REGION Network 8: XỬ LÍ CÂN CỐT LIỆU
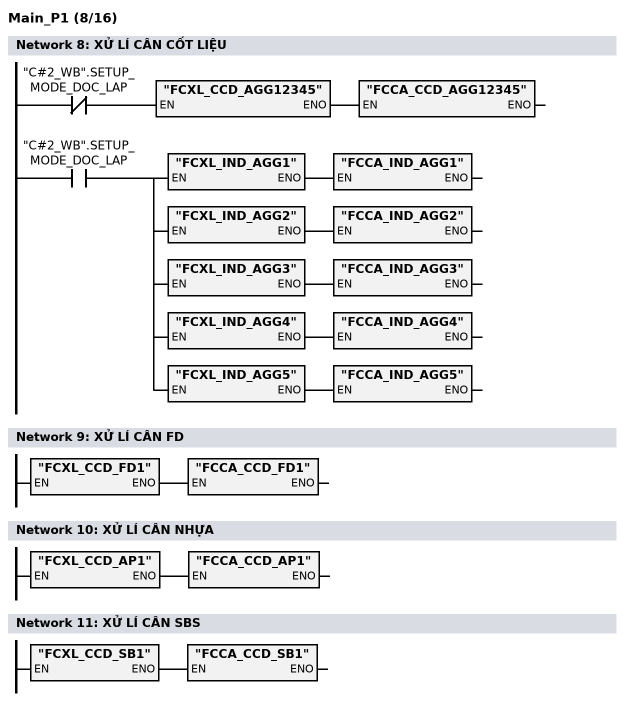
   RUNG wire#powerrail
      I_Contact( "C#2_WB".SETUP_MODE_DOC_LAP )
      "FCXL_CCD_AGG12345"()
      "FCCA_CCD_AGG12345"()
   END_RUNG
   RUNG wire#powerrail
      Contact( "C#2_WB".SETUP_MODE_DOC_LAP )
      wire#w1
      "FCXL_IND_AGG1"()
      "FCCA_IND_AGG1"()
   END_RUNG
   RUNG wire#w1
      "FCXL_IND_AGG2"()
      "FCCA_IND_AGG2"()
   END_RUNG
   RUNG wire#w1
      "FCXL_IND_AGG3"()
      "FCCA_IND_AGG3"()
   END_RUNG
   RUNG wire#w1
      "FCXL_IND_AGG4"()
      "FCCA_IND_AGG4"()
   END_RUNG
   RUNG wire#w1
      "FCXL_IND_AGG5"()
      "FCCA_IND_AGG5"()
   END_RUNG
   // the same network as SCL:
   "FCXL_CCD_AGG12345"(EN := NOT "C#2_WB".SETUP_MODE_DOC_LAP, ENO => #_w1);
   IF #_w1 THEN "FCCA_CCD_AGG12345"(); END_IF;
   #_w3 := "C#2_WB".SETUP_MODE_DOC_LAP;
   "FCXL_IND_AGG1"(EN := "C#2_WB".SETUP_MODE_DOC_LAP, ENO => #_w2);
   IF #_w2 THEN "FCCA_IND_AGG1"(); END_IF;
   "FCXL_IND_AGG2"(EN := #_w3, ENO => #_w4);
   IF #_w4 THEN "FCCA_IND_AGG2"(); END_IF;
   "FCXL_IND_AGG3"(EN := #_w3, ENO => #_w5);
   IF #_w5 THEN "FCCA_IND_AGG3"(); END_IF;
   "FCXL_IND_AGG4"(EN := #_w3, ENO => #_w6);
   IF #_w6 THEN "FCCA_IND_AGG4"(); END_IF;
   "FCXL_IND_AGG5"(EN := #_w3, ENO => #_w7);
   IF #_w7 THEN "FCCA_IND_AGG5"(); END_IF;
END_REGION

REGION Network 9: XỬ LÍ CÂN FD
   RUNG wire#powerrail
      "FCXL_CCD_FD1"()
      "FCCA_CCD_FD1"()
   END_RUNG
   // the same network as SCL:
   "FCXL_CCD_FD1"(ENO => #_w1);
   IF #_w1 THEN "FCCA_CCD_FD1"(); END_IF;
END_REGION

REGION Network 10: XỬ LÍ CÂN NHỰA
   RUNG wire#powerrail
      "FCXL_CCD_AP1"()
      "FCCA_CCD_AP1"()
   END_RUNG
   // the same network as SCL:
   "FCXL_CCD_AP1"(ENO => #_w1);
   IF #_w1 THEN "FCCA_CCD_AP1"(); END_IF;
END_REGION

REGION Network 11: XỬ LÍ CÂN SBS
   RUNG wire#powerrail
      "FCXL_CCD_SB1"()
      "FCCA_CCD_SB1"()
   END_RUNG
   // the same network as SCL:
   "FCXL_CCD_SB1"(ENO => #_w1);
   IF #_w1 THEN "FCCA_CCD_SB1"(); END_IF;
END_REGION

REGION Network 12: NẠP LIỆU NỒI TRỘN
   // Theo phân tích thì lẽ ra lệnh so sánh SV_FD1=0 nó phải bypass cả WCE1_FU thì mới đúng vì nếu theo logic cũ trong hàm xử lý cân (FC10 của FD1) tín hiệu SV_FD1=0 không bypass /NEXT_WCEM1 khiến WCE1_FU sẽ không được bật ON khi SV_FD1=0, dẫn đến mạch hở, không nạp liệu được.
   // Sau đó trong quá trình sửa đã bypass trong FC10, tuy nhiên làm như thế không hay, vì có cân đâu mà bảo nó FULL, vậy nên hay nhất sẽ là sửa ở đây, bypass WCE1_FU nếu như Setpoint của FD1=0
   // Lưu ý:
   // - Nhựa nóng thì cần có AP1 nên mới có lệnh so sánh SMX_AP1=SMC_MIXER và lệnh tiếp điểm WWA1_FU (cân đủ số mẻ và Full thì mới nạp được)
   // - Chỉ bypass bột đá FD1 hoặc phụ gia SB1 hoặc thậm chí bypass cả 2, nhưng không có chuyện bypass AP1
   // Nhựa nóng nên phải có nhựa, đó là lý do network này đang dự vào SMC_AP1 để so sánh với các SMC của các phểu cân FD1 và SBS1 (khoogn có AG1), mục đích là để kiểm tra xem các phểu cân đã được cân đầy và đủ thành phần chưa (có FD1/SBS1 không) (****)
   // - Lệnh so sánh SMX_FD1 hoặc SMX_SB1 với số mẻ trộn SMC_MIXER mục đích là để đảm bảo việc nạp liệu nó cần lặp lại giữa các mẻ. Logic ở đây là:
   // - Khi chưa nạp liêu (chưa nạp mẻ nào) thì SMC_MIXER tất nhiên là zero, và tất nhiên 2 thằng FD1 và SB1 nó cũng bằng zero, vì nó đã xả vào nồi mẻ nào đâu (lưu ý là sau khi nạp liệu xong thì biến NTR_FU sẽ bật và SMC_MIXER lúc này tăng lên 1)
   // - Vậy nên điều kiện này đúng, và tất nhiên trước khi xả thì tất cả các phểu cân phải có số mẻ cân bằng nhau nên nhận định 4**** ở trên là đúng (SMC_AP1=SMC_FD1=SMC_SB1), trừ khi không cân các thành phần này thì nó không bằng nhau, thì lúc đó có lệnh bypass lo.
   // - Còn lệnh so sánh SMX_AP1=SMC_MIXER là để kiểm tra việc xả các phểu cân liệu xong, rồi tới lúc nồi trộn nạp đầy NTR_FU thì SMC_MIXER tăng lên 1 (xem network13), đủ đk này thì mới nạp liệu lại được (nạp cho mẻ tiếp theo), logic ở đây là: lúc đầu chưa xả cái phểu nào thì 2 thông số này đều bằng zero đúng không, vậy thõa đk và có thể cho NẠP LIỆU, sau khi thằng AG1 nó xả/nạp vào nồi trộn thì SMX của nó tăng lên, tương tự cac phểu khác cũng có SMX tăng lên 1, trong đó có AP1, như vậy là NAP LIEU kết thúc, mà sau khi nạp liệu xong thì thằng nồi trộn nó phải xả ra chứ đúng không, vậy là một lúc sau khi nó trộn xong nó sẽ cả, lúc này SMX_MIXER sẽ tăng lên 1, làm điều kiện cần để cho một chu kỳ xả hay NẠP LIỆU tiếp theo.
   // - Sẽ có đứa hỏi, khi xả thì sẽ có thằng xả trước thằng xả sau, dẫn đến điều kiện so sánh nó không thỏa, mạch hở, NAP LIEU sẽ OFF, ví dụ như thằng SB1 nó ít nên nó xả lẹ hơn, empty sớm hơn mấy thằng kia, dẫn đến số mẻ xả của nó được tăng lên 1 sớm hơn, khi đó mất bit NAP LIEU thì các phểu các sao kịp xả.
   // ==> OK, phân tích tôt, nhưng chưa đủ sâu, cần phải biết là để xả/nạp liệu thì các phểu phải cân đủ liệu, và phải sẵn sàng hết tất cả sau đó mới nạp (tức thời điểm đó các điều kiện ở trên đều đã sẵn sàng), thứ 2 là NAP LIEU chỉ là đk cần cho việc bật tín hiệu NẠP tương ứng với tưng phểu cân, nhìn vào lệnh bên dưới sẽ thấy, và khi có NAP LIEU thì các tín hiệu sẽ được set lên đồng thời (vì điều kiện đã đợi sẵn hết cả rồi thím ợ, chỉ cần nhú lên là quất thôi).
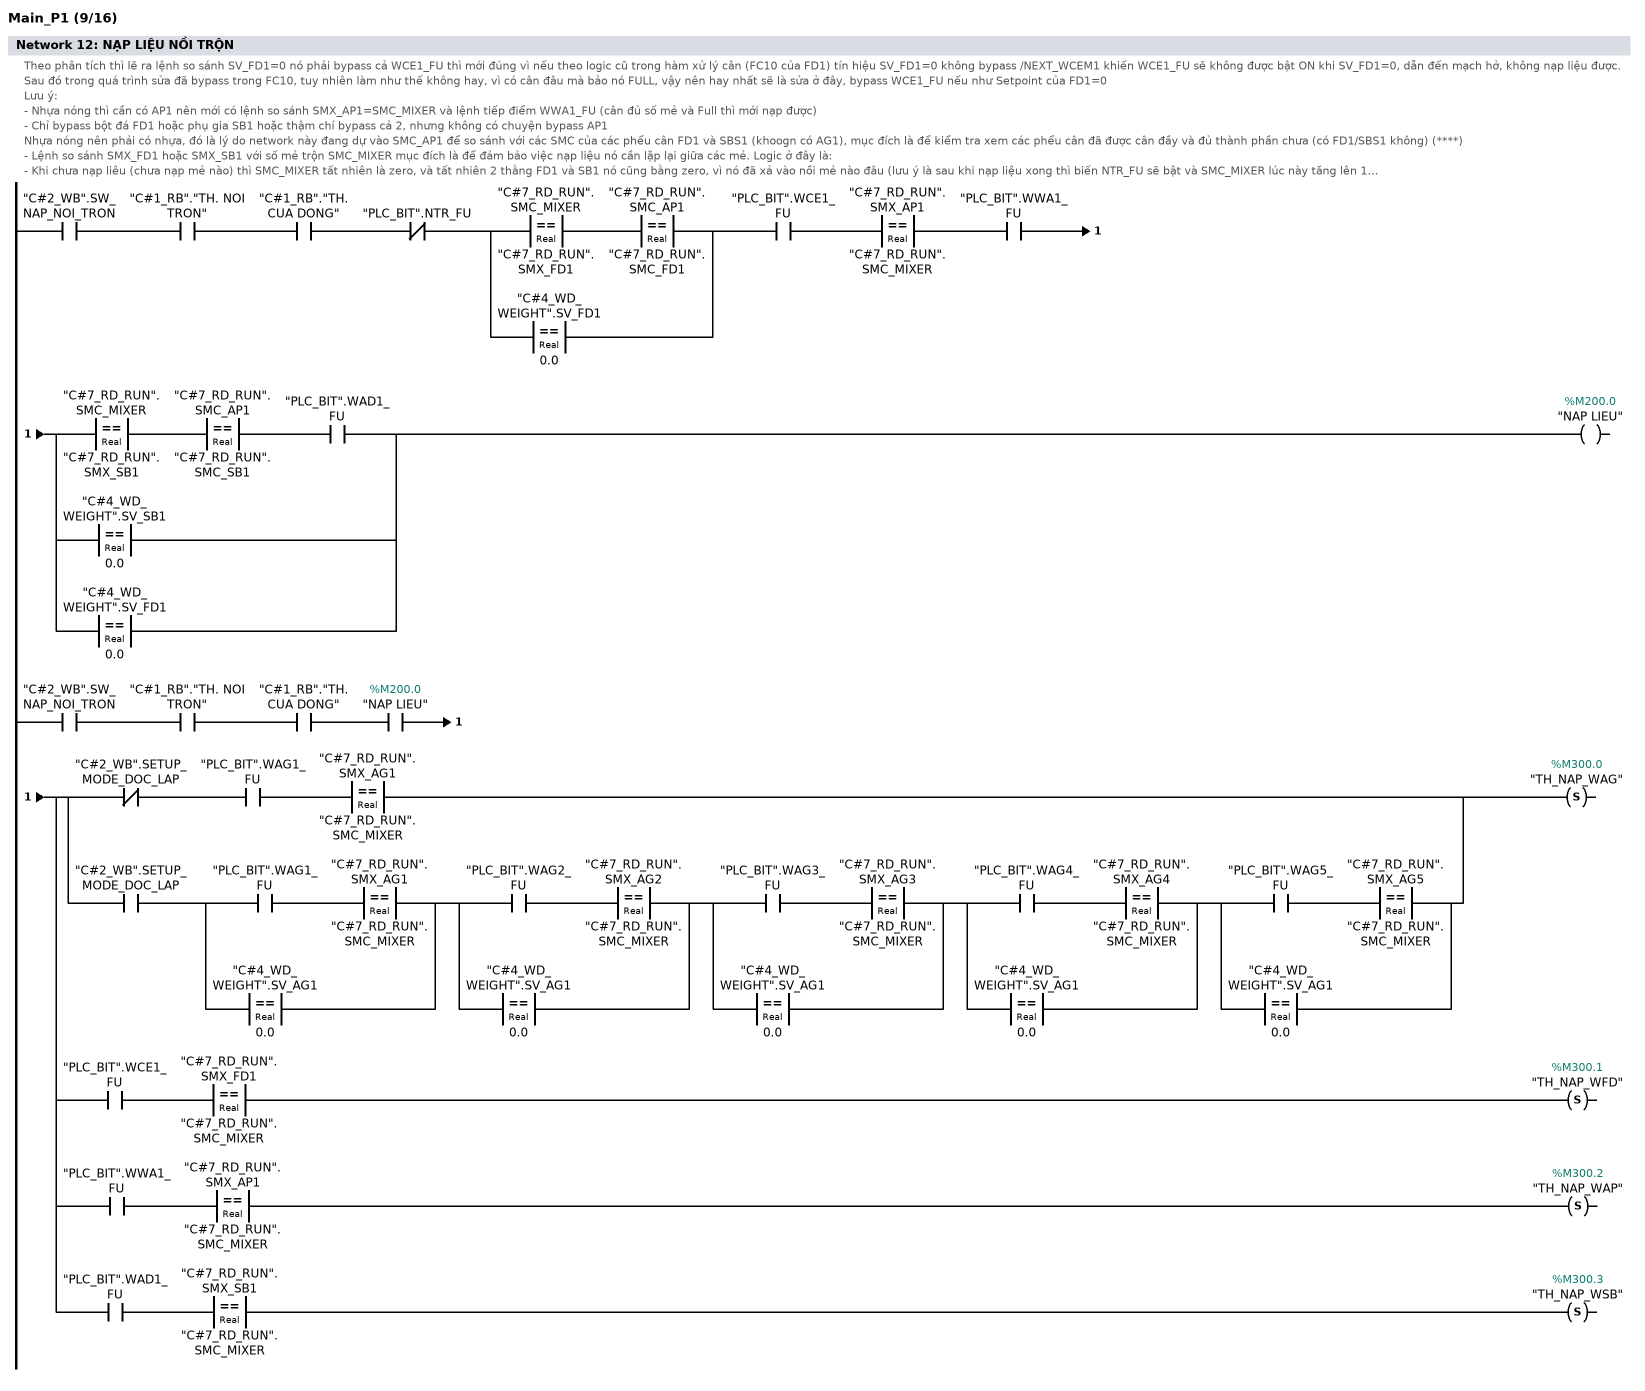
   RUNG wire#powerrail
      Contact( "C#2_WB".SW_NAP_NOI_TRON )
      Contact( "C#1_RB"."TH. NOI TRON" )
      Contact( "C#1_RB"."TH. CUA DONG" )
      I_Contact( "PLC_BIT".NTR_FU )
      wire#w1
      { S7_Templates := "SrcType := Real" } EQ_Contact(in1 := "C#7_RD_RUN".SMC_MIXER, in2 := "C#7_RD_RUN".SMX_FD1)
      { S7_Templates := "SrcType := Real" } EQ_Contact(in1 := "C#7_RD_RUN".SMC_AP1, in2 := "C#7_RD_RUN".SMC_FD1)
      wire#w2
      Contact( "PLC_BIT".WCE1_FU )
      { S7_Templates := "SrcType := Real" } EQ_Contact(in1 := "C#7_RD_RUN".SMX_AP1, in2 := "C#7_RD_RUN".SMC_MIXER)
      Contact( "PLC_BIT".WWA1_FU )
      wire#w3
      { S7_Templates := "SrcType := Real" } EQ_Contact(in1 := "C#7_RD_RUN".SMC_MIXER, in2 := "C#7_RD_RUN".SMX_SB1)
      { S7_Templates := "SrcType := Real" } EQ_Contact(in1 := "C#7_RD_RUN".SMC_AP1, in2 := "C#7_RD_RUN".SMC_SB1)
      Contact( "PLC_BIT".WAD1_FU )
      wire#w4
      Coil( "NAP LIEU" )
   END_RUNG
   RUNG wire#w1
      { S7_Templates := "SrcType := Real" } EQ_Contact(in1 := "C#4_WD_WEIGHT".SV_FD1, in2 := 0.0)
   END_RUNG wire#w2
   RUNG wire#w3
      { S7_Templates := "SrcType := Real" } EQ_Contact(in1 := "C#4_WD_WEIGHT".SV_SB1, in2 := 0.0)
   END_RUNG wire#w4
   RUNG wire#w3
      { S7_Templates := "SrcType := Real" } EQ_Contact(in1 := "C#4_WD_WEIGHT".SV_FD1, in2 := 0.0)
   END_RUNG wire#w4
   RUNG wire#powerrail
      Contact( "C#2_WB".SW_NAP_NOI_TRON )
      Contact( "C#1_RB"."TH. NOI TRON" )
      Contact( "C#1_RB"."TH. CUA DONG" )
      Contact( "NAP LIEU" )
      wire#w5
      I_Contact( "C#2_WB".SETUP_MODE_DOC_LAP )
      Contact( "PLC_BIT".WAG1_FU )
      { S7_Templates := "SrcType := Real" } EQ_Contact(in1 := "C#7_RD_RUN".SMX_AG1, in2 := "C#7_RD_RUN".SMC_MIXER)
      wire#w6
      S_Coil( "TH_NAP_WAG" )
   END_RUNG
   RUNG wire#w5
      Contact( "C#2_WB".SETUP_MODE_DOC_LAP )
      wire#w7
      Contact( "PLC_BIT".WAG1_FU )
      { S7_Templates := "SrcType := Real" } EQ_Contact(in1 := "C#7_RD_RUN".SMX_AG1, in2 := "C#7_RD_RUN".SMC_MIXER)
      wire#w8
      Contact( "PLC_BIT".WAG2_FU )
      { S7_Templates := "SrcType := Real" } EQ_Contact(in1 := "C#7_RD_RUN".SMX_AG2, in2 := "C#7_RD_RUN".SMC_MIXER)
      wire#w9
      Contact( "PLC_BIT".WAG3_FU )
      { S7_Templates := "SrcType := Real" } EQ_Contact(in1 := "C#7_RD_RUN".SMX_AG3, in2 := "C#7_RD_RUN".SMC_MIXER)
      wire#w10
      Contact( "PLC_BIT".WAG4_FU )
      { S7_Templates := "SrcType := Real" } EQ_Contact(in1 := "C#7_RD_RUN".SMX_AG4, in2 := "C#7_RD_RUN".SMC_MIXER)
      wire#w11
      Contact( "PLC_BIT".WAG5_FU )
      { S7_Templates := "SrcType := Real" } EQ_Contact(in1 := "C#7_RD_RUN".SMX_AG5, in2 := "C#7_RD_RUN".SMC_MIXER)
   END_RUNG wire#w6
   RUNG wire#w7
      { S7_Templates := "SrcType := Real" } EQ_Contact(in1 := "C#4_WD_WEIGHT".SV_AG1, in2 := 0.0)
   END_RUNG wire#w8
   RUNG wire#w8
      { S7_Templates := "SrcType := Real" } EQ_Contact(in1 := "C#4_WD_WEIGHT".SV_AG1, in2 := 0.0)
   END_RUNG wire#w9
   RUNG wire#w9
      { S7_Templates := "SrcType := Real" } EQ_Contact(in1 := "C#4_WD_WEIGHT".SV_AG1, in2 := 0.0)
   END_RUNG wire#w10
   RUNG wire#w10
      { S7_Templates := "SrcType := Real" } EQ_Contact(in1 := "C#4_WD_WEIGHT".SV_AG1, in2 := 0.0)
   END_RUNG wire#w11
   RUNG wire#w11
      { S7_Templates := "SrcType := Real" } EQ_Contact(in1 := "C#4_WD_WEIGHT".SV_AG1, in2 := 0.0)
   END_RUNG wire#w6
   RUNG wire#w5
      Contact( "PLC_BIT".WCE1_FU )
      { S7_Templates := "SrcType := Real" } EQ_Contact(in1 := "C#7_RD_RUN".SMX_FD1, in2 := "C#7_RD_RUN".SMC_MIXER)
      S_Coil( "TH_NAP_WFD" )
   END_RUNG
   RUNG wire#w5
      Contact( "PLC_BIT".WWA1_FU )
      { S7_Templates := "SrcType := Real" } EQ_Contact(in1 := "C#7_RD_RUN".SMX_AP1, in2 := "C#7_RD_RUN".SMC_MIXER)
      S_Coil( "TH_NAP_WAP" )
   END_RUNG
   RUNG wire#w5
      Contact( "PLC_BIT".WAD1_FU )
      { S7_Templates := "SrcType := Real" } EQ_Contact(in1 := "C#7_RD_RUN".SMX_SB1, in2 := "C#7_RD_RUN".SMC_MIXER)
      S_Coil( "TH_NAP_WSB" )
   END_RUNG
   // the same network as SCL:
   "NAP LIEU" := "C#2_WB".SW_NAP_NOI_TRON AND "C#1_RB"."TH. NOI TRON" AND "C#1_RB"."TH. CUA DONG" AND NOT "PLC_BIT".NTR_FU AND ((("C#7_RD_RUN".SMC_MIXER = "C#7_RD_RUN".SMX_FD1) AND ("C#7_RD_RUN".SMC_AP1 = "C#7_RD_RUN".SMC_FD1)) OR ("C#4_WD_WEIGHT".SV_FD1 = 0.0)) AND "PLC_BIT".WCE1_FU AND ("C#7_RD_RUN".SMX_AP1 = "C#7_RD_RUN".SMC_MIXER) AND "PLC_BIT".WWA1_FU AND ((("C#7_RD_RUN".SMC_MIXER = "C#7_RD_RUN".SMX_SB1) AND ("C#7_RD_RUN".SMC_AP1 = "C#7_RD_RUN".SMC_SB1) AND "PLC_BIT".WAD1_FU) OR ("C#4_WD_WEIGHT".SV_SB1 = 0.0) OR ("C#4_WD_WEIGHT".SV_FD1 = 0.0));
   #_w1 := "C#2_WB".SW_NAP_NOI_TRON AND "C#1_RB"."TH. NOI TRON" AND "C#1_RB"."TH. CUA DONG" AND "NAP LIEU";
   IF #_w1 AND ((NOT "C#2_WB".SETUP_MODE_DOC_LAP AND "PLC_BIT".WAG1_FU AND ("C#7_RD_RUN".SMX_AG1 = "C#7_RD_RUN".SMC_MIXER)) OR ("C#2_WB".SETUP_MODE_DOC_LAP AND (("PLC_BIT".WAG1_FU AND ("C#7_RD_RUN".SMX_AG1 = "C#7_RD_RUN".SMC_MIXER)) OR ("C#4_WD_WEIGHT".SV_AG1 = 0.0)) AND (("PLC_BIT".WAG2_FU AND ("C#7_RD_RUN".SMX_AG2 = "C#7_RD_RUN".SMC_MIXER)) OR ("C#4_WD_WEIGHT".SV_AG1 = 0.0)) AND (("PLC_BIT".WAG3_FU AND ("C#7_RD_RUN".SMX_AG3 = "C#7_RD_RUN".SMC_MIXER)) OR ("C#4_WD_WEIGHT".SV_AG1 = 0.0)) AND (("PLC_BIT".WAG4_FU AND ("C#7_RD_RUN".SMX_AG4 = "C#7_RD_RUN".SMC_MIXER)) OR ("C#4_WD_WEIGHT".SV_AG1 = 0.0)) AND (("PLC_BIT".WAG5_FU AND ("C#7_RD_RUN".SMX_AG5 = "C#7_RD_RUN".SMC_MIXER)) OR ("C#4_WD_WEIGHT".SV_AG1 = 0.0)))) THEN
       "TH_NAP_WAG" := TRUE;
   END_IF;
   IF #_w1 AND "PLC_BIT".WCE1_FU AND ("C#7_RD_RUN".SMX_FD1 = "C#7_RD_RUN".SMC_MIXER) THEN
       "TH_NAP_WFD" := TRUE;
   END_IF;
   IF #_w1 AND "PLC_BIT".WWA1_FU AND ("C#7_RD_RUN".SMX_AP1 = "C#7_RD_RUN".SMC_MIXER) THEN
       "TH_NAP_WAP" := TRUE;
   END_IF;
   IF #_w1 AND "PLC_BIT".WAD1_FU AND ("C#7_RD_RUN".SMX_SB1 = "C#7_RD_RUN".SMC_MIXER) THEN
       "TH_NAP_WSB" := TRUE;
   END_IF;
END_REGION

REGION Network 13: XỬ LÍ NỒI TRỘN
   // Đây là network xử lý tình huống là các phểu đã nạp/xả vào nồi trộn rồi, nhưng nồi trộn chưa có xả nhé (có thể là nó đang trộn nên mới đặt tên là NTR_FU, chứ thực tế thằng nồi trộn nó có cân mẹ đâu mà Full với không).
   // Lệnh so sánh SMX_AP1>SMC_MIXER sẽ thỏa, vì trước khi nạp vào nồi trộn thì SMC_AP1 cũng như các phểu cân khác đều sẽ lơn hơn SMC_MIXER, vụ thể là 1>0. mục đích là để việc bật bít NTR_FU diễn ra trước khi SMC_MIXER tăng lên 1, vì điều kiện đếm tăng là cạnh lên của NTR_FU mà.
   // @@@ XUỐNG TỚI NETWORK NÀY THÌ SMC_MIXER MỚI ĐƯỢC TĂNG LÊN 1@@@
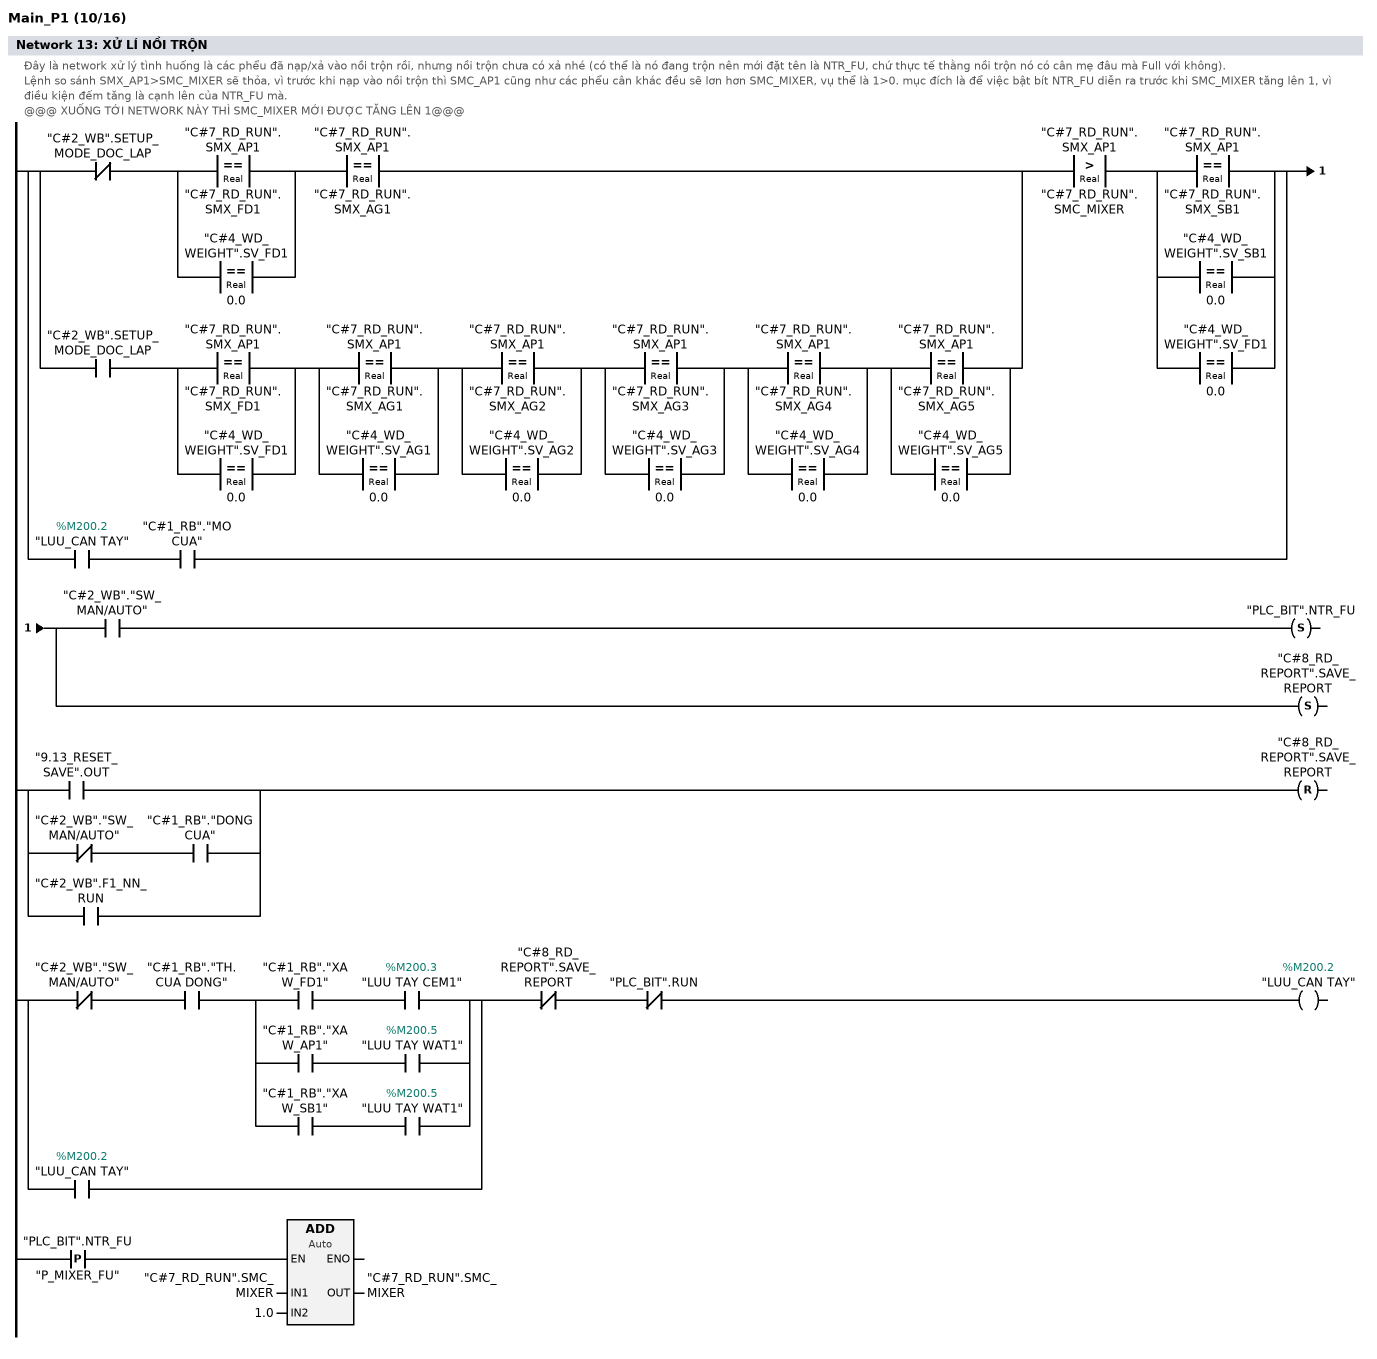
   RUNG wire#powerrail
      I_Contact( "C#2_WB".SETUP_MODE_DOC_LAP )
      wire#w1
      { S7_Templates := "SrcType := Real" } EQ_Contact(in1 := "C#7_RD_RUN".SMX_AP1, in2 := "C#7_RD_RUN".SMX_FD1)
      wire#w2
      { S7_Templates := "SrcType := Real" } EQ_Contact(in1 := "C#7_RD_RUN".SMX_AP1, in2 := "C#7_RD_RUN".SMX_AG1)
      wire#w3
      { S7_Templates := "SrcType := Real" } GT_Contact(in1 := "C#7_RD_RUN".SMX_AP1, in2 := "C#7_RD_RUN".SMC_MIXER)
      wire#w10
      { S7_Templates := "SrcType := Real" } EQ_Contact(in1 := "C#7_RD_RUN".SMX_AP1, in2 := "C#7_RD_RUN".SMX_SB1)
      wire#w11
      Contact( "C#2_WB"."SW_MAN/AUTO" )
      S_Coil( "PLC_BIT".NTR_FU )
   END_RUNG
   RUNG wire#w1
      { S7_Templates := "SrcType := Real" } EQ_Contact(in1 := "C#4_WD_WEIGHT".SV_FD1, in2 := 0.0)
   END_RUNG wire#w2
   RUNG wire#powerrail
      Contact( "C#2_WB".SETUP_MODE_DOC_LAP )
      wire#w4
      { S7_Templates := "SrcType := Real" } EQ_Contact(in1 := "C#7_RD_RUN".SMX_AP1, in2 := "C#7_RD_RUN".SMX_FD1)
      wire#w5
      { S7_Templates := "SrcType := Real" } EQ_Contact(in1 := "C#7_RD_RUN".SMX_AP1, in2 := "C#7_RD_RUN".SMX_AG1)
      wire#w6
      { S7_Templates := "SrcType := Real" } EQ_Contact(in1 := "C#7_RD_RUN".SMX_AP1, in2 := "C#7_RD_RUN".SMX_AG2)
      wire#w7
      { S7_Templates := "SrcType := Real" } EQ_Contact(in1 := "C#7_RD_RUN".SMX_AP1, in2 := "C#7_RD_RUN".SMX_AG3)
      wire#w8
      { S7_Templates := "SrcType := Real" } EQ_Contact(in1 := "C#7_RD_RUN".SMX_AP1, in2 := "C#7_RD_RUN".SMX_AG4)
      wire#w9
      { S7_Templates := "SrcType := Real" } EQ_Contact(in1 := "C#7_RD_RUN".SMX_AP1, in2 := "C#7_RD_RUN".SMX_AG5)
   END_RUNG wire#w3
   RUNG wire#w4
      { S7_Templates := "SrcType := Real" } EQ_Contact(in1 := "C#4_WD_WEIGHT".SV_FD1, in2 := 0.0)
   END_RUNG wire#w5
   RUNG wire#w5
      { S7_Templates := "SrcType := Real" } EQ_Contact(in1 := "C#4_WD_WEIGHT".SV_AG1, in2 := 0.0)
   END_RUNG wire#w6
   RUNG wire#w6
      { S7_Templates := "SrcType := Real" } EQ_Contact(in1 := "C#4_WD_WEIGHT".SV_AG2, in2 := 0.0)
   END_RUNG wire#w7
   RUNG wire#w7
      { S7_Templates := "SrcType := Real" } EQ_Contact(in1 := "C#4_WD_WEIGHT".SV_AG3, in2 := 0.0)
   END_RUNG wire#w8
   RUNG wire#w8
      { S7_Templates := "SrcType := Real" } EQ_Contact(in1 := "C#4_WD_WEIGHT".SV_AG4, in2 := 0.0)
   END_RUNG wire#w9
   RUNG wire#w9
      { S7_Templates := "SrcType := Real" } EQ_Contact(in1 := "C#4_WD_WEIGHT".SV_AG5, in2 := 0.0)
   END_RUNG wire#w3
   RUNG wire#w10
      { S7_Templates := "SrcType := Real" } EQ_Contact(in1 := "C#4_WD_WEIGHT".SV_SB1, in2 := 0.0)
   END_RUNG wire#w11
   RUNG wire#w10
      { S7_Templates := "SrcType := Real" } EQ_Contact(in1 := "C#4_WD_WEIGHT".SV_FD1, in2 := 0.0)
   END_RUNG wire#w11
   RUNG wire#powerrail
      Contact( "LUU_CAN TAY" )
      Contact( "C#1_RB"."MO CUA" )
   END_RUNG wire#w11
   RUNG wire#w11
      S_Coil( "C#8_RD_REPORT".SAVE_REPORT )
   END_RUNG
   RUNG wire#powerrail
      Contact( "9.13_RESET_SAVE".OUT )
      wire#w12
      R_Coil( "C#8_RD_REPORT".SAVE_REPORT )
   END_RUNG
   RUNG wire#powerrail
      I_Contact( "C#2_WB"."SW_MAN/AUTO" )
      Contact( "C#1_RB"."DONG CUA" )
   END_RUNG wire#w12
   RUNG wire#powerrail
      Contact( "C#2_WB".F1_NN_RUN )
   END_RUNG wire#w12
   RUNG wire#powerrail
      I_Contact( "C#2_WB"."SW_MAN/AUTO" )
      Contact( "C#1_RB"."TH. CUA DONG" )
      wire#w13
      Contact( "C#1_RB"."XA W_FD1" )
      Contact( "LUU TAY CEM1" )
      wire#w14
      I_Contact( "C#8_RD_REPORT".SAVE_REPORT )
      I_Contact( "PLC_BIT".RUN )
      Coil( "LUU_CAN TAY" )
   END_RUNG
   RUNG wire#w13
      Contact( "C#1_RB"."XA W_AP1" )
      Contact( "LUU TAY WAT1" )
   END_RUNG wire#w14
   RUNG wire#w13
      Contact( "C#1_RB"."XA W_SB1" )
      Contact( "LUU TAY WAT1" )
   END_RUNG wire#w14
   RUNG wire#powerrail
      Contact( "LUU_CAN TAY" )
   END_RUNG wire#w14
   RUNG wire#powerrail
      P_Contact(operand := "PLC_BIT".NTR_FU, bit := "P_MIXER_FU")
      Add(in1 := "C#7_RD_RUN".SMC_MIXER, in2 := 1.0, out => "C#7_RD_RUN".SMC_MIXER)
   END_RUNG
   // the same network as SCL:
   #_w1 := (((NOT "C#2_WB".SETUP_MODE_DOC_LAP AND (("C#7_RD_RUN".SMX_AP1 = "C#7_RD_RUN".SMX_FD1) OR ("C#4_WD_WEIGHT".SV_FD1 = 0.0)) AND ("C#7_RD_RUN".SMX_AP1 = "C#7_RD_RUN".SMX_AG1)) OR ("C#2_WB".SETUP_MODE_DOC_LAP AND (("C#7_RD_RUN".SMX_AP1 = "C#7_RD_RUN".SMX_FD1) OR ("C#4_WD_WEIGHT".SV_FD1 = 0.0)) AND (("C#7_RD_RUN".SMX_AP1 = "C#7_RD_RUN".SMX_AG1) OR ("C#4_WD_WEIGHT".SV_AG1 = 0.0)) AND (("C#7_RD_RUN".SMX_AP1 = "C#7_RD_RUN".SMX_AG2) OR ("C#4_WD_WEIGHT".SV_AG2 = 0.0)) AND (("C#7_RD_RUN".SMX_AP1 = "C#7_RD_RUN".SMX_AG3) OR ("C#4_WD_WEIGHT".SV_AG3 = 0.0)) AND (("C#7_RD_RUN".SMX_AP1 = "C#7_RD_RUN".SMX_AG4) OR ("C#4_WD_WEIGHT".SV_AG4 = 0.0)) AND (("C#7_RD_RUN".SMX_AP1 = "C#7_RD_RUN".SMX_AG5) OR ("C#4_WD_WEIGHT".SV_AG5 = 0.0)))) AND ("C#7_RD_RUN".SMX_AP1 > "C#7_RD_RUN".SMC_MIXER) AND (("C#7_RD_RUN".SMX_AP1 = "C#7_RD_RUN".SMX_SB1) OR ("C#4_WD_WEIGHT".SV_SB1 = 0.0) OR ("C#4_WD_WEIGHT".SV_FD1 = 0.0))) OR ("LUU_CAN TAY" AND "C#1_RB"."MO CUA");
   IF #_w1 AND "C#2_WB"."SW_MAN/AUTO" THEN "PLC_BIT".NTR_FU := TRUE; END_IF;
   IF #_w1 THEN "C#8_RD_REPORT".SAVE_REPORT := TRUE; END_IF;
   IF "9.13_RESET_SAVE".OUT OR (NOT "C#2_WB"."SW_MAN/AUTO" AND "C#1_RB"."DONG CUA") OR "C#2_WB".F1_NN_RUN THEN
       "C#8_RD_REPORT".SAVE_REPORT := FALSE;
   END_IF;
   "LUU_CAN TAY" := ((NOT "C#2_WB"."SW_MAN/AUTO" AND "C#1_RB"."TH. CUA DONG" AND (("C#1_RB"."XA W_FD1" AND "LUU TAY CEM1") OR ("C#1_RB"."XA W_AP1" AND "LUU TAY WAT1") OR ("C#1_RB"."XA W_SB1" AND "LUU TAY WAT1"))) OR "LUU_CAN TAY") AND NOT "C#8_RD_REPORT".SAVE_REPORT AND NOT "PLC_BIT".RUN;
   #_w2 := "PLC_BIT".NTR_FU AND NOT "P_MIXER_FU";   // rising edge of "PLC_BIT".NTR_FU
   "P_MIXER_FU" := "PLC_BIT".NTR_FU;
   IF #_w2 THEN "C#7_RD_RUN".SMC_MIXER := "C#7_RD_RUN".SMC_MIXER + 1.0; END_IF;
END_REGION

REGION Network 14: QUA TRÌNH NẠP LIỆU NỒI TRỘN
   // Network này sẽ bật các địa chỉ XẢ của phểu cân tương ứng nếu có tín hiệu NAP LIEU và các tín hiệu NAP_ của phểu cân tương ứng được bật lên
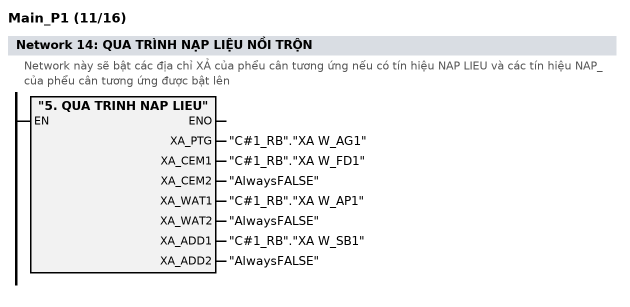
   RUNG wire#powerrail
      "5. QUA TRINH NAP LIEU"(XA_PTG => "C#1_RB"."XA W_AG1", XA_CEM1 => "C#1_RB"."XA W_FD1", XA_CEM2 => "AlwaysFALSE", XA_WAT1 => "C#1_RB"."XA W_AP1", XA_WAT2 => "AlwaysFALSE", XA_ADD1 => "C#1_RB"."XA W_SB1", XA_ADD2 => "AlwaysFALSE")
   END_RUNG
   // the same network as SCL:
   "5. QUA TRINH NAP LIEU"(XA_PTG => "C#1_RB"."XA W_AG1",
                           XA_CEM1 => "C#1_RB"."XA W_FD1",
                           XA_CEM2 => "AlwaysFALSE",
                           XA_WAT1 => "C#1_RB"."XA W_AP1",
                           XA_WAT2 => "AlwaysFALSE",
                           XA_ADD1 => "C#1_RB"."XA W_SB1",
                           XA_ADD2 => "AlwaysFALSE");
END_REGION

REGION Network 15: RESET NAP LIEU VA THOI GIAN TRE NAP SAU PTG
   // Ở chế độ CCD, việc xả sẽ theo trình tự, vậy nên sẽ có các timer để kiểm xoát, sử dụng hộp thoại cài đặt thời gian để cài đặt thời gian xả chậm hơn AGG là bao lâu (lúc trước chương trình ko có gửi giá trị cài đặt TG_Xa_FD_Sau_AG (Thời gian xả AP1 sau AGG), khả năng quên lập trình, nên lúc đó đã tạm thời thay thế địa chỉ cài đặt thời gian này thành thời gian xả SBS sau AGG, một giải pháp tạm). Theo đó, logic thời gian sẽ như sau:
   // - FD sẽ bắt đầu đếm thời gian sau khi phẩu cân AG1 có tín hiệu xả "C#1_RB"."XA W_AG1"
   // - AP1 và SBS1 sẽ bắt đầu đếm thời gian nếu như AG1 xả hết tức bít "PLC_BIT".WAG1_EM được bật
   // - Khi có tín hiệu nạp AP1, bơm tưới nhựa sẽ được bật (xả nhựa xuống là nó bơm luôn), nhưng nếu có cài thời gian cộng thêm cho nó thì sau khi phểu cân nhựa AP1 xả hết, nó sẽ bắt đầu đếm thời gian bơm nhựa thêm
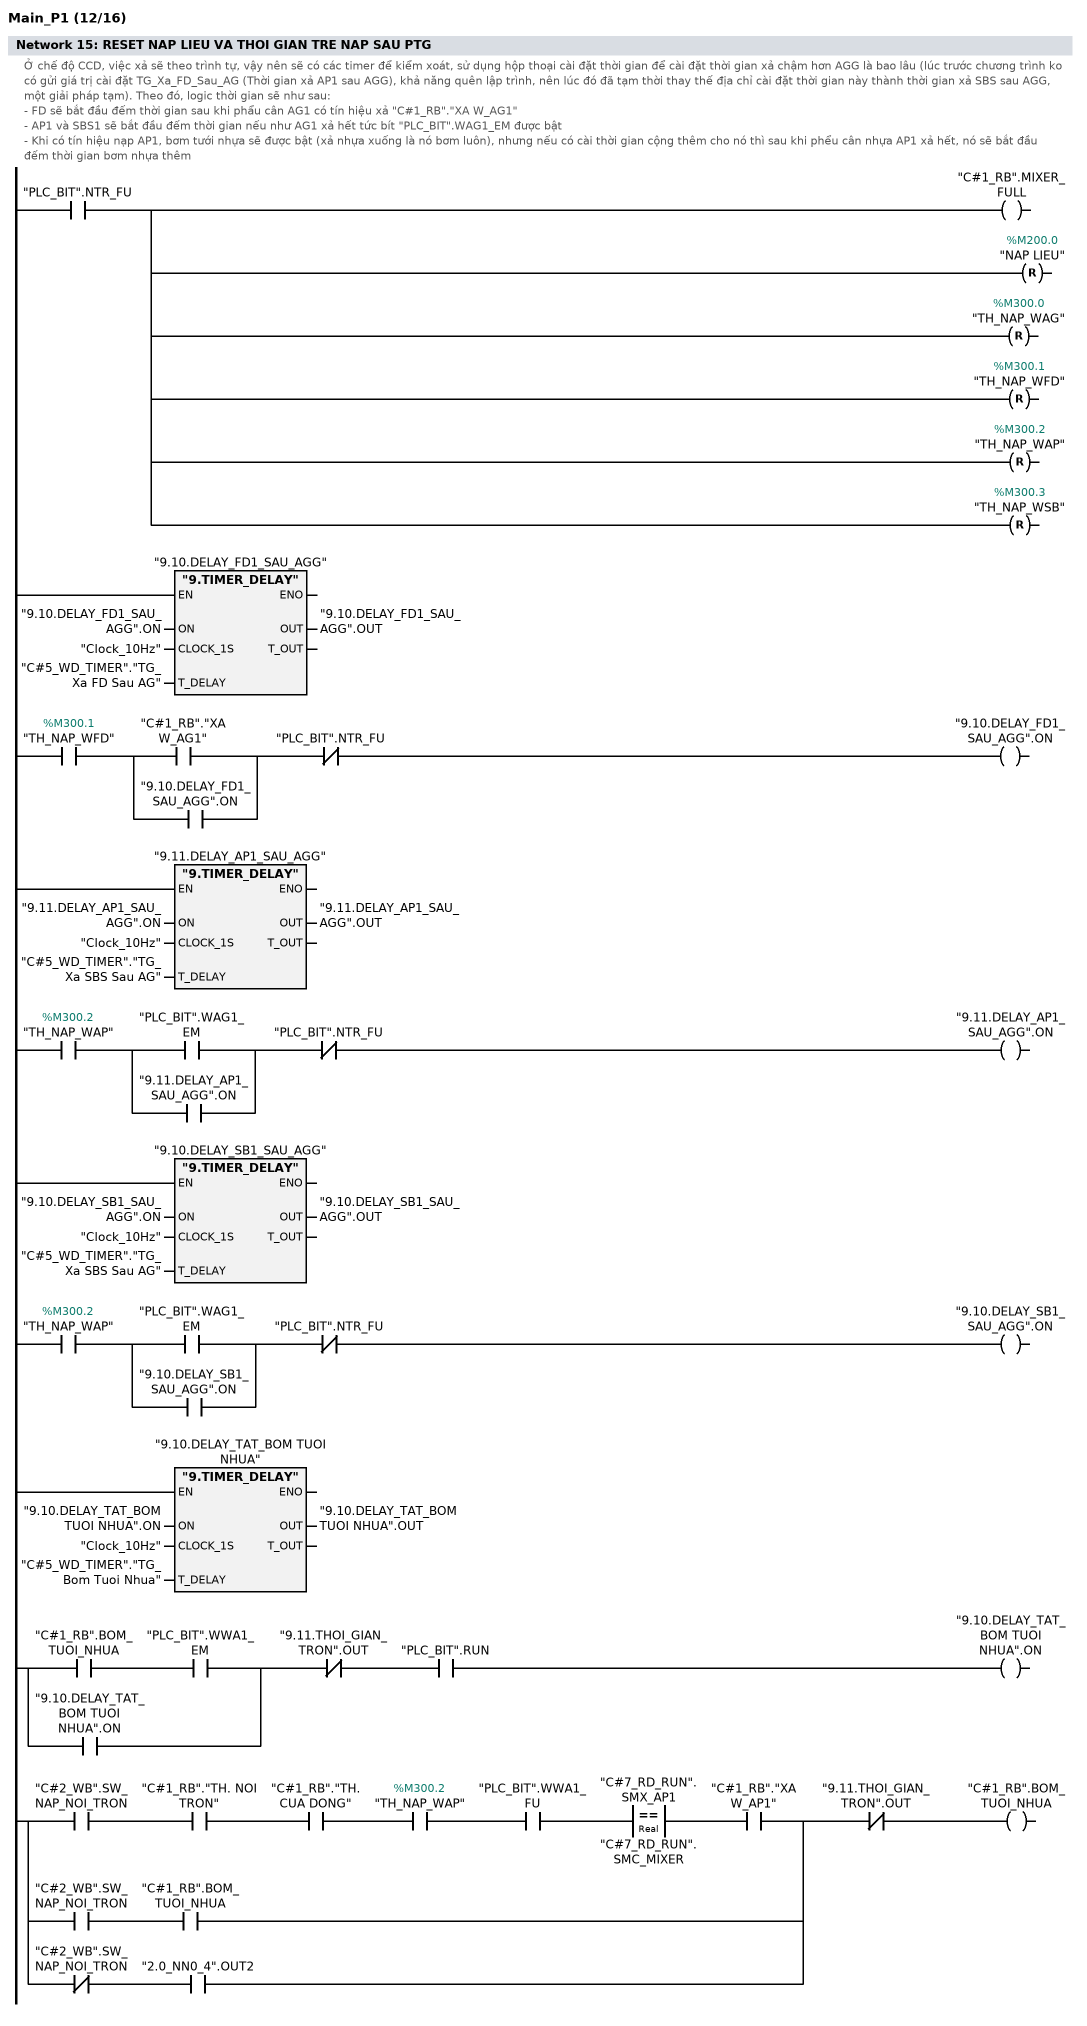
   RUNG wire#powerrail
      Contact( "PLC_BIT".NTR_FU )
      wire#w1
      Coil( "C#1_RB".MIXER_FULL )
   END_RUNG
   RUNG wire#w1
      R_Coil( "NAP LIEU" )
   END_RUNG
   RUNG wire#w1
      R_Coil( "TH_NAP_WAG" )
   END_RUNG
   RUNG wire#w1
      R_Coil( "TH_NAP_WFD" )
   END_RUNG
   RUNG wire#w1
      R_Coil( "TH_NAP_WAP" )
   END_RUNG
   RUNG wire#w1
      R_Coil( "TH_NAP_WSB" )
   END_RUNG
   RUNG wire#powerrail
      "9.10.DELAY_FD1_SAU_AGG"(ON := "9.10.DELAY_FD1_SAU_AGG".ON, CLOCK_1S := "Clock_10Hz", T_DELAY := "C#5_WD_TIMER"."TG_Xa FD Sau AG", OUT => "9.10.DELAY_FD1_SAU_AGG".OUT, T_OUT =>)
   END_RUNG
   RUNG wire#powerrail
      Contact( "TH_NAP_WFD" )
      wire#w2
      Contact( "C#1_RB"."XA W_AG1" )
      wire#w3
      I_Contact( "PLC_BIT".NTR_FU )
      Coil( "9.10.DELAY_FD1_SAU_AGG".ON )
   END_RUNG
   RUNG wire#w2
      Contact( "9.10.DELAY_FD1_SAU_AGG".ON )
   END_RUNG wire#w3
   RUNG wire#powerrail
      "9.11.DELAY_AP1_SAU_AGG"(ON := "9.11.DELAY_AP1_SAU_AGG".ON, CLOCK_1S := "Clock_10Hz", T_DELAY := "C#5_WD_TIMER"."TG_Xa SBS Sau AG", OUT => "9.11.DELAY_AP1_SAU_AGG".OUT, T_OUT =>)
   END_RUNG
   RUNG wire#powerrail
      Contact( "TH_NAP_WAP" )
      wire#w4
      Contact( "PLC_BIT".WAG1_EM )
      wire#w5
      I_Contact( "PLC_BIT".NTR_FU )
      Coil( "9.11.DELAY_AP1_SAU_AGG".ON )
   END_RUNG
   RUNG wire#w4
      Contact( "9.11.DELAY_AP1_SAU_AGG".ON )
   END_RUNG wire#w5
   RUNG wire#powerrail
      "9.10.DELAY_SB1_SAU_AGG"(ON := "9.10.DELAY_SB1_SAU_AGG".ON, CLOCK_1S := "Clock_10Hz", T_DELAY := "C#5_WD_TIMER"."TG_Xa SBS Sau AG", OUT => "9.10.DELAY_SB1_SAU_AGG".OUT, T_OUT =>)
   END_RUNG
   RUNG wire#powerrail
      Contact( "TH_NAP_WAP" )
      wire#w6
      Contact( "PLC_BIT".WAG1_EM )
      wire#w7
      I_Contact( "PLC_BIT".NTR_FU )
      Coil( "9.10.DELAY_SB1_SAU_AGG".ON )
   END_RUNG
   RUNG wire#w6
      Contact( "9.10.DELAY_SB1_SAU_AGG".ON )
   END_RUNG wire#w7
   RUNG wire#powerrail
      "9.10.DELAY_TAT_BOM TUOI NHUA"(ON := "9.10.DELAY_TAT_BOM TUOI NHUA".ON, CLOCK_1S := "Clock_10Hz", T_DELAY := "C#5_WD_TIMER"."TG_Bom Tuoi Nhua", OUT => "9.10.DELAY_TAT_BOM TUOI NHUA".OUT, T_OUT =>)
   END_RUNG
   RUNG wire#powerrail
      Contact( "C#1_RB".BOM_TUOI_NHUA )
      Contact( "PLC_BIT".WWA1_EM )
      wire#w8
      I_Contact( "9.11.THOI_GIAN_TRON".OUT )
      Contact( "PLC_BIT".RUN )
      Coil( "9.10.DELAY_TAT_BOM TUOI NHUA".ON )
   END_RUNG
   RUNG wire#powerrail
      Contact( "9.10.DELAY_TAT_BOM TUOI NHUA".ON )
   END_RUNG wire#w8
   RUNG wire#powerrail
      Contact( "C#2_WB".SW_NAP_NOI_TRON )
      Contact( "C#1_RB"."TH. NOI TRON" )
      Contact( "C#1_RB"."TH. CUA DONG" )
      Contact( "TH_NAP_WAP" )
      Contact( "PLC_BIT".WWA1_FU )
      { S7_Templates := "SrcType := Real" } EQ_Contact(in1 := "C#7_RD_RUN".SMX_AP1, in2 := "C#7_RD_RUN".SMC_MIXER)
      Contact( "C#1_RB"."XA W_AP1" )
      wire#w9
      I_Contact( "9.11.THOI_GIAN_TRON".OUT )
      Coil( "C#1_RB".BOM_TUOI_NHUA )
   END_RUNG
   RUNG wire#powerrail
      Contact( "C#2_WB".SW_NAP_NOI_TRON )
      Contact( "C#1_RB".BOM_TUOI_NHUA )
   END_RUNG wire#w9
   RUNG wire#powerrail
      I_Contact( "C#2_WB".SW_NAP_NOI_TRON )
      Contact( "2.0_NN0_4".OUT2 )
   END_RUNG wire#w9
   // the same network as SCL:
   "C#1_RB".MIXER_FULL := "PLC_BIT".NTR_FU;
   IF "PLC_BIT".NTR_FU THEN
       "NAP LIEU" := FALSE;
       "TH_NAP_WAG" := FALSE;
       "TH_NAP_WFD" := FALSE;
       "TH_NAP_WAP" := FALSE;
       "TH_NAP_WSB" := FALSE;
   END_IF;
   "9.10.DELAY_FD1_SAU_AGG"(ON := "9.10.DELAY_FD1_SAU_AGG".ON,   // "9.TIMER_DELAY"
                           CLOCK_1S := "Clock_10Hz",
                           T_DELAY := "C#5_WD_TIMER"."TG_Xa FD Sau AG",
                           OUT => "9.10.DELAY_FD1_SAU_AGG".OUT);
   "9.10.DELAY_FD1_SAU_AGG".ON := "TH_NAP_WFD" AND ("C#1_RB"."XA W_AG1" OR "9.10.DELAY_FD1_SAU_AGG".ON) AND NOT "PLC_BIT".NTR_FU;
   "9.11.DELAY_AP1_SAU_AGG"(ON := "9.11.DELAY_AP1_SAU_AGG".ON,   // "9.TIMER_DELAY"
                           CLOCK_1S := "Clock_10Hz",
                           T_DELAY := "C#5_WD_TIMER"."TG_Xa SBS Sau AG",
                           OUT => "9.11.DELAY_AP1_SAU_AGG".OUT);
   "9.11.DELAY_AP1_SAU_AGG".ON := "TH_NAP_WAP" AND ("PLC_BIT".WAG1_EM OR "9.11.DELAY_AP1_SAU_AGG".ON) AND NOT "PLC_BIT".NTR_FU;
   "9.10.DELAY_SB1_SAU_AGG"(ON := "9.10.DELAY_SB1_SAU_AGG".ON,   // "9.TIMER_DELAY"
                           CLOCK_1S := "Clock_10Hz",
                           T_DELAY := "C#5_WD_TIMER"."TG_Xa SBS Sau AG",
                           OUT => "9.10.DELAY_SB1_SAU_AGG".OUT);
   "9.10.DELAY_SB1_SAU_AGG".ON := "TH_NAP_WAP" AND ("PLC_BIT".WAG1_EM OR "9.10.DELAY_SB1_SAU_AGG".ON) AND NOT "PLC_BIT".NTR_FU;
   "9.10.DELAY_TAT_BOM TUOI NHUA"(ON := "9.10.DELAY_TAT_BOM TUOI NHUA".ON,   // "9.TIMER_DELAY"
                           CLOCK_1S := "Clock_10Hz",
                           T_DELAY := "C#5_WD_TIMER"."TG_Bom Tuoi Nhua",
                           OUT => "9.10.DELAY_TAT_BOM TUOI NHUA".OUT);
   "9.10.DELAY_TAT_BOM TUOI NHUA".ON := (("C#1_RB".BOM_TUOI_NHUA AND "PLC_BIT".WWA1_EM) OR "9.10.DELAY_TAT_BOM TUOI NHUA".ON) AND NOT "9.11.THOI_GIAN_TRON".OUT AND "PLC_BIT".RUN;
   "C#1_RB".BOM_TUOI_NHUA := (("C#2_WB".SW_NAP_NOI_TRON AND "C#1_RB"."TH. NOI TRON" AND "C#1_RB"."TH. CUA DONG" AND "TH_NAP_WAP" AND "PLC_BIT".WWA1_FU AND ("C#7_RD_RUN".SMX_AP1 = "C#7_RD_RUN".SMC_MIXER) AND "C#1_RB"."XA W_AP1") OR ("C#2_WB".SW_NAP_NOI_TRON AND "C#1_RB".BOM_TUOI_NHUA) OR (NOT "C#2_WB".SW_NAP_NOI_TRON AND "2.0_NN0_4".OUT2)) AND NOT "9.11.THOI_GIAN_TRON".OUT;
END_REGION

REGION Network 16: THOI GIAN TRON
   // Chỗ này tính thời gian TG_THUC TRON hơi dị, tại sao lại lấy giá trị cài đặt timer trừ đi giá trị đang đếm, nếu tính ra nó thời gian còn lại mà timer chưa đếm được do timer bị OFF đột ngột.
   // Cửa nổi sẽ bắt đầu mở sau thời gian cài đặt chính là thời gian Bơm tưới nhựa (thời gian cộng thêm)
   // Sau khi mở chạm giới hạn thì bắt đầu đếm thời gian xả được cài đặt bằng TG_XA 100, sau khi hết thời gian xả thì kích đóng cửa, cựa chạm vào giới hạn thì dừng.
   // @@@@Ở đây cần lưu ý:
   // - bít NTR_FU nó vẫn tồn tại cho đến chu trình xả, nó chỉ bị xóa đi khi đã kết thức quy trình xả
   // - SMX_MIXER sẽ được tăng lên 1 sau khi NTR_FU có cạnh xuống, hay chính xác hơn là khi nồi trộn xả hết mẻ đang trộn thì SMX_MIXER sẽ tăng lên 1 (hợp lý mà)
   // - Lệnh tăng SMC_MIXER bị lặp lại lần thứ 2, trước đó ở network 13 nó đã có rồi, ở đây lặp lại không cần thiêt.
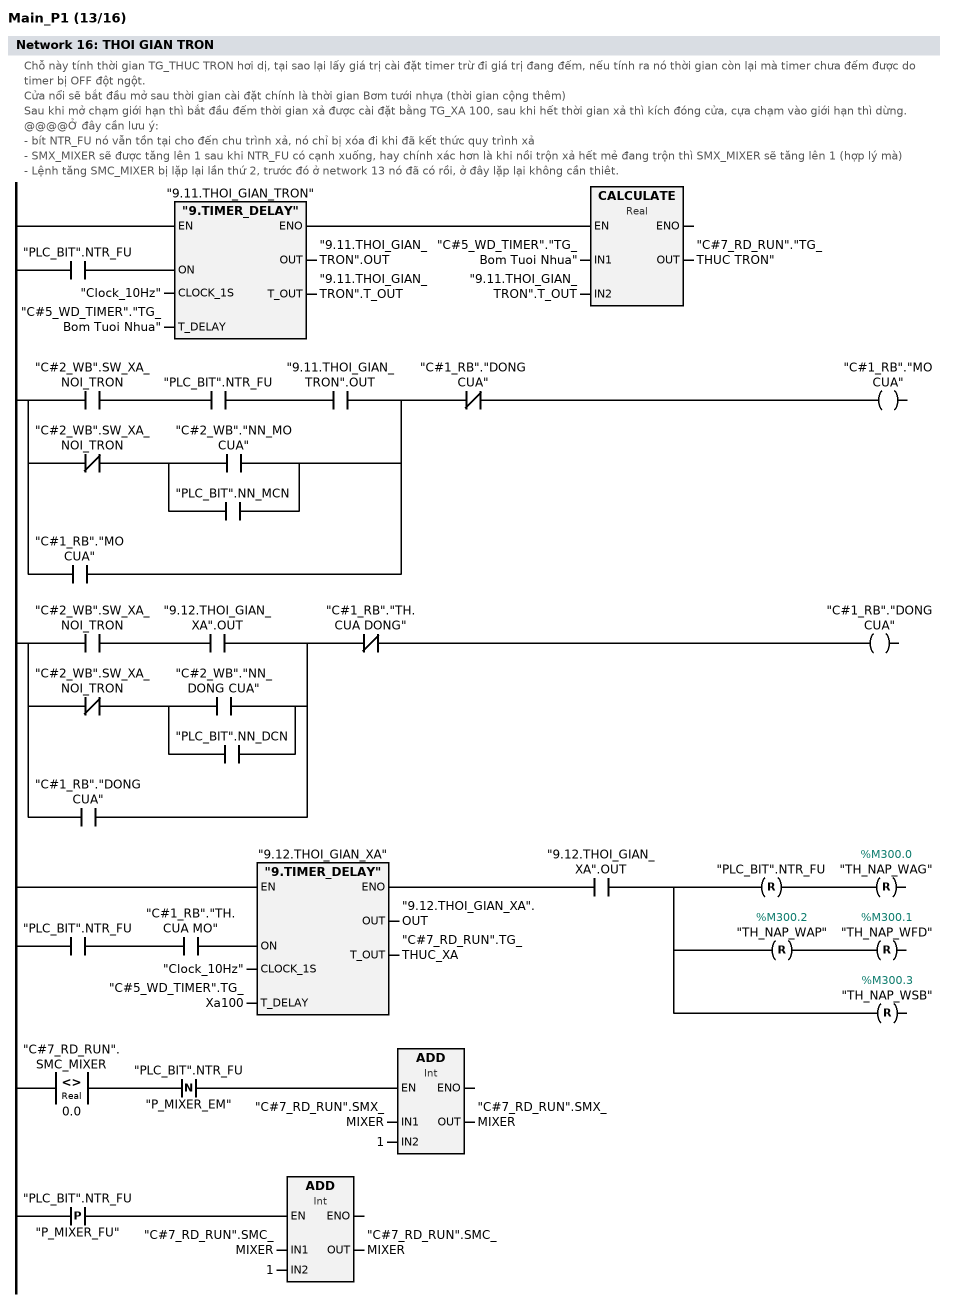
   RUNG wire#powerrail
      "9.11.THOI_GIAN_TRON"(ON := wire#w1, CLOCK_1S := "Clock_10Hz", T_DELAY := "C#5_WD_TIMER"."TG_Bom Tuoi Nhua", OUT => "9.11.THOI_GIAN_TRON".OUT, T_OUT => "9.11.THOI_GIAN_TRON".T_OUT)
      { S7_Templates := "SrcType := Real"; S7_Expression := "IN1-IN2" } Calculate(in1 := "C#5_WD_TIMER"."TG_Bom Tuoi Nhua", in2 := "9.11.THOI_GIAN_TRON".T_OUT, out => "C#7_RD_RUN"."TG_THUC TRON")
   END_RUNG
   RUNG wire#powerrail
      Contact( "PLC_BIT".NTR_FU )
   END_RUNG wire#w1
   RUNG wire#powerrail
      Contact( "C#2_WB".SW_XA_NOI_TRON )
      Contact( "PLC_BIT".NTR_FU )
      Contact( "9.11.THOI_GIAN_TRON".OUT )
      wire#w2
      I_Contact( "C#1_RB"."DONG CUA" )
      Coil( "C#1_RB"."MO CUA" )
   END_RUNG
   RUNG wire#powerrail
      I_Contact( "C#2_WB".SW_XA_NOI_TRON )
      wire#w3
      Contact( "C#2_WB"."NN_MO CUA" )
   END_RUNG wire#w2
   RUNG wire#w3
      Contact( "PLC_BIT".NN_MCN )
   END_RUNG wire#w2
   RUNG wire#powerrail
      Contact( "C#1_RB"."MO CUA" )
   END_RUNG wire#w2
   RUNG wire#powerrail
      Contact( "C#2_WB".SW_XA_NOI_TRON )
      Contact( "9.12.THOI_GIAN_XA".OUT )
      wire#w4
      I_Contact( "C#1_RB"."TH. CUA DONG" )
      Coil( "C#1_RB"."DONG CUA" )
   END_RUNG
   RUNG wire#powerrail
      I_Contact( "C#2_WB".SW_XA_NOI_TRON )
      wire#w5
      Contact( "C#2_WB"."NN_DONG CUA" )
   END_RUNG wire#w4
   RUNG wire#w5
      Contact( "PLC_BIT".NN_DCN )
   END_RUNG wire#w4
   RUNG wire#powerrail
      Contact( "C#1_RB"."DONG CUA" )
   END_RUNG wire#w4
   RUNG wire#powerrail
      "9.12.THOI_GIAN_XA"(ON := wire#w6, CLOCK_1S := "Clock_10Hz", T_DELAY := "C#5_WD_TIMER".TG_Xa100, OUT => "9.12.THOI_GIAN_XA".OUT, T_OUT => "C#7_RD_RUN".TG_THUC_XA)
      Contact( "9.12.THOI_GIAN_XA".OUT )
      wire#w7
      R_Coil( "PLC_BIT".NTR_FU )
      R_Coil( "TH_NAP_WAG" )
   END_RUNG
   RUNG wire#powerrail
      Contact( "PLC_BIT".NTR_FU )
      Contact( "C#1_RB"."TH. CUA MO" )
   END_RUNG wire#w6
   RUNG wire#w7
      R_Coil( "TH_NAP_WAP" )
      R_Coil( "TH_NAP_WFD" )
   END_RUNG
   RUNG wire#w7
      R_Coil( "TH_NAP_WSB" )
   END_RUNG
   RUNG wire#powerrail
      { S7_Templates := "SrcType := Real" } NE_Contact(in1 := "C#7_RD_RUN".SMC_MIXER, in2 := 0.0)
      N_Contact(operand := "PLC_BIT".NTR_FU, bit := "P_MIXER_EM")
      { S7_Templates := "SrcType := Int" } Add(in1 := "C#7_RD_RUN".SMX_MIXER, in2 := 1, out => "C#7_RD_RUN".SMX_MIXER)
   END_RUNG
   RUNG wire#powerrail
      P_Contact(operand := "PLC_BIT".NTR_FU, bit := "P_MIXER_FU")
      { S7_Templates := "SrcType := Int" } Add(in1 := "C#7_RD_RUN".SMC_MIXER, in2 := 1, out => "C#7_RD_RUN".SMC_MIXER)
   END_RUNG
   // the same network as SCL:
   "9.11.THOI_GIAN_TRON"(ON := "PLC_BIT".NTR_FU,   // "9.TIMER_DELAY"
                         CLOCK_1S := "Clock_10Hz",
                         T_DELAY := "C#5_WD_TIMER"."TG_Bom Tuoi Nhua",
                         OUT => "9.11.THOI_GIAN_TRON".OUT,
                         T_OUT => "9.11.THOI_GIAN_TRON".T_OUT,
                         ENO => #_w1);
   IF #_w1 THEN
       "C#7_RD_RUN"."TG_THUC TRON" := "C#5_WD_TIMER"."TG_Bom Tuoi Nhua"-"9.11.THOI_GIAN_TRON".T_OUT;
   END_IF;
   "C#1_RB"."MO CUA" := (("C#2_WB".SW_XA_NOI_TRON AND "PLC_BIT".NTR_FU AND "9.11.THOI_GIAN_TRON".OUT) OR (NOT "C#2_WB".SW_XA_NOI_TRON AND ("C#2_WB"."NN_MO CUA" OR "PLC_BIT".NN_MCN)) OR "C#1_RB"."MO CUA") AND NOT "C#1_RB"."DONG CUA";
   "C#1_RB"."DONG CUA" := (("C#2_WB".SW_XA_NOI_TRON AND "9.12.THOI_GIAN_XA".OUT) OR (NOT "C#2_WB".SW_XA_NOI_TRON AND ("C#2_WB"."NN_DONG CUA" OR "PLC_BIT".NN_DCN)) OR "C#1_RB"."DONG CUA") AND NOT "C#1_RB"."TH. CUA DONG";
   "9.12.THOI_GIAN_XA"(ON := "PLC_BIT".NTR_FU AND "C#1_RB"."TH. CUA MO",   // "9.TIMER_DELAY"
                       CLOCK_1S := "Clock_10Hz",
                       T_DELAY := "C#5_WD_TIMER".TG_Xa100,
                       OUT => "9.12.THOI_GIAN_XA".OUT,
                       T_OUT => "C#7_RD_RUN".TG_THUC_XA,
                       ENO => #_w2);
   IF #_w2 AND "9.12.THOI_GIAN_XA".OUT THEN
       "PLC_BIT".NTR_FU := FALSE;
       "TH_NAP_WAG" := FALSE;
       "TH_NAP_WAP" := FALSE;
       "TH_NAP_WFD" := FALSE;
       "TH_NAP_WSB" := FALSE;
   END_IF;
   #_w3 := ("C#7_RD_RUN".SMC_MIXER <> 0.0) AND NOT "PLC_BIT".NTR_FU AND "P_MIXER_EM";   // falling edge of "PLC_BIT".NTR_FU
   "P_MIXER_EM" := "PLC_BIT".NTR_FU;
   IF #_w3 THEN "C#7_RD_RUN".SMX_MIXER := "C#7_RD_RUN".SMX_MIXER + 1; END_IF;
   #_w4 := "PLC_BIT".NTR_FU AND NOT "P_MIXER_FU";   // rising edge of "PLC_BIT".NTR_FU
   "P_MIXER_FU" := "PLC_BIT".NTR_FU;
   IF #_w4 THEN "C#7_RD_RUN".SMC_MIXER := "C#7_RD_RUN".SMC_MIXER + 1; END_IF;
END_REGION

REGION Network 17: TEST SAVE DATA
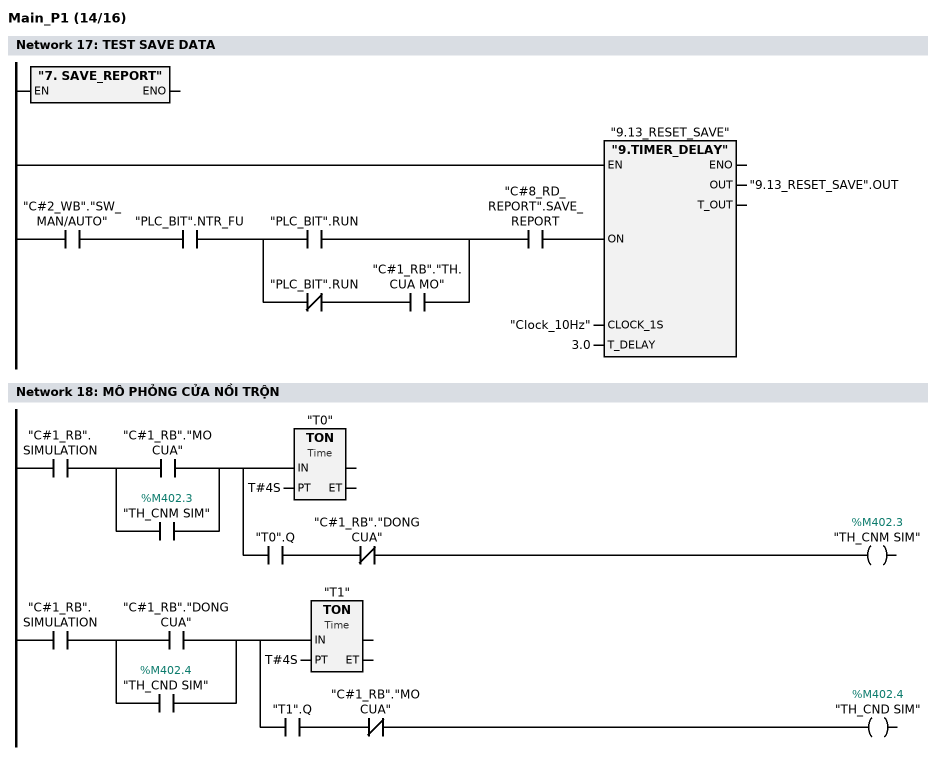
   RUNG wire#powerrail
      "7. SAVE_REPORT"()
   END_RUNG
   RUNG wire#powerrail
      "9.13_RESET_SAVE"(ON := wire#w3, CLOCK_1S := "Clock_10Hz", T_DELAY := 3.0, OUT => "9.13_RESET_SAVE".OUT, T_OUT =>)
   END_RUNG
   RUNG wire#powerrail
      Contact( "C#2_WB"."SW_MAN/AUTO" )
      Contact( "PLC_BIT".NTR_FU )
      wire#w1
      Contact( "PLC_BIT".RUN )
      wire#w2
      Contact( "C#8_RD_REPORT".SAVE_REPORT )
   END_RUNG wire#w3
   RUNG wire#w1
      I_Contact( "PLC_BIT".RUN )
      Contact( "C#1_RB"."TH. CUA MO" )
   END_RUNG wire#w2
   // the same network as SCL:
   "7. SAVE_REPORT"();
   "9.13_RESET_SAVE"(ON := "C#2_WB"."SW_MAN/AUTO" AND "PLC_BIT".NTR_FU AND ("PLC_BIT".RUN OR (NOT "PLC_BIT".RUN AND "C#1_RB"."TH. CUA MO")) AND "C#8_RD_REPORT".SAVE_REPORT,   // "9.TIMER_DELAY"
                     CLOCK_1S := "Clock_10Hz",
                     T_DELAY := 3.0,
                     OUT => "9.13_RESET_SAVE".OUT);
END_REGION

REGION Network 18: MÔ PHỎNG CỬA NỒI TRỘN
   RUNG wire#powerrail
      Contact( "C#1_RB".SIMULATION )
      wire#w1
      Contact( "C#1_RB"."MO CUA" )
      wire#w2
      { S7_Templates := "time_type := Time" } "T0".TON(pt := T#4S, et =>)
   END_RUNG
   RUNG wire#w1
      Contact( "TH_CNM SIM" )
   END_RUNG wire#w2
   RUNG wire#w2
      Contact( "T0".Q )
      I_Contact( "C#1_RB"."DONG CUA" )
      Coil( "TH_CNM SIM" )
   END_RUNG
   RUNG wire#powerrail
      Contact( "C#1_RB".SIMULATION )
      wire#w3
      Contact( "C#1_RB"."DONG CUA" )
      wire#w4
      { S7_Templates := "time_type := Time" } "T1".TON(pt := T#4S, et =>)
   END_RUNG
   RUNG wire#w3
      Contact( "TH_CND SIM" )
   END_RUNG wire#w4
   RUNG wire#w4
      Contact( "T1".Q )
      I_Contact( "C#1_RB"."MO CUA" )
      Coil( "TH_CND SIM" )
   END_RUNG
   // the same network as SCL:
   #_w1 := "C#1_RB".SIMULATION AND ("C#1_RB"."MO CUA" OR "TH_CNM SIM");
   "T0".TON(IN := #_w1, PT := T#4S);
   "TH_CNM SIM" := #_w1 AND "T0".Q AND NOT "C#1_RB"."DONG CUA";
   #_w2 := "C#1_RB".SIMULATION AND ("C#1_RB"."DONG CUA" OR "TH_CND SIM");
   "T1".TON(IN := #_w2, PT := T#4S);
   "TH_CND SIM" := #_w2 AND "T1".Q AND NOT "C#1_RB"."MO CUA";
END_REGION

REGION Network 19: CHẾ ĐỘ XẢ LIỆU
   // Cốt liệu ở đây là cac van Cát đá, khi người vận hành bật băng tải ngang và bật nút btnCheDoXaCan trên màn hình từ MAN sang Auto, thì cửa xả của các Cốt Liệu này sẽ được xả tự động nếu như Setpoint của các AGGx tương ứng khác 0, ở đây không thấy tín hiệu báo tràn AGx nó liên kết với Input hay nút nhấn nào trên màn hình (khả năng chưa có thiết lập).
   // Về cơ bản cách vận hành là người vận hành khi phát hiện tràn thì tắt chế độ xả Auto, và chuyển sang MAN, khi nào cần cốt liệu nào thì xả thủ công liệu đó.
   // Bên dưới có network dùng để rung các phểu này cho liệu nó rơi xuống, nếu bị kẹt (cái chấm tròn nhỏ trên phểu cân)
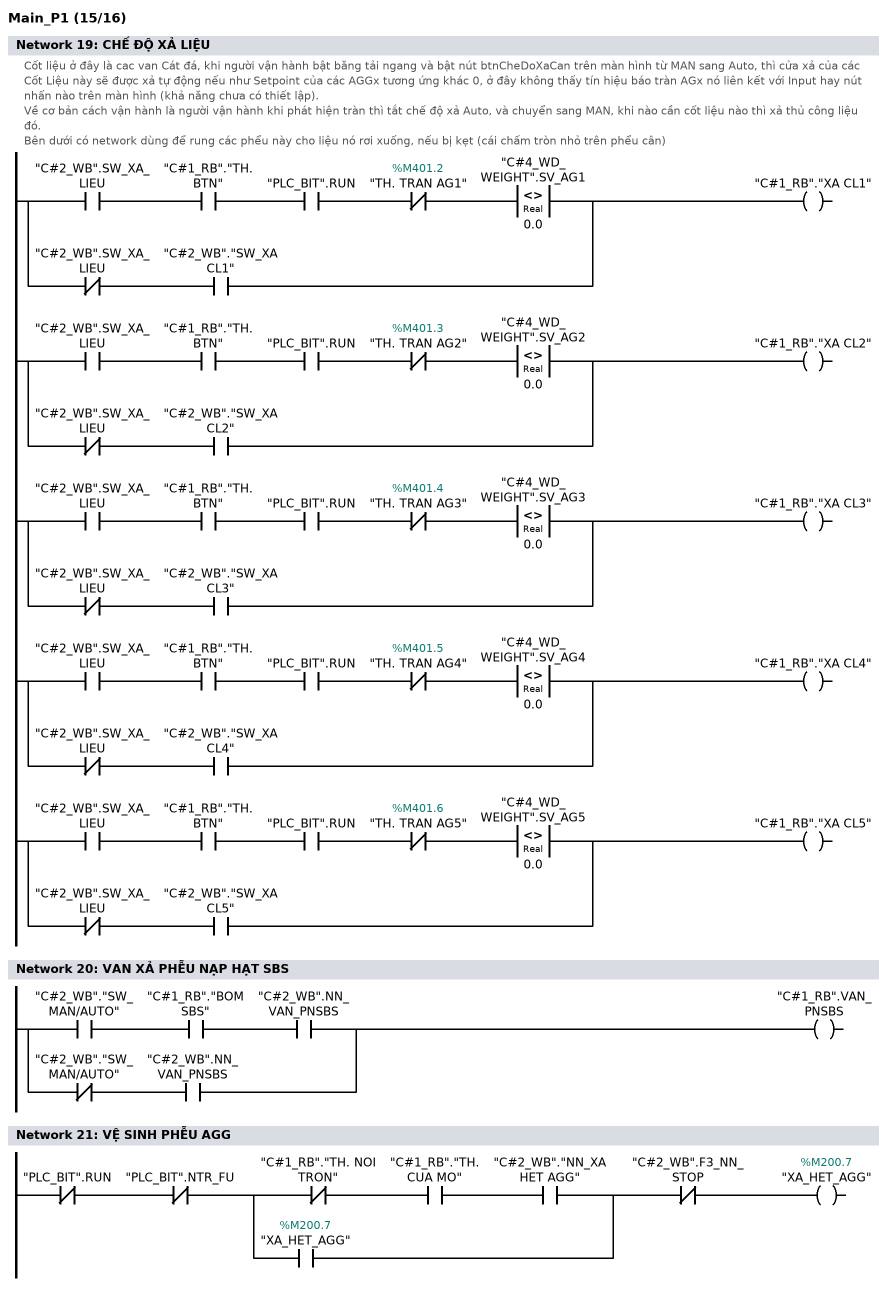
   RUNG wire#powerrail
      Contact( "C#2_WB".SW_XA_LIEU )
      Contact( "C#1_RB"."TH. BTN" )
      Contact( "PLC_BIT".RUN )
      I_Contact( "TH. TRAN AG1" )
      { S7_Templates := "SrcType := Real" } NE_Contact(in1 := "C#4_WD_WEIGHT".SV_AG1, in2 := 0.0)
      wire#w1
      Coil( "C#1_RB"."XA CL1" )
   END_RUNG
   RUNG wire#powerrail
      I_Contact( "C#2_WB".SW_XA_LIEU )
      Contact( "C#2_WB"."SW_XA CL1" )
   END_RUNG wire#w1
   RUNG wire#powerrail
      Contact( "C#2_WB".SW_XA_LIEU )
      Contact( "C#1_RB"."TH. BTN" )
      Contact( "PLC_BIT".RUN )
      I_Contact( "TH. TRAN AG2" )
      { S7_Templates := "SrcType := Real" } NE_Contact(in1 := "C#4_WD_WEIGHT".SV_AG2, in2 := 0.0)
      wire#w2
      Coil( "C#1_RB"."XA CL2" )
   END_RUNG
   RUNG wire#powerrail
      I_Contact( "C#2_WB".SW_XA_LIEU )
      Contact( "C#2_WB"."SW_XA CL2" )
   END_RUNG wire#w2
   RUNG wire#powerrail
      Contact( "C#2_WB".SW_XA_LIEU )
      Contact( "C#1_RB"."TH. BTN" )
      Contact( "PLC_BIT".RUN )
      I_Contact( "TH. TRAN AG3" )
      { S7_Templates := "SrcType := Real" } NE_Contact(in1 := "C#4_WD_WEIGHT".SV_AG3, in2 := 0.0)
      wire#w3
      Coil( "C#1_RB"."XA CL3" )
   END_RUNG
   RUNG wire#powerrail
      I_Contact( "C#2_WB".SW_XA_LIEU )
      Contact( "C#2_WB"."SW_XA CL3" )
   END_RUNG wire#w3
   RUNG wire#powerrail
      Contact( "C#2_WB".SW_XA_LIEU )
      Contact( "C#1_RB"."TH. BTN" )
      Contact( "PLC_BIT".RUN )
      I_Contact( "TH. TRAN AG4" )
      { S7_Templates := "SrcType := Real" } NE_Contact(in1 := "C#4_WD_WEIGHT".SV_AG4, in2 := 0.0)
      wire#w4
      Coil( "C#1_RB"."XA CL4" )
   END_RUNG
   RUNG wire#powerrail
      I_Contact( "C#2_WB".SW_XA_LIEU )
      Contact( "C#2_WB"."SW_XA CL4" )
   END_RUNG wire#w4
   RUNG wire#powerrail
      Contact( "C#2_WB".SW_XA_LIEU )
      Contact( "C#1_RB"."TH. BTN" )
      Contact( "PLC_BIT".RUN )
      I_Contact( "TH. TRAN AG5" )
      { S7_Templates := "SrcType := Real" } NE_Contact(in1 := "C#4_WD_WEIGHT".SV_AG5, in2 := 0.0)
      wire#w5
      Coil( "C#1_RB"."XA CL5" )
   END_RUNG
   RUNG wire#powerrail
      I_Contact( "C#2_WB".SW_XA_LIEU )
      Contact( "C#2_WB"."SW_XA CL5" )
   END_RUNG wire#w5
   // the same network as SCL:
   "C#1_RB"."XA CL1" := ("C#2_WB".SW_XA_LIEU AND "C#1_RB"."TH. BTN" AND "PLC_BIT".RUN AND NOT "TH. TRAN AG1" AND ("C#4_WD_WEIGHT".SV_AG1 <> 0.0)) OR (NOT "C#2_WB".SW_XA_LIEU AND "C#2_WB"."SW_XA CL1");
   "C#1_RB"."XA CL2" := ("C#2_WB".SW_XA_LIEU AND "C#1_RB"."TH. BTN" AND "PLC_BIT".RUN AND NOT "TH. TRAN AG2" AND ("C#4_WD_WEIGHT".SV_AG2 <> 0.0)) OR (NOT "C#2_WB".SW_XA_LIEU AND "C#2_WB"."SW_XA CL2");
   "C#1_RB"."XA CL3" := ("C#2_WB".SW_XA_LIEU AND "C#1_RB"."TH. BTN" AND "PLC_BIT".RUN AND NOT "TH. TRAN AG3" AND ("C#4_WD_WEIGHT".SV_AG3 <> 0.0)) OR (NOT "C#2_WB".SW_XA_LIEU AND "C#2_WB"."SW_XA CL3");
   "C#1_RB"."XA CL4" := ("C#2_WB".SW_XA_LIEU AND "C#1_RB"."TH. BTN" AND "PLC_BIT".RUN AND NOT "TH. TRAN AG4" AND ("C#4_WD_WEIGHT".SV_AG4 <> 0.0)) OR (NOT "C#2_WB".SW_XA_LIEU AND "C#2_WB"."SW_XA CL4");
   "C#1_RB"."XA CL5" := ("C#2_WB".SW_XA_LIEU AND "C#1_RB"."TH. BTN" AND "PLC_BIT".RUN AND NOT "TH. TRAN AG5" AND ("C#4_WD_WEIGHT".SV_AG5 <> 0.0)) OR (NOT "C#2_WB".SW_XA_LIEU AND "C#2_WB"."SW_XA CL5");
END_REGION

REGION Network 20: VAN XẢ PHỄU NẠP HẠT SBS
   RUNG wire#powerrail
      Contact( "C#2_WB"."SW_MAN/AUTO" )
      Contact( "C#1_RB"."BOM SBS" )
      Contact( "C#2_WB".NN_VAN_PNSBS )
      wire#w1
      Coil( "C#1_RB".VAN_PNSBS )
   END_RUNG
   RUNG wire#powerrail
      I_Contact( "C#2_WB"."SW_MAN/AUTO" )
      Contact( "C#2_WB".NN_VAN_PNSBS )
   END_RUNG wire#w1
   // the same network as SCL:
   "C#1_RB".VAN_PNSBS := ("C#2_WB"."SW_MAN/AUTO" AND "C#1_RB"."BOM SBS" AND "C#2_WB".NN_VAN_PNSBS) OR (NOT "C#2_WB"."SW_MAN/AUTO" AND "C#2_WB".NN_VAN_PNSBS);
END_REGION

REGION Network 21: VỆ SINH PHỄU AGG
   RUNG wire#powerrail
      I_Contact( "PLC_BIT".RUN )
      I_Contact( "PLC_BIT".NTR_FU )
      wire#w1
      I_Contact( "C#1_RB"."TH. NOI TRON" )
      Contact( "C#1_RB"."TH. CUA MO" )
      Contact( "C#2_WB"."NN_XA HET AGG" )
      wire#w2
      I_Contact( "C#2_WB".F3_NN_STOP )
      Coil( "XA_HET_AGG" )
   END_RUNG
   RUNG wire#w1
      Contact( "XA_HET_AGG" )
   END_RUNG wire#w2
   // the same network as SCL:
   "XA_HET_AGG" := NOT "PLC_BIT".RUN AND NOT "PLC_BIT".NTR_FU AND ((NOT "C#1_RB"."TH. NOI TRON" AND "C#1_RB"."TH. CUA MO" AND "C#2_WB"."NN_XA HET AGG") OR "XA_HET_AGG") AND NOT "C#2_WB".F3_NN_STOP;
END_REGION

REGION Network 22: RUNG PHEU COT LIEU
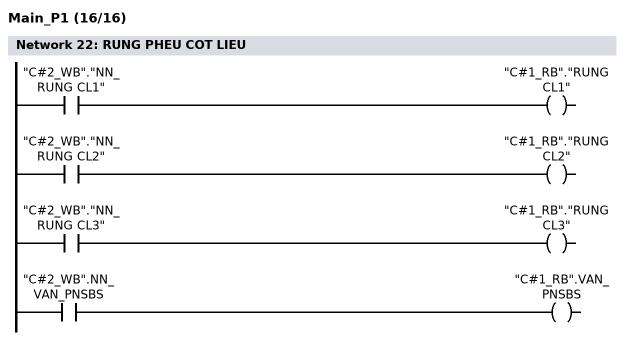
   RUNG wire#powerrail
      Contact( "C#2_WB"."NN_RUNG CL1" )
      Coil( "C#1_RB"."RUNG CL1" )
   END_RUNG
   RUNG wire#powerrail
      Contact( "C#2_WB"."NN_RUNG CL2" )
      Coil( "C#1_RB"."RUNG CL2" )
   END_RUNG
   RUNG wire#powerrail
      Contact( "C#2_WB"."NN_RUNG CL3" )
      Coil( "C#1_RB"."RUNG CL3" )
   END_RUNG
   RUNG wire#powerrail
      Contact( "C#2_WB".NN_VAN_PNSBS )
      Coil( "C#1_RB".VAN_PNSBS )
   END_RUNG
   // the same network as SCL:
   "C#1_RB"."RUNG CL1" := "C#2_WB"."NN_RUNG CL1";
   "C#1_RB"."RUNG CL2" := "C#2_WB"."NN_RUNG CL2";
   "C#1_RB"."RUNG CL3" := "C#2_WB"."NN_RUNG CL3";
   "C#1_RB".VAN_PNSBS := "C#2_WB".NN_VAN_PNSBS;
END_REGION
END_ORGANIZATION_BLOCK

FUNCTION "2.MOVE_OUT" : Void   // FC2, LAD
{ S7_Optimized_Access := 'TRUE' }
VERSION : 0.1
// stored: AutoNumber false, CodeModifiedDate 2025-08-27T17:06:54.9207011Z, CompileDate 2026-01-15T16:25:52.8890325Z, CreationDate 2026-01-15T16:22:49.8270549Z, HandleErrorsWithinBlock false, InterfaceModifiedDate 2023-08-09T15:10:11.0888586Z, IsConsistent true, IsIECCheckEnabled false, IsKnowHowProtected false, IsWriteProtected false, LibraryConformanceStatus The object is library-conformant., ModifiedDate 2025-08-27T17:06:54.9207011Z, ParameterModified 2023-08-09T15:10:11.0888586Z, PLCSimAdvancedSupport false, SetENOAutomatically False, StructureModified 2023-08-09T15:10:11.0888586Z, UDAEnableTagReadback false
   VAR_INPUT
      "0.0" : Bool;
      "0.1" : Bool;
      "0.2" : Bool;
      "0.3" : Bool;
      "0.4" : Bool;
      "0.5" : Bool;
      "0.6" : Bool;
      "0.7" : Bool;
   END_VAR
   VAR_OUTPUT
      "0_0" : Bool;
      "0_1" : Bool;
      "0_2" : Bool;
      "0_3" : Bool;
      "0_4" : Bool;
      "0_5" : Bool;
      "0_6" : Bool;
      "0_7" : Bool;
   END_VAR
BEGIN

REGION Network 3
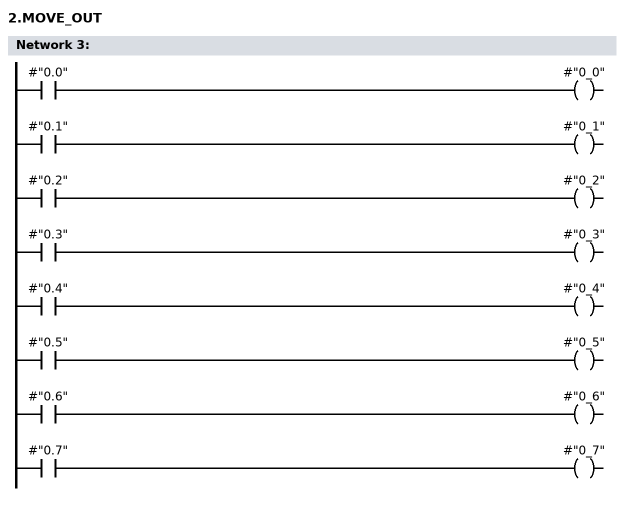
   RUNG wire#powerrail
      Contact( #"0.0" )
      Coil( #"0_0" )
   END_RUNG
   RUNG wire#powerrail
      Contact( #"0.1" )
      Coil( #"0_1" )
   END_RUNG
   RUNG wire#powerrail
      Contact( #"0.2" )
      Coil( #"0_2" )
   END_RUNG
   RUNG wire#powerrail
      Contact( #"0.3" )
      Coil( #"0_3" )
   END_RUNG
   RUNG wire#powerrail
      Contact( #"0.4" )
      Coil( #"0_4" )
   END_RUNG
   RUNG wire#powerrail
      Contact( #"0.5" )
      Coil( #"0_5" )
   END_RUNG
   RUNG wire#powerrail
      Contact( #"0.6" )
      Coil( #"0_6" )
   END_RUNG
   RUNG wire#powerrail
      Contact( #"0.7" )
      Coil( #"0_7" )
   END_RUNG
   // the same network as SCL:
   #"0_0" := #"0.0";
   #"0_1" := #"0.1";
   #"0_2" := #"0.2";
   #"0_3" := #"0.3";
   #"0_4" := #"0.4";
   #"0_5" := #"0.5";
   #"0_6" := #"0.6";
   #"0_7" := #"0.7";
END_REGION
END_FUNCTION

FUNCTION_BLOCK "2.MANUAL_CONTROL"   // FB2, LAD
TITLE = MODE=0 thì nhấn dạng Toggle, MODE=1 thì nhấn như một nút nhấn thông thường, nếu RS=1 thì ngõ ra sẽ bị Reset
{ S7_Optimized_Access := 'TRUE' }
VERSION : 0.1
// Chức năng của FB: xác định phương thức tác động khi nhấn nút NN1, NN2, NN3 theo 2 cách
// Cách 1: MODE = 0, thực hiện như một Toggle, mỗi lần nhấn sẽ đổi trạng thái OUT, từ OFF sang ON và ngược lại.
// NN là nút nhấn trên HMI/SCADA
// OUT là ngõ ra cần được SET hoặc RESET
// ST chính là OUT (nó như là phản hồi để biết OUT đang được SET hay RESET
// RS là tín hiệu để reset ngõ ra
// Nó dùng M là một biến Static để lưu số lần nhấn nút (ban đầu nếu chưa có ngõ ra OUT, thì M là 0, nhưng khi đã có OUT thì M  là 1), từ đây nếu NN nhấn mà chưa có OUT thì OUT11 sẽ được SET, còn nếu NN được nhấn mà có OUT11 thì sẽ Reset OUT11 đi)
// Cách 2: MODE=1, nó thực hiện như một nút nhấn mình thường dạng Momentory, nghĩa là Nhấn thì đầu ra sẽ có, còn nhả ra thì mất OUT.
// stored: AutoNumber false, CodeModifiedDate 2025-08-27T17:14:33.2091456Z, CompileDate 2026-01-15T16:25:51.6735735Z, CreationDate 2026-01-15T16:22:49.8270549Z, DownloadWithoutReinit false, HandleErrorsWithinBlock false, InterfaceModifiedDate 2025-08-27T17:14:33.2091456Z, IsConsistent true, IsIECCheckEnabled false, IsKnowHowProtected false, IsRetainMemResEnabled false, IsWriteProtected false, LibraryConformanceStatus The object is library-conformant., MemoryReserve 100, ModifiedDate 2025-10-23T13:27:09.8211701Z, ParameterModified 2024-10-13T14:59:19.5830719Z, PLCSimAdvancedSupport false, SetENOAutomatically False, StructureModified 2025-08-27T17:14:33.2091456Z, UDAEnableTagReadback false
   VAR_INPUT
      MODE : Bool;
      NN1 : Bool;
      NN2 : Bool;
      NN3 : Bool;
      ST1 : Bool;
      ST2 : Bool;
      ST3 : Bool;
      RS1 : Bool;
      RS2 : Bool;
      RS3 : Bool;
   END_VAR
   VAR_OUTPUT
      OUT1 : Bool;
      OUT2 : Bool;
      OUT3 : Bool;
   END_VAR
   VAR
      OUT11 : Bool;
      OUT12 : Bool;
      OUT21 : Bool;
      OUT22 : Bool;
      OUT31 : Bool;
      OUT32 : Bool;
      M1 : Int;
      M2 : Int;
      M3 : Int;
      M4 : Bool;
      M5 : Bool;
      M6 : Bool;
   END_VAR
   VAR_TEMP
      T1 : Bool;
      T2 : Bool;
      T3 : Bool;
      T4 : Bool;
      T5 : Bool;
      T6 : Bool;
   END_VAR
   VAR_TEMP   // added for the SCL form of the ladder/FBD networks
      _w1 : Bool;
   END_VAR
BEGIN

REGION Network 1
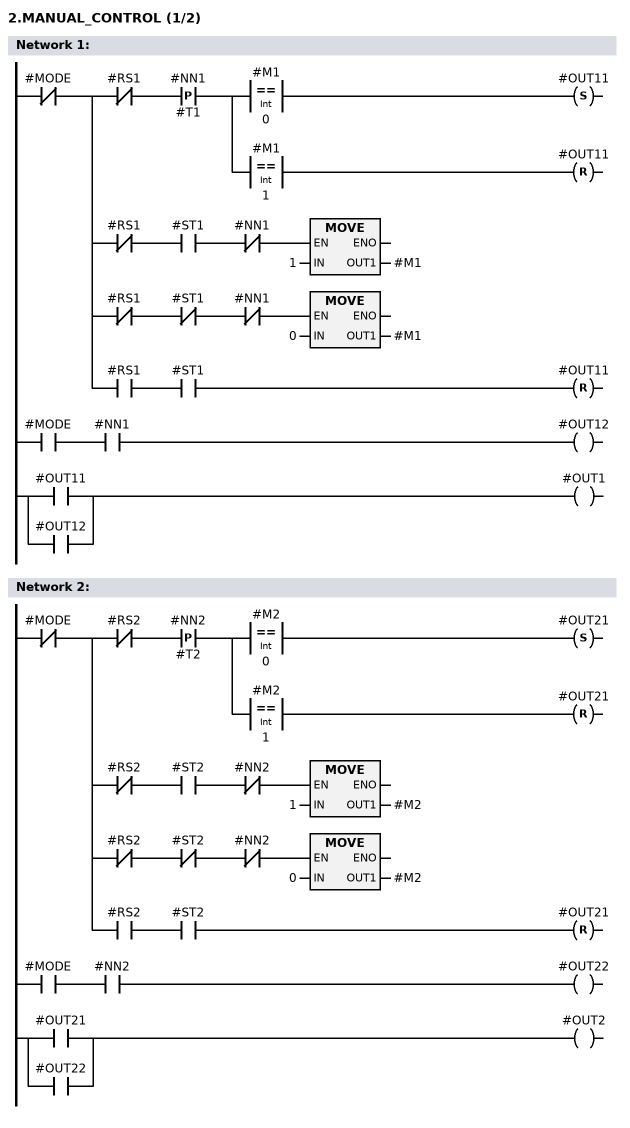
   RUNG wire#powerrail
      I_Contact( #MODE )
      wire#w1
      I_Contact( #RS1 )
      P_Contact(operand := #NN1, bit := #T1)
      wire#w2
      { S7_Templates := "SrcType := Int" } EQ_Contact(in1 := #M1, in2 := 0)
      S_Coil( #OUT11 )
   END_RUNG
   RUNG wire#w2
      { S7_Templates := "SrcType := Int" } EQ_Contact(in1 := #M1, in2 := 1)
      R_Coil( #OUT11 )
   END_RUNG
   RUNG wire#w1
      I_Contact( #RS1 )
      Contact( #ST1 )
      I_Contact( #NN1 )
      Move(in := 1, out1 => #M1)
   END_RUNG
   RUNG wire#w1
      I_Contact( #RS1 )
      I_Contact( #ST1 )
      I_Contact( #NN1 )
      Move(in := 0, out1 => #M1)
   END_RUNG
   RUNG wire#w1
      Contact( #RS1 )
      Contact( #ST1 )
      R_Coil( #OUT11 )
   END_RUNG
   RUNG wire#powerrail
      Contact( #MODE )
      Contact( #NN1 )
      Coil( #OUT12 )
   END_RUNG
   RUNG wire#powerrail
      Contact( #OUT11 )
      wire#w3
      Coil( #OUT1 )
   END_RUNG
   RUNG wire#powerrail
      Contact( #OUT12 )
   END_RUNG wire#w3
   // the same network as SCL:
   #_w1 := NOT #MODE AND NOT #RS1 AND #NN1 AND NOT #T1;   // rising edge of #NN1
   #T1 := #NN1;
   IF #_w1 AND (#M1 = 0) THEN #OUT11 := TRUE; END_IF;
   IF #_w1 AND (#M1 = 1) THEN #OUT11 := FALSE; END_IF;
   IF NOT #MODE AND NOT #RS1 AND #ST1 AND NOT #NN1 THEN #M1 := 1; END_IF;
   IF NOT #MODE AND NOT #RS1 AND NOT #ST1 AND NOT #NN1 THEN #M1 := 0; END_IF;
   IF NOT #MODE AND #RS1 AND #ST1 THEN #OUT11 := FALSE; END_IF;
   #OUT12 := #MODE AND #NN1;
   #OUT1 := #OUT11 OR #OUT12;
END_REGION

REGION Network 2
   RUNG wire#powerrail
      I_Contact( #MODE )
      wire#w1
      I_Contact( #RS2 )
      P_Contact(operand := #NN2, bit := #T2)
      wire#w2
      { S7_Templates := "SrcType := Int" } EQ_Contact(in1 := #M2, in2 := 0)
      S_Coil( #OUT21 )
   END_RUNG
   RUNG wire#w2
      { S7_Templates := "SrcType := Int" } EQ_Contact(in1 := #M2, in2 := 1)
      R_Coil( #OUT21 )
   END_RUNG
   RUNG wire#w1
      I_Contact( #RS2 )
      Contact( #ST2 )
      I_Contact( #NN2 )
      Move(in := 1, out1 => #M2)
   END_RUNG
   RUNG wire#w1
      I_Contact( #RS2 )
      I_Contact( #ST2 )
      I_Contact( #NN2 )
      Move(in := 0, out1 => #M2)
   END_RUNG
   RUNG wire#w1
      Contact( #RS2 )
      Contact( #ST2 )
      R_Coil( #OUT21 )
   END_RUNG
   RUNG wire#powerrail
      Contact( #MODE )
      Contact( #NN2 )
      Coil( #OUT22 )
   END_RUNG
   RUNG wire#powerrail
      Contact( #OUT21 )
      wire#w3
      Coil( #OUT2 )
   END_RUNG
   RUNG wire#powerrail
      Contact( #OUT22 )
   END_RUNG wire#w3
   // the same network as SCL:
   #_w1 := NOT #MODE AND NOT #RS2 AND #NN2 AND NOT #T2;   // rising edge of #NN2
   #T2 := #NN2;
   IF #_w1 AND (#M2 = 0) THEN #OUT21 := TRUE; END_IF;
   IF #_w1 AND (#M2 = 1) THEN #OUT21 := FALSE; END_IF;
   IF NOT #MODE AND NOT #RS2 AND #ST2 AND NOT #NN2 THEN #M2 := 1; END_IF;
   IF NOT #MODE AND NOT #RS2 AND NOT #ST2 AND NOT #NN2 THEN #M2 := 0; END_IF;
   IF NOT #MODE AND #RS2 AND #ST2 THEN #OUT21 := FALSE; END_IF;
   #OUT22 := #MODE AND #NN2;
   #OUT2 := #OUT21 OR #OUT22;
END_REGION

REGION Network 3
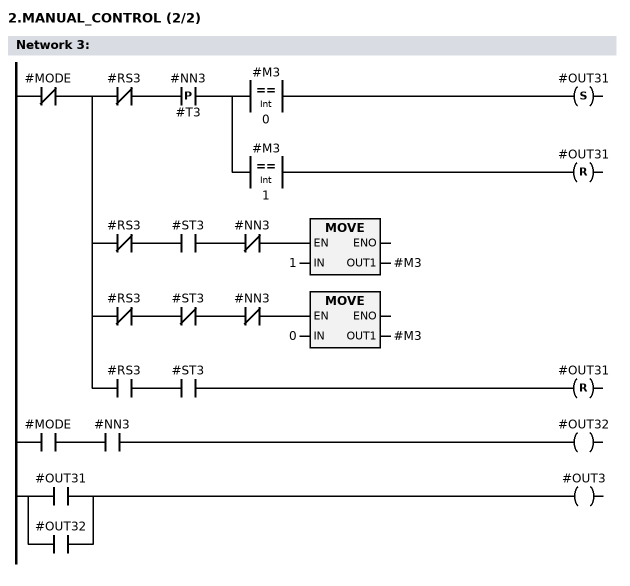
   RUNG wire#powerrail
      I_Contact( #MODE )
      wire#w1
      I_Contact( #RS3 )
      P_Contact(operand := #NN3, bit := #T3)
      wire#w2
      { S7_Templates := "SrcType := Int" } EQ_Contact(in1 := #M3, in2 := 0)
      S_Coil( #OUT31 )
   END_RUNG
   RUNG wire#w2
      { S7_Templates := "SrcType := Int" } EQ_Contact(in1 := #M3, in2 := 1)
      R_Coil( #OUT31 )
   END_RUNG
   RUNG wire#w1
      I_Contact( #RS3 )
      Contact( #ST3 )
      I_Contact( #NN3 )
      Move(in := 1, out1 => #M3)
   END_RUNG
   RUNG wire#w1
      I_Contact( #RS3 )
      I_Contact( #ST3 )
      I_Contact( #NN3 )
      Move(in := 0, out1 => #M3)
   END_RUNG
   RUNG wire#w1
      Contact( #RS3 )
      Contact( #ST3 )
      R_Coil( #OUT31 )
   END_RUNG
   RUNG wire#powerrail
      Contact( #MODE )
      Contact( #NN3 )
      Coil( #OUT32 )
   END_RUNG
   RUNG wire#powerrail
      Contact( #OUT31 )
      wire#w3
      Coil( #OUT3 )
   END_RUNG
   RUNG wire#powerrail
      Contact( #OUT32 )
   END_RUNG wire#w3
   // the same network as SCL:
   #_w1 := NOT #MODE AND NOT #RS3 AND #NN3 AND NOT #T3;   // rising edge of #NN3
   #T3 := #NN3;
   IF #_w1 AND (#M3 = 0) THEN #OUT31 := TRUE; END_IF;
   IF #_w1 AND (#M3 = 1) THEN #OUT31 := FALSE; END_IF;
   IF NOT #MODE AND NOT #RS3 AND #ST3 AND NOT #NN3 THEN #M3 := 1; END_IF;
   IF NOT #MODE AND NOT #RS3 AND NOT #ST3 AND NOT #NN3 THEN #M3 := 0; END_IF;
   IF NOT #MODE AND #RS3 AND #ST3 THEN #OUT31 := FALSE; END_IF;
   #OUT32 := #MODE AND #NN3;
   #OUT3 := #OUT31 OR #OUT32;
END_REGION
END_FUNCTION_BLOCK

FUNCTION_BLOCK "1.ANALOG_INPUT"   // FB1, LAD
{ S7_Optimized_Access := 'TRUE' }
VERSION : 0.1
// stored: AutoNumber false, CodeModifiedDate 2025-09-22T19:33:21.555545Z, CompileDate 2026-01-15T16:25:51.8952099Z, CreationDate 2026-01-15T16:22:49.8270549Z, DownloadWithoutReinit false, HandleErrorsWithinBlock false, InterfaceModifiedDate 2025-09-22T19:30:11.8403437Z, IsConsistent true, IsIECCheckEnabled false, IsKnowHowProtected false, IsRetainMemResEnabled false, IsWriteProtected false, LibraryConformanceStatus The object is library-conformant., MemoryReserve 100, ModifiedDate 2026-01-11T09:46:51.3925903Z, ParameterModified 2025-08-30T17:31:01.4104373Z, PLCSimAdvancedSupport false, SetENOAutomatically False, StructureModified 2025-09-22T19:30:11.8403437Z, UDAEnableTagReadback false
   VAR_INPUT
      AI : Int;
      A_MODE : Real;
      ZERO : Real;
      SPAN : Real;
      BT_ZERO : Bool;
      BT_SPAN : Bool;
      B_MANUAL : Real;
      HMI_Manual_Trigger : Bool;
   END_VAR
   VAR_OUTPUT
      W_OUT : Real;
      X_OUT : Real;
   END_VAR
   VAR RETAIN
      T_AI { ExternalAccessible := 'False'; ExternalVisible := 'False'; ExternalWritable := 'False'} : Real;
      T_AN { ExternalAccessible := 'False'; ExternalVisible := 'False'; ExternalWritable := 'False'} : Real;
      T_ZERO { ExternalAccessible := 'False'; ExternalVisible := 'False'; ExternalWritable := 'False'} : Real;
      AN_ZERO { ExternalAccessible := 'False'; ExternalVisible := 'False'; ExternalWritable := 'False'} : Real;
      T_SPAN { ExternalAccessible := 'False'; ExternalVisible := 'False'; ExternalWritable := 'False'} : Real;
      AN_SPAN { ExternalAccessible := 'False'; ExternalVisible := 'False'; ExternalWritable := 'False'} : Real;
   END_VAR
   VAR
      B_MANUAL_SAVED : Real;
      B_HAS_CHANGED : Bool;
   END_VAR
   VAR RETAIN
      IS_MANUAL_MODE : Bool;
   END_VAR
   VAR
      BT_ZERO_Raising : Bool;
      BT_SPAN_Riasing : Bool;
      MANUAL_Raissing : Bool;
      Bit_Reset_Man_Mode : Bool;
   END_VAR
   VAR_TEMP
      AI_MIN : Int;
      AI_MAX : Int;
      AN_MIN : Real;
      AN_MAX : Real;
      GT_INTEGER : DInt;
      TEMP_RESULT_DINT : DInt;
      W_OUT_MANUAL : Real;
      W_OUT_AUTO : Real;
   END_VAR
   VAR_TEMP   // added for the SCL form of the ladder/FBD networks
      _w1 : Bool;
   END_VAR
BEGIN

REGION Network 1: ANALOG MODE
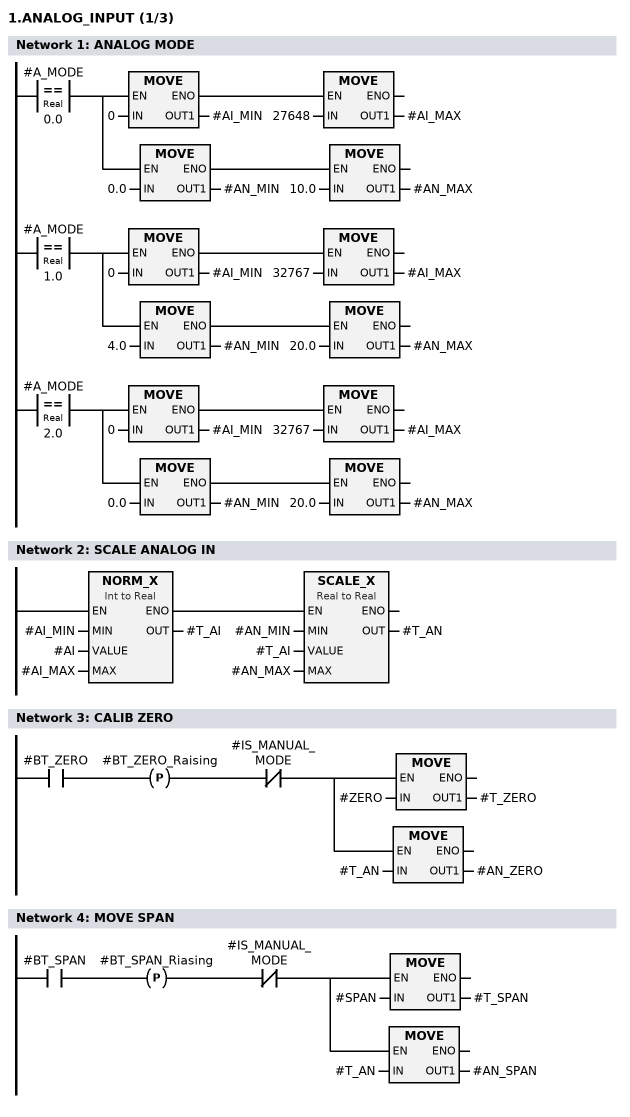
   RUNG wire#powerrail
      { S7_Templates := "SrcType := Real" } EQ_Contact(in1 := #A_MODE, in2 := 0.0)
      wire#w1
      Move(in := 0, out1 => #AI_MIN)
      Move(in := 27648, out1 => #AI_MAX)
   END_RUNG
   RUNG wire#w1
      Move(in := 0.0, out1 => #AN_MIN)
      Move(in := 10.0, out1 => #AN_MAX)
   END_RUNG
   RUNG wire#powerrail
      { S7_Templates := "SrcType := Real" } EQ_Contact(in1 := #A_MODE, in2 := 1.0)
      wire#w2
      Move(in := 0, out1 => #AI_MIN)
      Move(in := 32767, out1 => #AI_MAX)
   END_RUNG
   RUNG wire#w2
      Move(in := 4.0, out1 => #AN_MIN)
      Move(in := 20.0, out1 => #AN_MAX)
   END_RUNG
   RUNG wire#powerrail
      { S7_Templates := "SrcType := Real" } EQ_Contact(in1 := #A_MODE, in2 := 2.0)
      wire#w3
      Move(in := 0, out1 => #AI_MIN)
      Move(in := 32767, out1 => #AI_MAX)
   END_RUNG
   RUNG wire#w3
      Move(in := 0.0, out1 => #AN_MIN)
      Move(in := 20.0, out1 => #AN_MAX)
   END_RUNG
   // the same network as SCL:
   IF #A_MODE = 0.0 THEN
       #AI_MIN := 0;
       #AI_MAX := 27648;
       #AN_MIN := 0.0;
       #AN_MAX := 10.0;
   END_IF;
   IF #A_MODE = 1.0 THEN
       #AI_MIN := 0;
       #AI_MAX := 32767;
       #AN_MIN := 4.0;
       #AN_MAX := 20.0;
   END_IF;
   IF #A_MODE = 2.0 THEN
       #AI_MIN := 0;
       #AI_MAX := 32767;
       #AN_MIN := 0.0;
       #AN_MAX := 20.0;
   END_IF;
END_REGION

REGION Network 2: SCALE ANALOG IN
   RUNG wire#powerrail
      { S7_Templates := "[SrcType := Int, DestType := Real]" } Normalize(min := #AI_MIN, value := #AI, max := #AI_MAX, out => #T_AI)
      { S7_Templates := "[SrcType := Real, DestType := Real]" } Scale(min := #AN_MIN, value := #T_AI, max := #AN_MAX, out => #T_AN)
   END_RUNG
   // the same network as SCL:
   #T_AI := NORM_X(MIN := #AI_MIN, VALUE := #AI, MAX := #AI_MAX);
   #T_AN := SCALE_X(MIN := #AN_MIN, VALUE := #T_AI, MAX := #AN_MAX);
END_REGION

REGION Network 3: CALIB ZERO
   RUNG wire#powerrail
      Contact( #BT_ZERO )
      P_Trig( #BT_ZERO_Raising )
      I_Contact( #IS_MANUAL_MODE )
      wire#w1
      Move(in := #ZERO, out1 => #T_ZERO)
   END_RUNG
   RUNG wire#w1
      Move(in := #T_AN, out1 => #AN_ZERO)
   END_RUNG
   // the same network as SCL:
   #_w1 := #BT_ZERO AND NOT #BT_ZERO_Raising;   // rising edge
   #BT_ZERO_Raising := #BT_ZERO;
   IF #_w1 AND NOT #IS_MANUAL_MODE THEN
       #T_ZERO := #ZERO;
       #AN_ZERO := #T_AN;
   END_IF;
END_REGION

REGION Network 4: MOVE SPAN
   RUNG wire#powerrail
      Contact( #BT_SPAN )
      P_Trig( #BT_SPAN_Riasing )
      I_Contact( #IS_MANUAL_MODE )
      wire#w1
      Move(in := #SPAN, out1 => #T_SPAN)
   END_RUNG
   RUNG wire#w1
      Move(in := #T_AN, out1 => #AN_SPAN)
   END_RUNG
   // the same network as SCL:
   #_w1 := #BT_SPAN AND NOT #BT_SPAN_Riasing;   // rising edge
   #BT_SPAN_Riasing := #BT_SPAN;
   IF #_w1 AND NOT #IS_MANUAL_MODE THEN
       #T_SPAN := #SPAN;
       #AN_SPAN := #T_AN;
   END_IF;
END_REGION

REGION Network 5: WEIGHT OUT
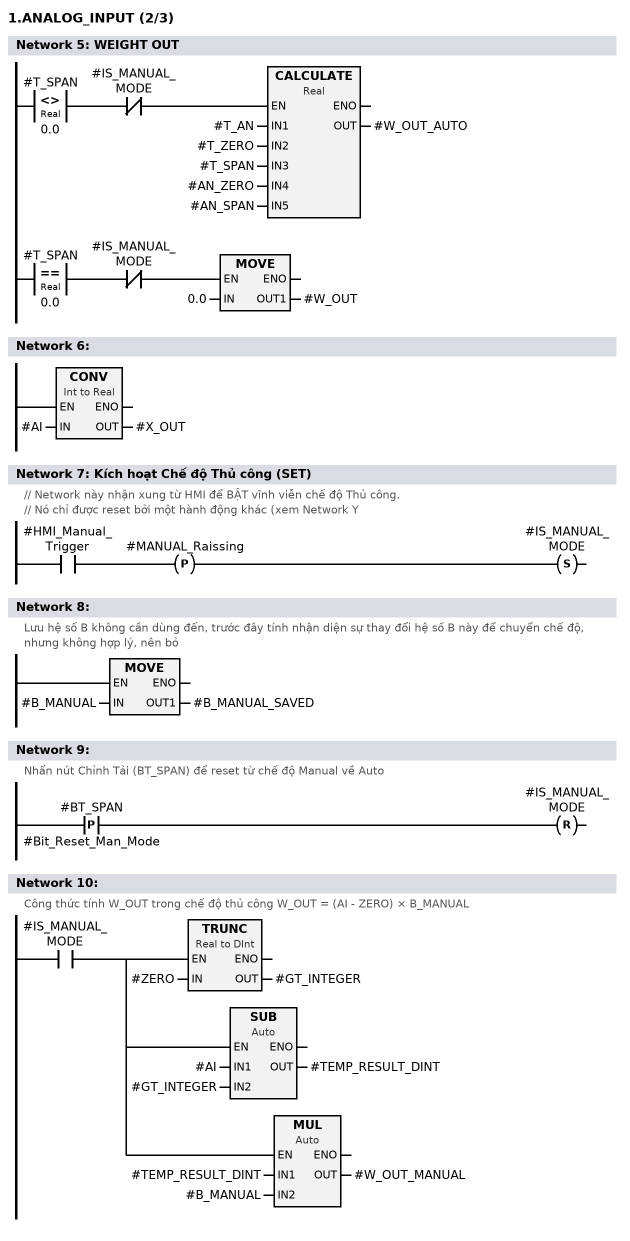
   RUNG wire#powerrail
      { S7_Templates := "SrcType := Real" } NE_Contact(in1 := #T_SPAN, in2 := 0.0)
      I_Contact( #IS_MANUAL_MODE )
      { S7_Templates := "SrcType := Real"; S7_Expression := "(IN1-IN4)/((IN5-IN4)/(IN3-IN2))" } Calculate(in1 := #T_AN, in2 := #T_ZERO, in3 := #T_SPAN, in4 := #AN_ZERO, in5 := #AN_SPAN, out => #W_OUT_AUTO)
   END_RUNG
   RUNG wire#powerrail
      { S7_Templates := "SrcType := Real" } EQ_Contact(in1 := #T_SPAN, in2 := 0.0)
      I_Contact( #IS_MANUAL_MODE )
      Move(in := 0.0, out1 => #W_OUT)
   END_RUNG
   // the same network as SCL:
   IF (#T_SPAN <> 0.0) AND NOT #IS_MANUAL_MODE THEN
       #W_OUT_AUTO := (#T_AN-#AN_ZERO)/((#AN_SPAN-#AN_ZERO)/(#T_SPAN-#T_ZERO));
   END_IF;
   IF (#T_SPAN = 0.0) AND NOT #IS_MANUAL_MODE THEN #W_OUT := 0.0; END_IF;
END_REGION

REGION Network 6
   RUNG wire#powerrail
      { S7_Templates := "[SrcType := Int, DestType := Real]" } Convert(in := #AI, out => #X_OUT)
   END_RUNG
   // the same network as SCL:
   #X_OUT := INT_TO_REAL(#AI);
END_REGION

REGION Network 7: Kích hoạt Chế độ Thủ công (SET)
   // // Network này nhận xung từ HMI để BẬT vĩnh viễn chế độ Thủ công.
   // // Nó chỉ được reset bởi một hành động khác (xem Network Y
   RUNG wire#powerrail
      Contact( #HMI_Manual_Trigger )
      P_Trig( #MANUAL_Raissing )
      S_Coil( #IS_MANUAL_MODE )
   END_RUNG
   // the same network as SCL:
   #_w1 := #HMI_Manual_Trigger AND NOT #MANUAL_Raissing;   // rising edge
   #MANUAL_Raissing := #HMI_Manual_Trigger;
   IF #_w1 THEN #IS_MANUAL_MODE := TRUE; END_IF;
END_REGION

REGION Network 8
   // Lưu hệ số B không cần dùng đến, trước đây tính nhận diện sự thay đổi hệ số B này để chuyển chế độ, nhưng không hợp lý, nên bỏ
   RUNG wire#powerrail
      Move(in := #B_MANUAL, out1 => #B_MANUAL_SAVED)
   END_RUNG
   // the same network as SCL:
   #B_MANUAL_SAVED := #B_MANUAL;
END_REGION

REGION Network 9
   // Nhấn nút Chỉnh Tải (BT_SPAN) để reset từ chế độ Manual về Auto
   RUNG wire#powerrail
      P_Contact(operand := #BT_SPAN, bit := #Bit_Reset_Man_Mode)
      R_Coil( #IS_MANUAL_MODE )
   END_RUNG
   // the same network as SCL:
   #_w1 := #BT_SPAN AND NOT #Bit_Reset_Man_Mode;   // rising edge of #BT_SPAN
   #Bit_Reset_Man_Mode := #BT_SPAN;
   IF #_w1 THEN #IS_MANUAL_MODE := FALSE; END_IF;
END_REGION

REGION Network 10
   // Công thức tính W_OUT trong chế độ thủ công W_OUT = (AI - ZERO) × B_MANUAL
   RUNG wire#powerrail
      Contact( #IS_MANUAL_MODE )
      wire#w1
      { S7_Templates := "[SrcType := Real, DestType := DInt]" } Trunc(in := #ZERO, out => #GT_INTEGER)
   END_RUNG
   RUNG wire#w1
      Sub(in1 := #AI, in2 := #GT_INTEGER, out => #TEMP_RESULT_DINT)
   END_RUNG
   RUNG wire#w1
      Mul(in1 := #TEMP_RESULT_DINT, in2 := #B_MANUAL, out => #W_OUT_MANUAL)
   END_RUNG
   // the same network as SCL:
   IF #IS_MANUAL_MODE THEN
       #GT_INTEGER := TRUNC(#ZERO);
       #TEMP_RESULT_DINT := #AI - #GT_INTEGER;
       #W_OUT_MANUAL := #TEMP_RESULT_DINT * #B_MANUAL;
   END_IF;
END_REGION

REGION Network 11
   // Lệnh chọn đầu ra W_OUT theo 2 chế độ Auto và Manual
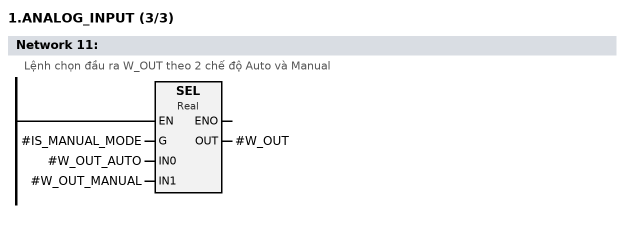
   RUNG wire#powerrail
      { S7_Templates := "value_type := Real" } SEL(g := #IS_MANUAL_MODE, in0 := #W_OUT_AUTO, in1 := #W_OUT_MANUAL, out => #W_OUT)
   END_RUNG
   // the same network as SCL:
   #W_OUT := SEL(G := #IS_MANUAL_MODE, IN0 := #W_OUT_AUTO, IN1 := #W_OUT_MANUAL);
END_REGION
END_FUNCTION_BLOCK

FUNCTION "1. CONVER TC" : Void   // FC1, LAD
{ S7_Optimized_Access := 'TRUE' }
VERSION : 0.1
// stored: AutoNumber true, CodeModifiedDate 2025-08-27T17:05:49.4204143Z, CompileDate 2026-01-15T16:25:52.7071747Z, CreationDate 2026-01-15T16:22:49.8270549Z, HandleErrorsWithinBlock false, InterfaceModifiedDate 2024-10-18T04:03:55.072308Z, IsConsistent true, IsIECCheckEnabled false, IsKnowHowProtected false, IsWriteProtected false, LibraryConformanceStatus The object is library-conformant., ModifiedDate 2025-08-27T17:05:49.4204143Z, ParameterModified 2024-10-18T04:03:55.072308Z, PLCSimAdvancedSupport false, SetENOAutomatically False, StructureModified 2024-10-18T04:03:55.072308Z, UDAEnableTagReadback false
   VAR_INPUT
      AI : Int;
      HS : Real;
   END_VAR
   VAR_OUTPUT
      TEMP_OUT : Real;
      XUNG_OUT : Real;
   END_VAR
   VAR_TEMP
      AI_REAL : Real;
   END_VAR
BEGIN

REGION Network 1
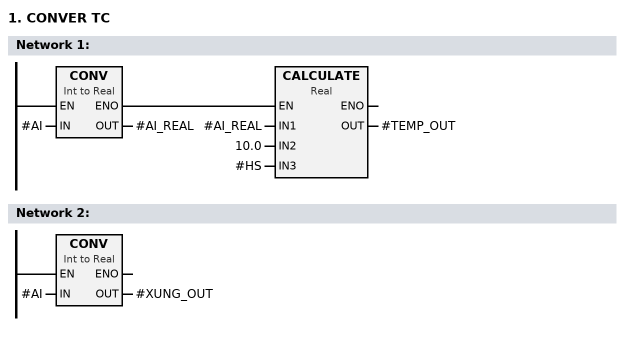
   RUNG wire#powerrail
      { S7_Templates := "[SrcType := Int, DestType := Real]" } Convert(in := #AI, out => #AI_REAL)
      { S7_Templates := "SrcType := Real"; S7_Expression := "(IN1/IN2)*IN3" } Calculate(in1 := #AI_REAL, in2 := 10.0, in3 := #HS, out => #TEMP_OUT)
   END_RUNG
   // the same network as SCL:
   #AI_REAL := INT_TO_REAL(#AI);
   #TEMP_OUT := (#AI_REAL/10.0)*#HS;
END_REGION

REGION Network 2
   RUNG wire#powerrail
      { S7_Templates := "[SrcType := Int, DestType := Real]" } Convert(in := #AI, out => #XUNG_OUT)
   END_RUNG
   // the same network as SCL:
   #XUNG_OUT := INT_TO_REAL(#AI);
END_REGION
END_FUNCTION

FUNCTION_BLOCK "4.SIMULATION_DATA"   // FB4, LAD
{ S7_Optimized_Access := 'TRUE' }
VERSION : 0.1
// stored: AutoNumber false, CodeModifiedDate 2025-08-27T17:12:03.7644125Z, CompileDate 2026-01-15T16:25:51.5973447Z, CreationDate 2026-01-15T16:22:49.8270549Z, DownloadWithoutReinit false, HandleErrorsWithinBlock false, InterfaceModifiedDate 2023-11-28T22:28:44.2264332Z, IsConsistent true, IsIECCheckEnabled false, IsKnowHowProtected false, IsRetainMemResEnabled false, IsWriteProtected false, LibraryConformanceStatus The object is library-conformant., MemoryReserve 100, ModifiedDate 2025-08-27T17:12:03.7644125Z, ParameterModified 2023-11-28T22:28:44.2264332Z, PLCSimAdvancedSupport false, SetENOAutomatically False, StructureModified 2023-11-28T22:28:44.2264332Z, UDAEnableTagReadback false
   VAR_INPUT
      RE_SET : Bool;
      XUNG_CLOCK : Bool;
      CAN_1 : Bool;
      CAN_2 : Bool;
      CAN_3 : Bool;
      CAN_4 : Bool;
      CAN_5 : Bool;
      CAN_6 : Bool;
      CAN_7 : Bool;
      CAN_8 : Bool;
      CAN_9 : Bool;
      CAN_10 : Bool;
      CAN_11 : Bool;
      CAN_12 : Bool;
      XA_1 : Bool;
      XA_2 : Bool;
      XA_3 : Bool;
      XA_4 : Bool;
      XA_5 : Bool;
      XA_6 : Bool;
      XA_7 : Bool;
      XA_8 : Bool;
      XA_9 : Bool;
      XA_10 : Bool;
      XA_11 : Bool;
      XA_12 : Bool;
      HS_NAP_AGG1 : Real;
      HS_NAP_AGG2 : Real;
      HS_NAP_AGG3 : Real;
      HS_NAP_AGG4 : Real;
      HS_NAP_AGG5 : Real;
      HS_NAP_AGG6 : Real;
      HS_NAP_CEM1 : Real;
      HS_NAP_CEM2 : Real;
      HS_NAP_WAT1 : Real;
      HS_NAP_WAT2 : Real;
      HS_NAP_ADD1 : Real;
      HS_NAP_ADD2 : Real;
      HS_XA_AGG1 : Real;
      HS_XA_AGG2 : Real;
      HS_XA_AGG3 : Real;
      HS_XA_AGG4 : Real;
      HS_XA_AGG5 : Real;
      HS_XA_AGG6 : Real;
      HS_XA_CEM1 : Real;
      HS_XA_CEM2 : Real;
      HS_XA_WAT1 : Real;
      HS_XA_WAT2 : Real;
      HS_XA_ADD1 : Real;
      HS_XA_ADD2 : Real;
   END_VAR
   VAR_OUTPUT
      AGG1 : Real;
      AGG2 : Real;
      AGG3 : Real;
      AGG4 : Real;
      AGG5 : Real;
      AGG6 : Real;
      CEM1 : Real;
      CEM2 : Real;
      WAT1 : Real;
      WAT2 : Real;
      WADD1 : Real;
      WADD2 : Real;
   END_VAR
   VAR
      A1 : Bool;
      B1 : Bool;
      A2 : Bool;
      B2 : Bool;
      A3 : Bool;
      B3 : Bool;
      A4 : Bool;
      B4 : Bool;
      A5 : Bool;
      B5 : Bool;
      A6 : Bool;
      B6 : Bool;
      A7 : Bool;
      B7 : Bool;
      A8 : Bool;
      B8 : Bool;
      A9 : Bool;
      B9 : Bool;
      A10 : Bool;
      B10 : Bool;
      A11 : Bool;
      B11 : Bool;
      A12 : Bool;
      B12 : Bool;
   END_VAR
   VAR_TEMP   // added for the SCL form of the ladder/FBD networks
      _w1 : Bool;
      _w2 : Bool;
   END_VAR
BEGIN

REGION Network 1: RESET
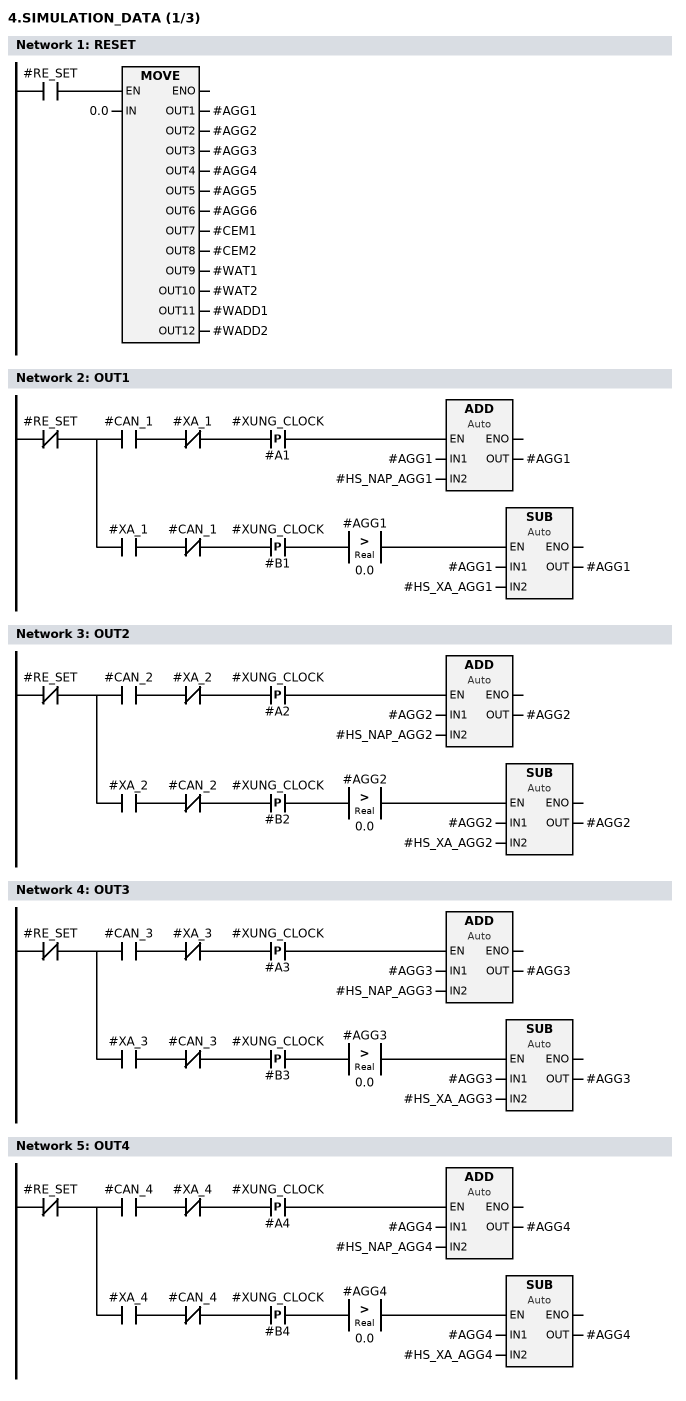
   RUNG wire#powerrail
      Contact( #RE_SET )
      Move(in := 0.0, out1 => #AGG1, out2 => #AGG2, out3 => #AGG3, out4 => #AGG4, out5 => #AGG5, out6 => #AGG6, out7 => #CEM1, out8 => #CEM2, out9 => #WAT1, out10 => #WAT2, out11 => #WADD1, out12 => #WADD2)
   END_RUNG
   // the same network as SCL:
   IF #RE_SET THEN
       #AGG1 := 0.0;
       #AGG2 := 0.0;
       #AGG3 := 0.0;
       #AGG4 := 0.0;
       #AGG5 := 0.0;
       #AGG6 := 0.0;
       #CEM1 := 0.0;
       #CEM2 := 0.0;
       #WAT1 := 0.0;
       #WAT2 := 0.0;
       #WADD1 := 0.0;
       #WADD2 := 0.0;
   END_IF;
END_REGION

REGION Network 2: OUT1
   RUNG wire#powerrail
      I_Contact( #RE_SET )
      wire#w1
      Contact( #CAN_1 )
      I_Contact( #XA_1 )
      P_Contact(operand := #XUNG_CLOCK, bit := #A1)
      Add(in1 := #AGG1, in2 := #HS_NAP_AGG1, out => #AGG1)
   END_RUNG
   RUNG wire#w1
      Contact( #XA_1 )
      I_Contact( #CAN_1 )
      P_Contact(operand := #XUNG_CLOCK, bit := #B1)
      { S7_Templates := "SrcType := Real" } GT_Contact(in1 := #AGG1, in2 := 0.0)
      Sub(in1 := #AGG1, in2 := #HS_XA_AGG1, out => #AGG1)
   END_RUNG
   // the same network as SCL:
   #_w1 := NOT #RE_SET AND #CAN_1 AND NOT #XA_1 AND #XUNG_CLOCK AND NOT #A1;   // rising edge of #XUNG_CLOCK
   #A1 := #XUNG_CLOCK;
   IF #_w1 THEN #AGG1 := #AGG1 + #HS_NAP_AGG1; END_IF;
   #_w2 := NOT #RE_SET AND #XA_1 AND NOT #CAN_1 AND #XUNG_CLOCK AND NOT #B1;   // rising edge of #XUNG_CLOCK
   #B1 := #XUNG_CLOCK;
   IF #_w2 AND (#AGG1 > 0.0) THEN #AGG1 := #AGG1 - #HS_XA_AGG1; END_IF;
END_REGION

REGION Network 3: OUT2
   RUNG wire#powerrail
      I_Contact( #RE_SET )
      wire#w1
      Contact( #CAN_2 )
      I_Contact( #XA_2 )
      P_Contact(operand := #XUNG_CLOCK, bit := #A2)
      Add(in1 := #AGG2, in2 := #HS_NAP_AGG2, out => #AGG2)
   END_RUNG
   RUNG wire#w1
      Contact( #XA_2 )
      I_Contact( #CAN_2 )
      P_Contact(operand := #XUNG_CLOCK, bit := #B2)
      { S7_Templates := "SrcType := Real" } GT_Contact(in1 := #AGG2, in2 := 0.0)
      Sub(in1 := #AGG2, in2 := #HS_XA_AGG2, out => #AGG2)
   END_RUNG
   // the same network as SCL:
   #_w1 := NOT #RE_SET AND #CAN_2 AND NOT #XA_2 AND #XUNG_CLOCK AND NOT #A2;   // rising edge of #XUNG_CLOCK
   #A2 := #XUNG_CLOCK;
   IF #_w1 THEN #AGG2 := #AGG2 + #HS_NAP_AGG2; END_IF;
   #_w2 := NOT #RE_SET AND #XA_2 AND NOT #CAN_2 AND #XUNG_CLOCK AND NOT #B2;   // rising edge of #XUNG_CLOCK
   #B2 := #XUNG_CLOCK;
   IF #_w2 AND (#AGG2 > 0.0) THEN #AGG2 := #AGG2 - #HS_XA_AGG2; END_IF;
END_REGION

REGION Network 4: OUT3
   RUNG wire#powerrail
      I_Contact( #RE_SET )
      wire#w1
      Contact( #CAN_3 )
      I_Contact( #XA_3 )
      P_Contact(operand := #XUNG_CLOCK, bit := #A3)
      Add(in1 := #AGG3, in2 := #HS_NAP_AGG3, out => #AGG3)
   END_RUNG
   RUNG wire#w1
      Contact( #XA_3 )
      I_Contact( #CAN_3 )
      P_Contact(operand := #XUNG_CLOCK, bit := #B3)
      { S7_Templates := "SrcType := Real" } GT_Contact(in1 := #AGG3, in2 := 0.0)
      Sub(in1 := #AGG3, in2 := #HS_XA_AGG3, out => #AGG3)
   END_RUNG
   // the same network as SCL:
   #_w1 := NOT #RE_SET AND #CAN_3 AND NOT #XA_3 AND #XUNG_CLOCK AND NOT #A3;   // rising edge of #XUNG_CLOCK
   #A3 := #XUNG_CLOCK;
   IF #_w1 THEN #AGG3 := #AGG3 + #HS_NAP_AGG3; END_IF;
   #_w2 := NOT #RE_SET AND #XA_3 AND NOT #CAN_3 AND #XUNG_CLOCK AND NOT #B3;   // rising edge of #XUNG_CLOCK
   #B3 := #XUNG_CLOCK;
   IF #_w2 AND (#AGG3 > 0.0) THEN #AGG3 := #AGG3 - #HS_XA_AGG3; END_IF;
END_REGION

REGION Network 5: OUT4
   RUNG wire#powerrail
      I_Contact( #RE_SET )
      wire#w1
      Contact( #CAN_4 )
      I_Contact( #XA_4 )
      P_Contact(operand := #XUNG_CLOCK, bit := #A4)
      Add(in1 := #AGG4, in2 := #HS_NAP_AGG4, out => #AGG4)
   END_RUNG
   RUNG wire#w1
      Contact( #XA_4 )
      I_Contact( #CAN_4 )
      P_Contact(operand := #XUNG_CLOCK, bit := #B4)
      { S7_Templates := "SrcType := Real" } GT_Contact(in1 := #AGG4, in2 := 0.0)
      Sub(in1 := #AGG4, in2 := #HS_XA_AGG4, out => #AGG4)
   END_RUNG
   // the same network as SCL:
   #_w1 := NOT #RE_SET AND #CAN_4 AND NOT #XA_4 AND #XUNG_CLOCK AND NOT #A4;   // rising edge of #XUNG_CLOCK
   #A4 := #XUNG_CLOCK;
   IF #_w1 THEN #AGG4 := #AGG4 + #HS_NAP_AGG4; END_IF;
   #_w2 := NOT #RE_SET AND #XA_4 AND NOT #CAN_4 AND #XUNG_CLOCK AND NOT #B4;   // rising edge of #XUNG_CLOCK
   #B4 := #XUNG_CLOCK;
   IF #_w2 AND (#AGG4 > 0.0) THEN #AGG4 := #AGG4 - #HS_XA_AGG4; END_IF;
END_REGION

REGION Network 6: OUT5
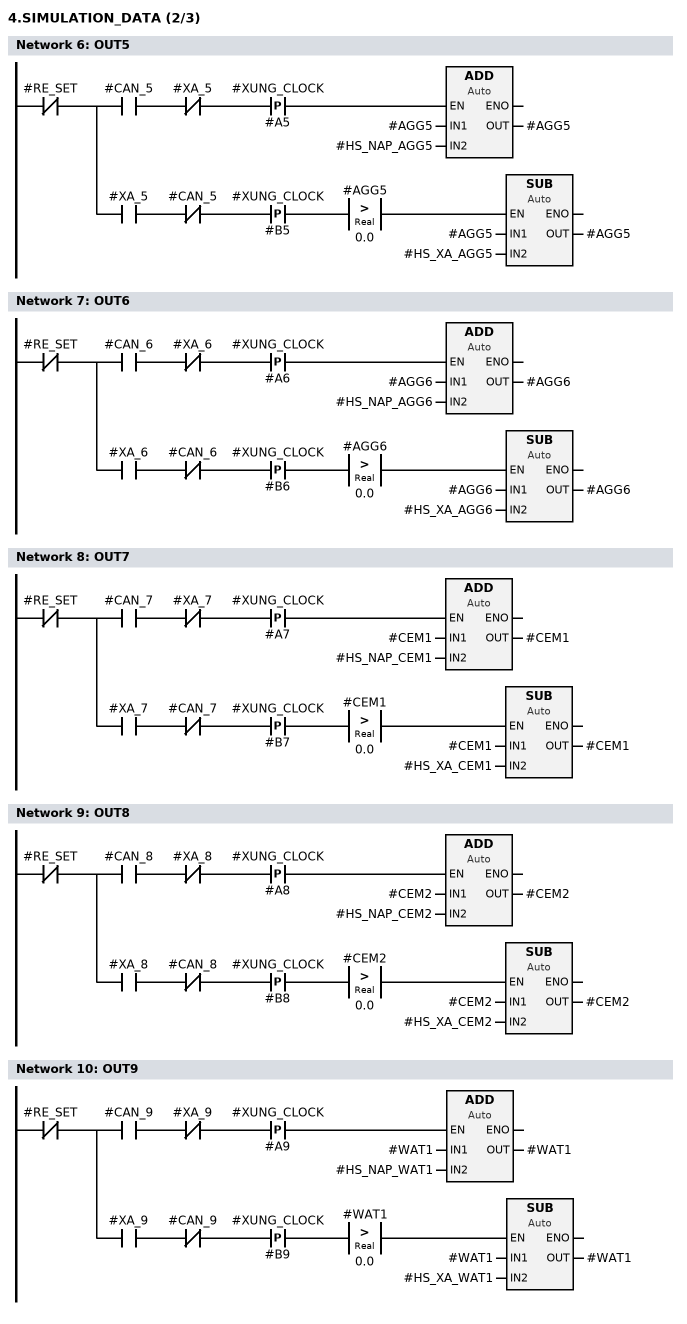
   RUNG wire#powerrail
      I_Contact( #RE_SET )
      wire#w1
      Contact( #CAN_5 )
      I_Contact( #XA_5 )
      P_Contact(operand := #XUNG_CLOCK, bit := #A5)
      Add(in1 := #AGG5, in2 := #HS_NAP_AGG5, out => #AGG5)
   END_RUNG
   RUNG wire#w1
      Contact( #XA_5 )
      I_Contact( #CAN_5 )
      P_Contact(operand := #XUNG_CLOCK, bit := #B5)
      { S7_Templates := "SrcType := Real" } GT_Contact(in1 := #AGG5, in2 := 0.0)
      Sub(in1 := #AGG5, in2 := #HS_XA_AGG5, out => #AGG5)
   END_RUNG
   // the same network as SCL:
   #_w1 := NOT #RE_SET AND #CAN_5 AND NOT #XA_5 AND #XUNG_CLOCK AND NOT #A5;   // rising edge of #XUNG_CLOCK
   #A5 := #XUNG_CLOCK;
   IF #_w1 THEN #AGG5 := #AGG5 + #HS_NAP_AGG5; END_IF;
   #_w2 := NOT #RE_SET AND #XA_5 AND NOT #CAN_5 AND #XUNG_CLOCK AND NOT #B5;   // rising edge of #XUNG_CLOCK
   #B5 := #XUNG_CLOCK;
   IF #_w2 AND (#AGG5 > 0.0) THEN #AGG5 := #AGG5 - #HS_XA_AGG5; END_IF;
END_REGION

REGION Network 7: OUT6
   RUNG wire#powerrail
      I_Contact( #RE_SET )
      wire#w1
      Contact( #CAN_6 )
      I_Contact( #XA_6 )
      P_Contact(operand := #XUNG_CLOCK, bit := #A6)
      Add(in1 := #AGG6, in2 := #HS_NAP_AGG6, out => #AGG6)
   END_RUNG
   RUNG wire#w1
      Contact( #XA_6 )
      I_Contact( #CAN_6 )
      P_Contact(operand := #XUNG_CLOCK, bit := #B6)
      { S7_Templates := "SrcType := Real" } GT_Contact(in1 := #AGG6, in2 := 0.0)
      Sub(in1 := #AGG6, in2 := #HS_XA_AGG6, out => #AGG6)
   END_RUNG
   // the same network as SCL:
   #_w1 := NOT #RE_SET AND #CAN_6 AND NOT #XA_6 AND #XUNG_CLOCK AND NOT #A6;   // rising edge of #XUNG_CLOCK
   #A6 := #XUNG_CLOCK;
   IF #_w1 THEN #AGG6 := #AGG6 + #HS_NAP_AGG6; END_IF;
   #_w2 := NOT #RE_SET AND #XA_6 AND NOT #CAN_6 AND #XUNG_CLOCK AND NOT #B6;   // rising edge of #XUNG_CLOCK
   #B6 := #XUNG_CLOCK;
   IF #_w2 AND (#AGG6 > 0.0) THEN #AGG6 := #AGG6 - #HS_XA_AGG6; END_IF;
END_REGION

REGION Network 8: OUT7
   RUNG wire#powerrail
      I_Contact( #RE_SET )
      wire#w1
      Contact( #CAN_7 )
      I_Contact( #XA_7 )
      P_Contact(operand := #XUNG_CLOCK, bit := #A7)
      Add(in1 := #CEM1, in2 := #HS_NAP_CEM1, out => #CEM1)
   END_RUNG
   RUNG wire#w1
      Contact( #XA_7 )
      I_Contact( #CAN_7 )
      P_Contact(operand := #XUNG_CLOCK, bit := #B7)
      { S7_Templates := "SrcType := Real" } GT_Contact(in1 := #CEM1, in2 := 0.0)
      Sub(in1 := #CEM1, in2 := #HS_XA_CEM1, out => #CEM1)
   END_RUNG
   // the same network as SCL:
   #_w1 := NOT #RE_SET AND #CAN_7 AND NOT #XA_7 AND #XUNG_CLOCK AND NOT #A7;   // rising edge of #XUNG_CLOCK
   #A7 := #XUNG_CLOCK;
   IF #_w1 THEN #CEM1 := #CEM1 + #HS_NAP_CEM1; END_IF;
   #_w2 := NOT #RE_SET AND #XA_7 AND NOT #CAN_7 AND #XUNG_CLOCK AND NOT #B7;   // rising edge of #XUNG_CLOCK
   #B7 := #XUNG_CLOCK;
   IF #_w2 AND (#CEM1 > 0.0) THEN #CEM1 := #CEM1 - #HS_XA_CEM1; END_IF;
END_REGION

REGION Network 9: OUT8
   RUNG wire#powerrail
      I_Contact( #RE_SET )
      wire#w1
      Contact( #CAN_8 )
      I_Contact( #XA_8 )
      P_Contact(operand := #XUNG_CLOCK, bit := #A8)
      Add(in1 := #CEM2, in2 := #HS_NAP_CEM2, out => #CEM2)
   END_RUNG
   RUNG wire#w1
      Contact( #XA_8 )
      I_Contact( #CAN_8 )
      P_Contact(operand := #XUNG_CLOCK, bit := #B8)
      { S7_Templates := "SrcType := Real" } GT_Contact(in1 := #CEM2, in2 := 0.0)
      Sub(in1 := #CEM2, in2 := #HS_XA_CEM2, out => #CEM2)
   END_RUNG
   // the same network as SCL:
   #_w1 := NOT #RE_SET AND #CAN_8 AND NOT #XA_8 AND #XUNG_CLOCK AND NOT #A8;   // rising edge of #XUNG_CLOCK
   #A8 := #XUNG_CLOCK;
   IF #_w1 THEN #CEM2 := #CEM2 + #HS_NAP_CEM2; END_IF;
   #_w2 := NOT #RE_SET AND #XA_8 AND NOT #CAN_8 AND #XUNG_CLOCK AND NOT #B8;   // rising edge of #XUNG_CLOCK
   #B8 := #XUNG_CLOCK;
   IF #_w2 AND (#CEM2 > 0.0) THEN #CEM2 := #CEM2 - #HS_XA_CEM2; END_IF;
END_REGION

REGION Network 10: OUT9
   RUNG wire#powerrail
      I_Contact( #RE_SET )
      wire#w1
      Contact( #CAN_9 )
      I_Contact( #XA_9 )
      P_Contact(operand := #XUNG_CLOCK, bit := #A9)
      Add(in1 := #WAT1, in2 := #HS_NAP_WAT1, out => #WAT1)
   END_RUNG
   RUNG wire#w1
      Contact( #XA_9 )
      I_Contact( #CAN_9 )
      P_Contact(operand := #XUNG_CLOCK, bit := #B9)
      { S7_Templates := "SrcType := Real" } GT_Contact(in1 := #WAT1, in2 := 0.0)
      Sub(in1 := #WAT1, in2 := #HS_XA_WAT1, out => #WAT1)
   END_RUNG
   // the same network as SCL:
   #_w1 := NOT #RE_SET AND #CAN_9 AND NOT #XA_9 AND #XUNG_CLOCK AND NOT #A9;   // rising edge of #XUNG_CLOCK
   #A9 := #XUNG_CLOCK;
   IF #_w1 THEN #WAT1 := #WAT1 + #HS_NAP_WAT1; END_IF;
   #_w2 := NOT #RE_SET AND #XA_9 AND NOT #CAN_9 AND #XUNG_CLOCK AND NOT #B9;   // rising edge of #XUNG_CLOCK
   #B9 := #XUNG_CLOCK;
   IF #_w2 AND (#WAT1 > 0.0) THEN #WAT1 := #WAT1 - #HS_XA_WAT1; END_IF;
END_REGION

REGION Network 11: OUT10
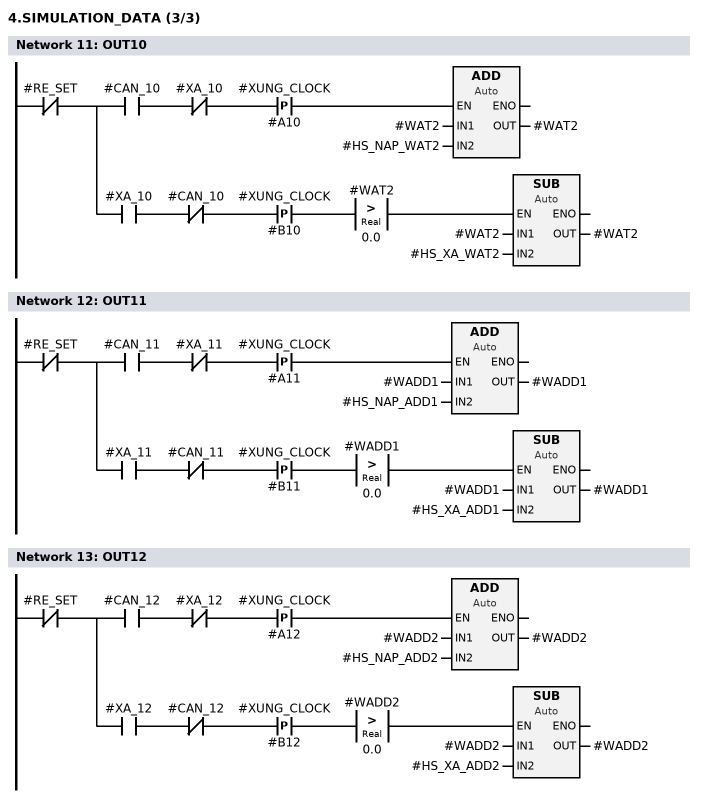
   RUNG wire#powerrail
      I_Contact( #RE_SET )
      wire#w1
      Contact( #CAN_10 )
      I_Contact( #XA_10 )
      P_Contact(operand := #XUNG_CLOCK, bit := #A10)
      Add(in1 := #WAT2, in2 := #HS_NAP_WAT2, out => #WAT2)
   END_RUNG
   RUNG wire#w1
      Contact( #XA_10 )
      I_Contact( #CAN_10 )
      P_Contact(operand := #XUNG_CLOCK, bit := #B10)
      { S7_Templates := "SrcType := Real" } GT_Contact(in1 := #WAT2, in2 := 0.0)
      Sub(in1 := #WAT2, in2 := #HS_XA_WAT2, out => #WAT2)
   END_RUNG
   // the same network as SCL:
   #_w1 := NOT #RE_SET AND #CAN_10 AND NOT #XA_10 AND #XUNG_CLOCK AND NOT #A10;   // rising edge of #XUNG_CLOCK
   #A10 := #XUNG_CLOCK;
   IF #_w1 THEN #WAT2 := #WAT2 + #HS_NAP_WAT2; END_IF;
   #_w2 := NOT #RE_SET AND #XA_10 AND NOT #CAN_10 AND #XUNG_CLOCK AND NOT #B10;   // rising edge of #XUNG_CLOCK
   #B10 := #XUNG_CLOCK;
   IF #_w2 AND (#WAT2 > 0.0) THEN #WAT2 := #WAT2 - #HS_XA_WAT2; END_IF;
END_REGION

REGION Network 12: OUT11
   RUNG wire#powerrail
      I_Contact( #RE_SET )
      wire#w1
      Contact( #CAN_11 )
      I_Contact( #XA_11 )
      P_Contact(operand := #XUNG_CLOCK, bit := #A11)
      Add(in1 := #WADD1, in2 := #HS_NAP_ADD1, out => #WADD1)
   END_RUNG
   RUNG wire#w1
      Contact( #XA_11 )
      I_Contact( #CAN_11 )
      P_Contact(operand := #XUNG_CLOCK, bit := #B11)
      { S7_Templates := "SrcType := Real" } GT_Contact(in1 := #WADD1, in2 := 0.0)
      Sub(in1 := #WADD1, in2 := #HS_XA_ADD1, out => #WADD1)
   END_RUNG
   // the same network as SCL:
   #_w1 := NOT #RE_SET AND #CAN_11 AND NOT #XA_11 AND #XUNG_CLOCK AND NOT #A11;   // rising edge of #XUNG_CLOCK
   #A11 := #XUNG_CLOCK;
   IF #_w1 THEN #WADD1 := #WADD1 + #HS_NAP_ADD1; END_IF;
   #_w2 := NOT #RE_SET AND #XA_11 AND NOT #CAN_11 AND #XUNG_CLOCK AND NOT #B11;   // rising edge of #XUNG_CLOCK
   #B11 := #XUNG_CLOCK;
   IF #_w2 AND (#WADD1 > 0.0) THEN #WADD1 := #WADD1 - #HS_XA_ADD1; END_IF;
END_REGION

REGION Network 13: OUT12
   RUNG wire#powerrail
      I_Contact( #RE_SET )
      wire#w1
      Contact( #CAN_12 )
      I_Contact( #XA_12 )
      P_Contact(operand := #XUNG_CLOCK, bit := #A12)
      Add(in1 := #WADD2, in2 := #HS_NAP_ADD2, out => #WADD2)
   END_RUNG
   RUNG wire#w1
      Contact( #XA_12 )
      I_Contact( #CAN_12 )
      P_Contact(operand := #XUNG_CLOCK, bit := #B12)
      { S7_Templates := "SrcType := Real" } GT_Contact(in1 := #WADD2, in2 := 0.0)
      Sub(in1 := #WADD2, in2 := #HS_XA_ADD2, out => #WADD2)
   END_RUNG
   // the same network as SCL:
   #_w1 := NOT #RE_SET AND #CAN_12 AND NOT #XA_12 AND #XUNG_CLOCK AND NOT #A12;   // rising edge of #XUNG_CLOCK
   #A12 := #XUNG_CLOCK;
   IF #_w1 THEN #WADD2 := #WADD2 + #HS_NAP_ADD2; END_IF;
   #_w2 := NOT #RE_SET AND #XA_12 AND NOT #CAN_12 AND #XUNG_CLOCK AND NOT #B12;   // rising edge of #XUNG_CLOCK
   #B12 := #XUNG_CLOCK;
   IF #_w2 AND (#WADD2 > 0.0) THEN #WADD2 := #WADD2 - #HS_XA_ADD2; END_IF;
END_REGION
END_FUNCTION_BLOCK

FUNCTION "FCXL_CCD_AGG12345" : Void   // FC9, LAD
{ S7_Optimized_Access := 'TRUE' }
VERSION : 0.1
// stored: AutoNumber true, CodeModifiedDate 2026-01-15T16:25:54.9938096Z, CompileDate 2026-01-15T16:25:55.0442288Z, CreationDate 2026-01-15T16:24:02.4619467Z, HandleErrorsWithinBlock false, InterfaceModifiedDate 2024-08-08T03:04:52.4075121Z, IsConsistent true, IsIECCheckEnabled false, IsKnowHowProtected false, IsWriteProtected false, LibraryConformanceStatus Error: The block contains calls of single instances. Warning: The object contains access to global data blocks. Warning: The block contains direct access to inputs, outputs, bit memories, indirect access to the registry or indirect access to external memory areas that are unknown at the time of compilation., ModifiedDate 2026-01-15T16:25:54.9938096Z, ParameterModified 2024-08-08T03:04:52.4075121Z, PLCSimAdvancedSupport false, SetENOAutomatically False, StructureModified 2024-08-08T03:04:52.4075121Z, UDAEnableTagReadback false
   VAR_TEMP   // added for the SCL form of the ladder/FBD networks
      _w1 : Bool;
      _w2 : Bool;
      _w3 : Bool;
   END_VAR
BEGIN

REGION Network 1: XU LY CAN AGG1
   // Các chân PV_IN và chân WR_IN không có tác dụng cho FB6
   // Mục đích của FB6 là xử lý giá trị cân WE_AG1 để biến nó thành cân có thể cân nhiều thành phần,bằng cách trừ bì thành phần đã cân trước đó
   // Chú ý tránh nhầm lẫn:
   // WE_AG1 hay những biến có chữ AG1 chưa chắc là dành cho cân thành phần AGG1 nhé, có thể nó là đang nói đến cái cân (thường có chữ W ở trước, ví dụ WE_AG1 là cái cân AGG nhé)
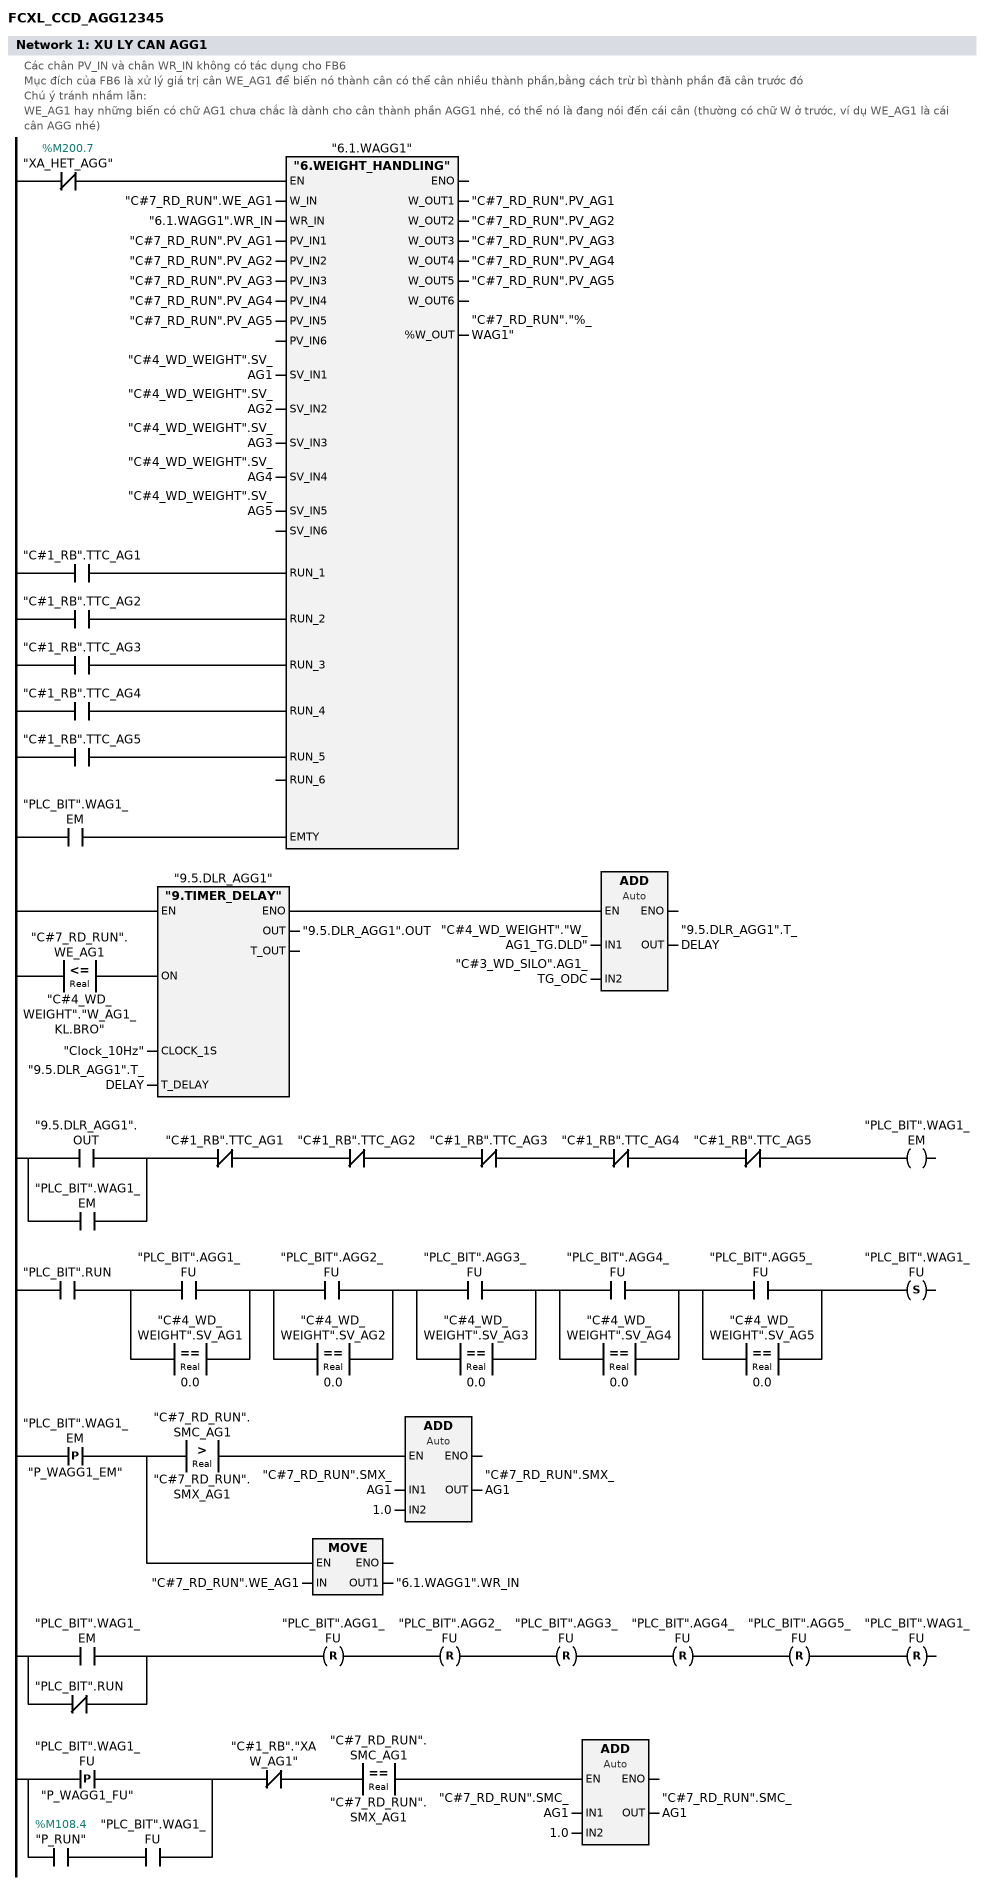
   RUNG wire#powerrail
      I_Contact( "XA_HET_AGG" )
      "6.1.WAGG1"(RUN_1 := wire#w1, RUN_2 := wire#w2, RUN_3 := wire#w3, RUN_4 := wire#w4, RUN_5 := wire#w5, EMTY := wire#w6, W_IN := "C#7_RD_RUN".WE_AG1, WR_IN := "6.1.WAGG1".WR_IN, PV_IN1 := "C#7_RD_RUN".PV_AG1, PV_IN2 := "C#7_RD_RUN".PV_AG2, PV_IN3 := "C#7_RD_RUN".PV_AG3, PV_IN4 := "C#7_RD_RUN".PV_AG4, PV_IN5 := "C#7_RD_RUN".PV_AG5, PV_IN6 :=, SV_IN1 := "C#4_WD_WEIGHT".SV_AG1, SV_IN2 := "C#4_WD_WEIGHT".SV_AG2, SV_IN3 := "C#4_WD_WEIGHT".SV_AG3, SV_IN4 := "C#4_WD_WEIGHT".SV_AG4, SV_IN5 := "C#4_WD_WEIGHT".SV_AG5, SV_IN6 :=, RUN_6 :=, W_OUT1 => "C#7_RD_RUN".PV_AG1, W_OUT2 => "C#7_RD_RUN".PV_AG2, W_OUT3 => "C#7_RD_RUN".PV_AG3, W_OUT4 => "C#7_RD_RUN".PV_AG4, W_OUT5 => "C#7_RD_RUN".PV_AG5, W_OUT6 =>, "%W_OUT" => "C#7_RD_RUN"."%_WAG1")
   END_RUNG
   RUNG wire#powerrail
      Contact( "C#1_RB".TTC_AG1 )
   END_RUNG wire#w1
   RUNG wire#powerrail
      Contact( "C#1_RB".TTC_AG2 )
   END_RUNG wire#w2
   RUNG wire#powerrail
      Contact( "C#1_RB".TTC_AG3 )
   END_RUNG wire#w3
   RUNG wire#powerrail
      Contact( "C#1_RB".TTC_AG4 )
   END_RUNG wire#w4
   RUNG wire#powerrail
      Contact( "C#1_RB".TTC_AG5 )
   END_RUNG wire#w5
   RUNG wire#powerrail
      Contact( "PLC_BIT".WAG1_EM )
   END_RUNG wire#w6
   RUNG wire#powerrail
      "9.5.DLR_AGG1"(ON := wire#w7, CLOCK_1S := "Clock_10Hz", T_DELAY := "9.5.DLR_AGG1".T_DELAY, OUT => "9.5.DLR_AGG1".OUT, T_OUT =>)
      Add(in1 := "C#4_WD_WEIGHT"."W_AG1_TG.DLD", in2 := "C#3_WD_SILO".AG1_TG_ODC, out => "9.5.DLR_AGG1".T_DELAY)
   END_RUNG
   RUNG wire#powerrail
      { S7_Templates := "SrcType := Real" } LE_Contact(in1 := "C#7_RD_RUN".WE_AG1, in2 := "C#4_WD_WEIGHT"."W_AG1_KL.BRO")
   END_RUNG wire#w7
   RUNG wire#powerrail
      Contact( "9.5.DLR_AGG1".OUT )
      wire#w8
      I_Contact( "C#1_RB".TTC_AG1 )
      I_Contact( "C#1_RB".TTC_AG2 )
      I_Contact( "C#1_RB".TTC_AG3 )
      I_Contact( "C#1_RB".TTC_AG4 )
      I_Contact( "C#1_RB".TTC_AG5 )
      Coil( "PLC_BIT".WAG1_EM )
   END_RUNG
   RUNG wire#powerrail
      Contact( "PLC_BIT".WAG1_EM )
   END_RUNG wire#w8
   RUNG wire#powerrail
      Contact( "PLC_BIT".RUN )
      wire#w9
      Contact( "PLC_BIT".AGG1_FU )
      wire#w10
      Contact( "PLC_BIT".AGG2_FU )
      wire#w11
      Contact( "PLC_BIT".AGG3_FU )
      wire#w12
      Contact( "PLC_BIT".AGG4_FU )
      wire#w13
      Contact( "PLC_BIT".AGG5_FU )
      wire#w14
      S_Coil( "PLC_BIT".WAG1_FU )
   END_RUNG
   RUNG wire#w9
      { S7_Templates := "SrcType := Real" } EQ_Contact(in1 := "C#4_WD_WEIGHT".SV_AG1, in2 := 0.0)
   END_RUNG wire#w10
   RUNG wire#w10
      { S7_Templates := "SrcType := Real" } EQ_Contact(in1 := "C#4_WD_WEIGHT".SV_AG2, in2 := 0.0)
   END_RUNG wire#w11
   RUNG wire#w11
      { S7_Templates := "SrcType := Real" } EQ_Contact(in1 := "C#4_WD_WEIGHT".SV_AG3, in2 := 0.0)
   END_RUNG wire#w12
   RUNG wire#w12
      { S7_Templates := "SrcType := Real" } EQ_Contact(in1 := "C#4_WD_WEIGHT".SV_AG4, in2 := 0.0)
   END_RUNG wire#w13
   RUNG wire#w13
      { S7_Templates := "SrcType := Real" } EQ_Contact(in1 := "C#4_WD_WEIGHT".SV_AG5, in2 := 0.0)
   END_RUNG wire#w14
   RUNG wire#powerrail
      P_Contact(operand := "PLC_BIT".WAG1_EM, bit := "P_WAGG1_EM")
      wire#w15
      { S7_Templates := "SrcType := Real" } GT_Contact(in1 := "C#7_RD_RUN".SMC_AG1, in2 := "C#7_RD_RUN".SMX_AG1)
      Add(in1 := "C#7_RD_RUN".SMX_AG1, in2 := 1.0, out => "C#7_RD_RUN".SMX_AG1)
   END_RUNG
   RUNG wire#w15
      Move(in := "C#7_RD_RUN".WE_AG1, out1 => "6.1.WAGG1".WR_IN)
   END_RUNG
   RUNG wire#powerrail
      Contact( "PLC_BIT".WAG1_EM )
      wire#w16
      R_Coil( "PLC_BIT".AGG1_FU )
      R_Coil( "PLC_BIT".AGG2_FU )
      R_Coil( "PLC_BIT".AGG3_FU )
      R_Coil( "PLC_BIT".AGG4_FU )
      R_Coil( "PLC_BIT".AGG5_FU )
      R_Coil( "PLC_BIT".WAG1_FU )
   END_RUNG
   RUNG wire#powerrail
      I_Contact( "PLC_BIT".RUN )
   END_RUNG wire#w16
   RUNG wire#powerrail
      P_Contact(operand := "PLC_BIT".WAG1_FU, bit := "P_WAGG1_FU")
      wire#w17
      I_Contact( "C#1_RB"."XA W_AG1" )
      { S7_Templates := "SrcType := Real" } EQ_Contact(in1 := "C#7_RD_RUN".SMC_AG1, in2 := "C#7_RD_RUN".SMX_AG1)
      Add(in1 := "C#7_RD_RUN".SMC_AG1, in2 := 1.0, out => "C#7_RD_RUN".SMC_AG1)
   END_RUNG
   RUNG wire#powerrail
      Contact( "P_RUN" )
      Contact( "PLC_BIT".WAG1_FU )
   END_RUNG wire#w17
   // the same network as SCL:
   IF NOT "XA_HET_AGG" THEN
       "6.1.WAGG1"(W_IN := "C#7_RD_RUN".WE_AG1,   // "6.WEIGHT_HANDLING"
                   WR_IN := "6.1.WAGG1".WR_IN,
                   PV_IN1 := "C#7_RD_RUN".PV_AG1,
                   PV_IN2 := "C#7_RD_RUN".PV_AG2,
                   PV_IN3 := "C#7_RD_RUN".PV_AG3,
                   PV_IN4 := "C#7_RD_RUN".PV_AG4,
                   PV_IN5 := "C#7_RD_RUN".PV_AG5,
                   SV_IN1 := "C#4_WD_WEIGHT".SV_AG1,
                   SV_IN2 := "C#4_WD_WEIGHT".SV_AG2,
                   SV_IN3 := "C#4_WD_WEIGHT".SV_AG3,
                   SV_IN4 := "C#4_WD_WEIGHT".SV_AG4,
                   SV_IN5 := "C#4_WD_WEIGHT".SV_AG5,
                   RUN_1 := "C#1_RB".TTC_AG1,
                   RUN_2 := "C#1_RB".TTC_AG2,
                   RUN_3 := "C#1_RB".TTC_AG3,
                   RUN_4 := "C#1_RB".TTC_AG4,
                   RUN_5 := "C#1_RB".TTC_AG5,
                   EMTY := "PLC_BIT".WAG1_EM,
                   W_OUT1 => "C#7_RD_RUN".PV_AG1,
                   W_OUT2 => "C#7_RD_RUN".PV_AG2,
                   W_OUT3 => "C#7_RD_RUN".PV_AG3,
                   W_OUT4 => "C#7_RD_RUN".PV_AG4,
                   W_OUT5 => "C#7_RD_RUN".PV_AG5,
                   "%W_OUT" => "C#7_RD_RUN"."%_WAG1");
   END_IF;
   "9.5.DLR_AGG1"(ON := "C#7_RD_RUN".WE_AG1 <= "C#4_WD_WEIGHT"."W_AG1_KL.BRO",   // "9.TIMER_DELAY"
                  CLOCK_1S := "Clock_10Hz",
                  T_DELAY := "9.5.DLR_AGG1".T_DELAY,
                  OUT => "9.5.DLR_AGG1".OUT,
                  ENO => #_w1);
   IF #_w1 THEN "9.5.DLR_AGG1".T_DELAY := "C#4_WD_WEIGHT"."W_AG1_TG.DLD" + "C#3_WD_SILO".AG1_TG_ODC; END_IF;
   "PLC_BIT".WAG1_EM := ("9.5.DLR_AGG1".OUT OR "PLC_BIT".WAG1_EM) AND NOT "C#1_RB".TTC_AG1 AND NOT "C#1_RB".TTC_AG2 AND NOT "C#1_RB".TTC_AG3 AND NOT "C#1_RB".TTC_AG4 AND NOT "C#1_RB".TTC_AG5;
   IF "PLC_BIT".RUN AND ("PLC_BIT".AGG1_FU OR ("C#4_WD_WEIGHT".SV_AG1 = 0.0)) AND ("PLC_BIT".AGG2_FU OR ("C#4_WD_WEIGHT".SV_AG2 = 0.0)) AND ("PLC_BIT".AGG3_FU OR ("C#4_WD_WEIGHT".SV_AG3 = 0.0)) AND ("PLC_BIT".AGG4_FU OR ("C#4_WD_WEIGHT".SV_AG4 = 0.0)) AND ("PLC_BIT".AGG5_FU OR ("C#4_WD_WEIGHT".SV_AG5 = 0.0)) THEN
       "PLC_BIT".WAG1_FU := TRUE;
   END_IF;
   #_w2 := "PLC_BIT".WAG1_EM AND NOT "P_WAGG1_EM";   // rising edge of "PLC_BIT".WAG1_EM
   "P_WAGG1_EM" := "PLC_BIT".WAG1_EM;
   IF #_w2 AND ("C#7_RD_RUN".SMC_AG1 > "C#7_RD_RUN".SMX_AG1) THEN
       "C#7_RD_RUN".SMX_AG1 := "C#7_RD_RUN".SMX_AG1 + 1.0;
   END_IF;
   IF #_w2 THEN "6.1.WAGG1".WR_IN := "C#7_RD_RUN".WE_AG1; END_IF;
   IF "PLC_BIT".WAG1_EM OR NOT "PLC_BIT".RUN THEN
       "PLC_BIT".AGG1_FU := FALSE;
       "PLC_BIT".AGG2_FU := FALSE;
       "PLC_BIT".AGG3_FU := FALSE;
       "PLC_BIT".AGG4_FU := FALSE;
       "PLC_BIT".AGG5_FU := FALSE;
       "PLC_BIT".WAG1_FU := FALSE;
   END_IF;
   #_w3 := "PLC_BIT".WAG1_FU AND NOT "P_WAGG1_FU";   // rising edge of "PLC_BIT".WAG1_FU
   "P_WAGG1_FU" := "PLC_BIT".WAG1_FU;
   IF (#_w3 OR ("P_RUN" AND "PLC_BIT".WAG1_FU)) AND NOT "C#1_RB"."XA W_AG1" AND ("C#7_RD_RUN".SMC_AG1 = "C#7_RD_RUN".SMX_AG1) THEN
       "C#7_RD_RUN".SMC_AG1 := "C#7_RD_RUN".SMC_AG1 + 1.0;
   END_IF;
END_REGION
END_FUNCTION

FUNCTION_BLOCK "6.WEIGHT_HANDLING"   // FB6, LAD
{ S7_Optimized_Access := 'TRUE' }
VERSION : 0.1
// stored: AutoNumber false, CodeModifiedDate 2025-08-27T17:12:27.5610885Z, CompileDate 2026-01-15T16:25:50.7557128Z, CreationDate 2026-01-15T16:22:49.8270549Z, DownloadWithoutReinit false, HandleErrorsWithinBlock false, InterfaceModifiedDate 2023-12-29T17:39:18.5236469Z, IsConsistent true, IsIECCheckEnabled false, IsKnowHowProtected false, IsRetainMemResEnabled false, IsWriteProtected false, LibraryConformanceStatus The object is library-conformant., MemoryReserve 100, ModifiedDate 2025-08-27T17:12:27.5610885Z, ParameterModified 2023-11-29T03:49:57.2782849Z, PLCSimAdvancedSupport false, SetENOAutomatically False, StructureModified 2023-12-29T17:39:18.5236469Z, UDAEnableTagReadback false
   VAR_INPUT
      W_IN { ExternalAccessible := 'False'; ExternalVisible := 'False'; ExternalWritable := 'False'} : Real;
      WR_IN : Real;
      PV_IN1 : Real;
      PV_IN2 : Real;
      PV_IN3 : Real;
      PV_IN4 : Real;
      PV_IN5 : Real;
      PV_IN6 : Real;
      SV_IN1 : Real;
      SV_IN2 : Real;
      SV_IN3 : Real;
      SV_IN4 : Real;
      SV_IN5 : Real;
      SV_IN6 : Real;
      RUN_1 { ExternalAccessible := 'False'; ExternalVisible := 'False'; ExternalWritable := 'False'} : Bool;
      RUN_2 { ExternalAccessible := 'False'; ExternalVisible := 'False'; ExternalWritable := 'False'} : Bool;
      RUN_3 { ExternalAccessible := 'False'; ExternalVisible := 'False'; ExternalWritable := 'False'} : Bool;
      RUN_4 { ExternalAccessible := 'False'; ExternalVisible := 'False'; ExternalWritable := 'False'} : Bool;
      RUN_5 { ExternalAccessible := 'False'; ExternalVisible := 'False'; ExternalWritable := 'False'} : Bool;
      RUN_6 { ExternalAccessible := 'False'; ExternalVisible := 'False'; ExternalWritable := 'False'} : Bool;
      EMTY { ExternalAccessible := 'False'; ExternalVisible := 'False'; ExternalWritable := 'False'} : Bool;
   END_VAR
   VAR_OUTPUT
      W_OUT1 { ExternalAccessible := 'False'; ExternalVisible := 'False'; ExternalWritable := 'False'} : Real;
      W_OUT2 { ExternalAccessible := 'False'; ExternalVisible := 'False'; ExternalWritable := 'False'} : Real;
      W_OUT3 { ExternalAccessible := 'False'; ExternalVisible := 'False'; ExternalWritable := 'False'} : Real;
      W_OUT4 { ExternalAccessible := 'False'; ExternalVisible := 'False'; ExternalWritable := 'False'} : Real;
      W_OUT5 { ExternalAccessible := 'False'; ExternalVisible := 'False'; ExternalWritable := 'False'} : Real;
      W_OUT6 { ExternalAccessible := 'False'; ExternalVisible := 'False'; ExternalWritable := 'False'} : Real;
      "%W_OUT" { ExternalAccessible := 'False'; ExternalVisible := 'False'; ExternalWritable := 'False'} : Real;
   END_VAR
   VAR RETAIN
      W_Star : Real;
      W_Temp : Real;
   END_VAR
   VAR
      P_RUN1 : Bool;
      P_RUN2 : Bool;
      P_RUN3 : Bool;
      P_RUN4 : Bool;
      P_RUN5 : Bool;
      P_RUN6 : Bool;
      N_RUN1 : Bool;
      N_RUN2 : Bool;
      N_RUN3 : Bool;
      N_RUN4 : Bool;
      N_RUN5 : Bool;
      N_RUN6 : Bool;
   END_VAR
   VAR RETAIN
      PV1 : Real;
      PV2 : Real;
      PV3 : Real;
      PV4 : Real;
      PV5 : Real;
      PV6 : Real;
   END_VAR
   VAR_TEMP   // added for the SCL form of the ladder/FBD networks
      _w1 : Bool;
      _w2 : Bool;
      _w3 : Bool;
      _w4 : Bool;
      _w5 : Bool;
      _w6 : Bool;
   END_VAR
BEGIN

REGION Network 1
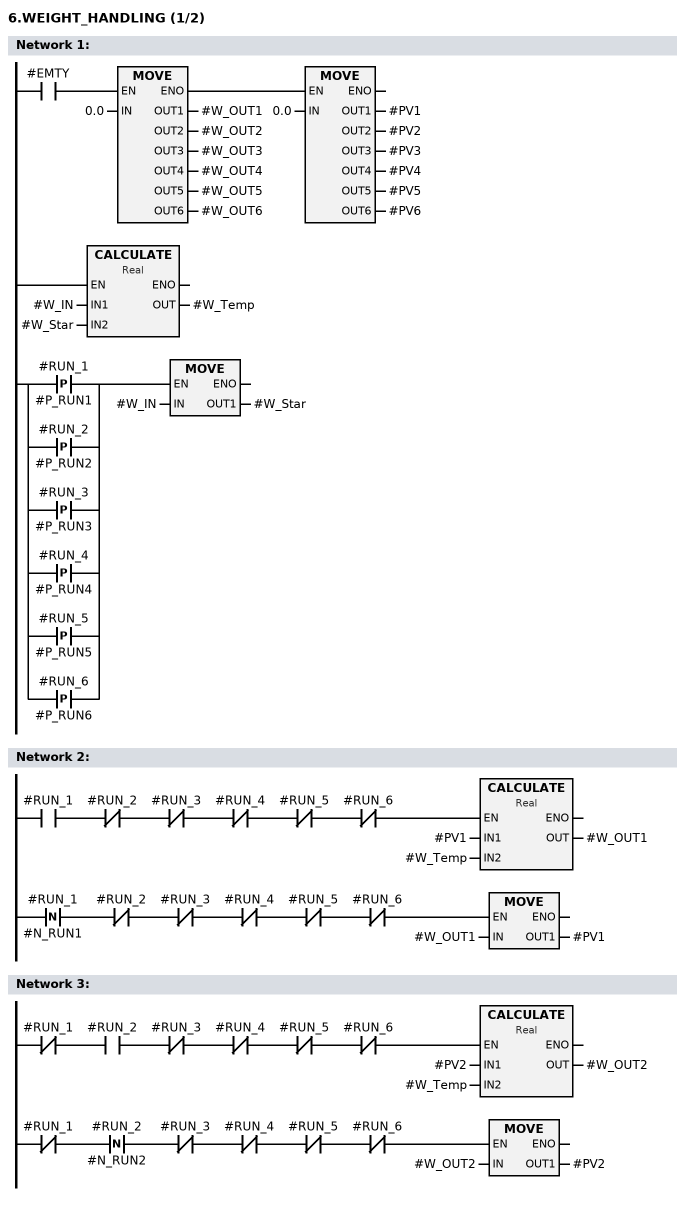
   RUNG wire#powerrail
      Contact( #EMTY )
      Move(in := 0.0, out1 => #W_OUT1, out2 => #W_OUT2, out3 => #W_OUT3, out4 => #W_OUT4, out5 => #W_OUT5, out6 => #W_OUT6)
      Move(in := 0.0, out1 => #PV1, out2 => #PV2, out3 => #PV3, out4 => #PV4, out5 => #PV5, out6 => #PV6)
   END_RUNG
   RUNG wire#powerrail
      { S7_Templates := "SrcType := Real"; S7_Expression := "IN1-IN2" } Calculate(in1 := #W_IN, in2 := #W_Star, out => #W_Temp)
   END_RUNG
   RUNG wire#powerrail
      P_Contact(operand := #RUN_1, bit := #P_RUN1)
      wire#w1
      Move(in := #W_IN, out1 => #W_Star)
   END_RUNG
   RUNG wire#powerrail
      P_Contact(operand := #RUN_2, bit := #P_RUN2)
   END_RUNG wire#w1
   RUNG wire#powerrail
      P_Contact(operand := #RUN_3, bit := #P_RUN3)
   END_RUNG wire#w1
   RUNG wire#powerrail
      P_Contact(operand := #RUN_4, bit := #P_RUN4)
   END_RUNG wire#w1
   RUNG wire#powerrail
      P_Contact(operand := #RUN_5, bit := #P_RUN5)
   END_RUNG wire#w1
   RUNG wire#powerrail
      P_Contact(operand := #RUN_6, bit := #P_RUN6)
   END_RUNG wire#w1
   // the same network as SCL:
   IF #EMTY THEN
       #W_OUT1 := 0.0;
       #W_OUT2 := 0.0;
       #W_OUT3 := 0.0;
       #W_OUT4 := 0.0;
       #W_OUT5 := 0.0;
       #W_OUT6 := 0.0;
       #PV1 := 0.0;
       #PV2 := 0.0;
       #PV3 := 0.0;
       #PV4 := 0.0;
       #PV5 := 0.0;
       #PV6 := 0.0;
   END_IF;
   #W_Temp := #W_IN-#W_Star;
   #_w1 := #RUN_1 AND NOT #P_RUN1;   // rising edge of #RUN_1
   #P_RUN1 := #RUN_1;
   #_w2 := #RUN_2 AND NOT #P_RUN2;   // rising edge of #RUN_2
   #P_RUN2 := #RUN_2;
   #_w3 := #RUN_3 AND NOT #P_RUN3;   // rising edge of #RUN_3
   #P_RUN3 := #RUN_3;
   #_w4 := #RUN_4 AND NOT #P_RUN4;   // rising edge of #RUN_4
   #P_RUN4 := #RUN_4;
   #_w5 := #RUN_5 AND NOT #P_RUN5;   // rising edge of #RUN_5
   #P_RUN5 := #RUN_5;
   #_w6 := #RUN_6 AND NOT #P_RUN6;   // rising edge of #RUN_6
   #P_RUN6 := #RUN_6;
   IF #_w1 OR #_w2 OR #_w3 OR #_w4 OR #_w5 OR #_w6 THEN #W_Star := #W_IN; END_IF;
END_REGION

REGION Network 2
   RUNG wire#powerrail
      Contact( #RUN_1 )
      I_Contact( #RUN_2 )
      I_Contact( #RUN_3 )
      I_Contact( #RUN_4 )
      I_Contact( #RUN_5 )
      I_Contact( #RUN_6 )
      { S7_Templates := "SrcType := Real"; S7_Expression := "IN1+IN2" } Calculate(in1 := #PV1, in2 := #W_Temp, out => #W_OUT1)
   END_RUNG
   RUNG wire#powerrail
      N_Contact(operand := #RUN_1, bit := #N_RUN1)
      I_Contact( #RUN_2 )
      I_Contact( #RUN_3 )
      I_Contact( #RUN_4 )
      I_Contact( #RUN_5 )
      I_Contact( #RUN_6 )
      Move(in := #W_OUT1, out1 => #PV1)
   END_RUNG
   // the same network as SCL:
   IF #RUN_1 AND NOT #RUN_2 AND NOT #RUN_3 AND NOT #RUN_4 AND NOT #RUN_5 AND NOT #RUN_6 THEN
       #W_OUT1 := #PV1+#W_Temp;
   END_IF;
   #_w1 := NOT #RUN_1 AND #N_RUN1;   // falling edge of #RUN_1
   #N_RUN1 := #RUN_1;
   IF #_w1 AND NOT #RUN_2 AND NOT #RUN_3 AND NOT #RUN_4 AND NOT #RUN_5 AND NOT #RUN_6 THEN
       #PV1 := #W_OUT1;
   END_IF;
END_REGION

REGION Network 3
   RUNG wire#powerrail
      I_Contact( #RUN_1 )
      Contact( #RUN_2 )
      I_Contact( #RUN_3 )
      I_Contact( #RUN_4 )
      I_Contact( #RUN_5 )
      I_Contact( #RUN_6 )
      { S7_Templates := "SrcType := Real"; S7_Expression := "IN1+IN2" } Calculate(in1 := #PV2, in2 := #W_Temp, out => #W_OUT2)
   END_RUNG
   RUNG wire#powerrail
      I_Contact( #RUN_1 )
      N_Contact(operand := #RUN_2, bit := #N_RUN2)
      I_Contact( #RUN_3 )
      I_Contact( #RUN_4 )
      I_Contact( #RUN_5 )
      I_Contact( #RUN_6 )
      Move(in := #W_OUT2, out1 => #PV2)
   END_RUNG
   // the same network as SCL:
   IF NOT #RUN_1 AND #RUN_2 AND NOT #RUN_3 AND NOT #RUN_4 AND NOT #RUN_5 AND NOT #RUN_6 THEN
       #W_OUT2 := #PV2+#W_Temp;
   END_IF;
   #_w1 := NOT #RUN_1 AND NOT #RUN_2 AND #N_RUN2;   // falling edge of #RUN_2
   #N_RUN2 := #RUN_2;
   IF #_w1 AND NOT #RUN_3 AND NOT #RUN_4 AND NOT #RUN_5 AND NOT #RUN_6 THEN #PV2 := #W_OUT2; END_IF;
END_REGION

REGION Network 4
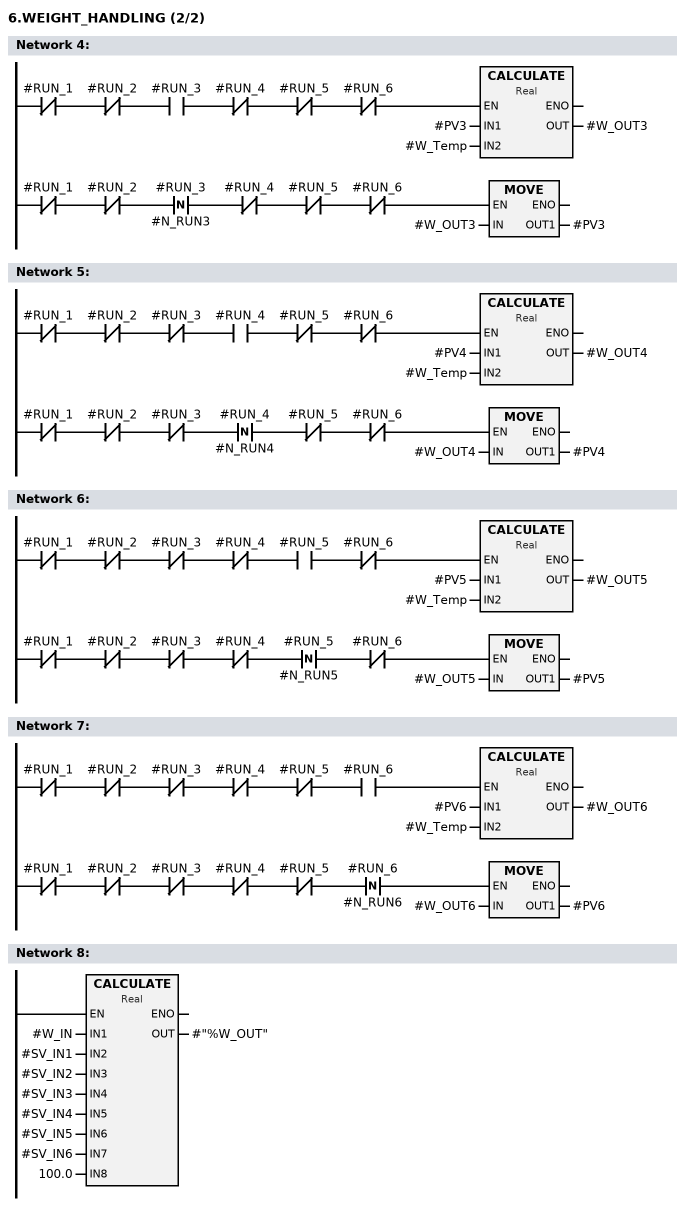
   RUNG wire#powerrail
      I_Contact( #RUN_1 )
      I_Contact( #RUN_2 )
      Contact( #RUN_3 )
      I_Contact( #RUN_4 )
      I_Contact( #RUN_5 )
      I_Contact( #RUN_6 )
      { S7_Templates := "SrcType := Real"; S7_Expression := "IN1+IN2" } Calculate(in1 := #PV3, in2 := #W_Temp, out => #W_OUT3)
   END_RUNG
   RUNG wire#powerrail
      I_Contact( #RUN_1 )
      I_Contact( #RUN_2 )
      N_Contact(operand := #RUN_3, bit := #N_RUN3)
      I_Contact( #RUN_4 )
      I_Contact( #RUN_5 )
      I_Contact( #RUN_6 )
      Move(in := #W_OUT3, out1 => #PV3)
   END_RUNG
   // the same network as SCL:
   IF NOT #RUN_1 AND NOT #RUN_2 AND #RUN_3 AND NOT #RUN_4 AND NOT #RUN_5 AND NOT #RUN_6 THEN
       #W_OUT3 := #PV3+#W_Temp;
   END_IF;
   #_w1 := NOT #RUN_1 AND NOT #RUN_2 AND NOT #RUN_3 AND #N_RUN3;   // falling edge of #RUN_3
   #N_RUN3 := #RUN_3;
   IF #_w1 AND NOT #RUN_4 AND NOT #RUN_5 AND NOT #RUN_6 THEN #PV3 := #W_OUT3; END_IF;
END_REGION

REGION Network 5
   RUNG wire#powerrail
      I_Contact( #RUN_1 )
      I_Contact( #RUN_2 )
      I_Contact( #RUN_3 )
      Contact( #RUN_4 )
      I_Contact( #RUN_5 )
      I_Contact( #RUN_6 )
      { S7_Templates := "SrcType := Real"; S7_Expression := "IN1+IN2" } Calculate(in1 := #PV4, in2 := #W_Temp, out => #W_OUT4)
   END_RUNG
   RUNG wire#powerrail
      I_Contact( #RUN_1 )
      I_Contact( #RUN_2 )
      I_Contact( #RUN_3 )
      N_Contact(operand := #RUN_4, bit := #N_RUN4)
      I_Contact( #RUN_5 )
      I_Contact( #RUN_6 )
      Move(in := #W_OUT4, out1 => #PV4)
   END_RUNG
   // the same network as SCL:
   IF NOT #RUN_1 AND NOT #RUN_2 AND NOT #RUN_3 AND #RUN_4 AND NOT #RUN_5 AND NOT #RUN_6 THEN
       #W_OUT4 := #PV4+#W_Temp;
   END_IF;
   #_w1 := NOT #RUN_1 AND NOT #RUN_2 AND NOT #RUN_3 AND NOT #RUN_4 AND #N_RUN4;   // falling edge of #RUN_4
   #N_RUN4 := #RUN_4;
   IF #_w1 AND NOT #RUN_5 AND NOT #RUN_6 THEN #PV4 := #W_OUT4; END_IF;
END_REGION

REGION Network 6
   RUNG wire#powerrail
      I_Contact( #RUN_1 )
      I_Contact( #RUN_2 )
      I_Contact( #RUN_3 )
      I_Contact( #RUN_4 )
      Contact( #RUN_5 )
      I_Contact( #RUN_6 )
      { S7_Templates := "SrcType := Real"; S7_Expression := "IN1+IN2" } Calculate(in1 := #PV5, in2 := #W_Temp, out => #W_OUT5)
   END_RUNG
   RUNG wire#powerrail
      I_Contact( #RUN_1 )
      I_Contact( #RUN_2 )
      I_Contact( #RUN_3 )
      I_Contact( #RUN_4 )
      N_Contact(operand := #RUN_5, bit := #N_RUN5)
      I_Contact( #RUN_6 )
      Move(in := #W_OUT5, out1 => #PV5)
   END_RUNG
   // the same network as SCL:
   IF NOT #RUN_1 AND NOT #RUN_2 AND NOT #RUN_3 AND NOT #RUN_4 AND #RUN_5 AND NOT #RUN_6 THEN
       #W_OUT5 := #PV5+#W_Temp;
   END_IF;
   #_w1 := NOT #RUN_1 AND NOT #RUN_2 AND NOT #RUN_3 AND NOT #RUN_4 AND NOT #RUN_5 AND #N_RUN5;   // falling edge of #RUN_5
   #N_RUN5 := #RUN_5;
   IF #_w1 AND NOT #RUN_6 THEN #PV5 := #W_OUT5; END_IF;
END_REGION

REGION Network 7
   RUNG wire#powerrail
      I_Contact( #RUN_1 )
      I_Contact( #RUN_2 )
      I_Contact( #RUN_3 )
      I_Contact( #RUN_4 )
      I_Contact( #RUN_5 )
      Contact( #RUN_6 )
      { S7_Templates := "SrcType := Real"; S7_Expression := "IN1+IN2" } Calculate(in1 := #PV6, in2 := #W_Temp, out => #W_OUT6)
   END_RUNG
   RUNG wire#powerrail
      I_Contact( #RUN_1 )
      I_Contact( #RUN_2 )
      I_Contact( #RUN_3 )
      I_Contact( #RUN_4 )
      I_Contact( #RUN_5 )
      N_Contact(operand := #RUN_6, bit := #N_RUN6)
      Move(in := #W_OUT6, out1 => #PV6)
   END_RUNG
   // the same network as SCL:
   IF NOT #RUN_1 AND NOT #RUN_2 AND NOT #RUN_3 AND NOT #RUN_4 AND NOT #RUN_5 AND #RUN_6 THEN
       #W_OUT6 := #PV6+#W_Temp;
   END_IF;
   #_w1 := NOT #RUN_1 AND NOT #RUN_2 AND NOT #RUN_3 AND NOT #RUN_4 AND NOT #RUN_5 AND NOT #RUN_6 AND #N_RUN6;   // falling edge of #RUN_6
   #N_RUN6 := #RUN_6;
   IF #_w1 THEN #PV6 := #W_OUT6; END_IF;
END_REGION

REGION Network 8
   RUNG wire#powerrail
      { S7_Templates := "SrcType := Real"; S7_Expression := "(IN1/(IN2+IN3+IN4+IN5+IN6+IN7))*IN8" } Calculate(in1 := #W_IN, in2 := #SV_IN1, in3 := #SV_IN2, in4 := #SV_IN3, in5 := #SV_IN4, in6 := #SV_IN5, in7 := #SV_IN6, in8 := 100.0, out => #"%W_OUT")
   END_RUNG
   // the same network as SCL:
   #"%W_OUT" := (#W_IN/(#SV_IN1+#SV_IN2+#SV_IN3+#SV_IN4+#SV_IN5+#SV_IN6))*100.0;
END_REGION
END_FUNCTION_BLOCK

FUNCTION_BLOCK "9.TIMER_DELAY"   // FB9, LAD
{ S7_Optimized_Access := 'TRUE' }
VERSION : 0.1
// stored: AutoNumber false, CodeModifiedDate 2025-08-27T17:13:13.1552526Z, CompileDate 2026-01-15T16:25:50.0427227Z, CreationDate 2026-01-15T16:22:49.8270549Z, DownloadWithoutReinit false, HandleErrorsWithinBlock false, InterfaceModifiedDate 2022-05-24T16:36:11.1705081Z, IsConsistent true, IsIECCheckEnabled false, IsKnowHowProtected false, IsRetainMemResEnabled false, IsWriteProtected false, LibraryConformanceStatus The object is library-conformant., MemoryReserve 100, ModifiedDate 2025-08-27T17:13:13.1552526Z, ParameterModified 2022-05-24T16:36:11.1705081Z, PLCSimAdvancedSupport false, SetENOAutomatically False, StructureModified 2022-05-24T16:36:11.1705081Z, UDAEnableTagReadback false
   VAR_INPUT
      ON : Bool;
      CLOCK_1S : Bool;
      T_DELAY : Real;
   END_VAR
   VAR_OUTPUT
      OUT : Bool;
      T_OUT : Real;
   END_VAR
   VAR
      TDL : Real;
      CLK : Bool;
   END_VAR
   VAR_TEMP   // added for the SCL form of the ladder/FBD networks
      _w1 : Bool;
   END_VAR
BEGIN

REGION Network 1
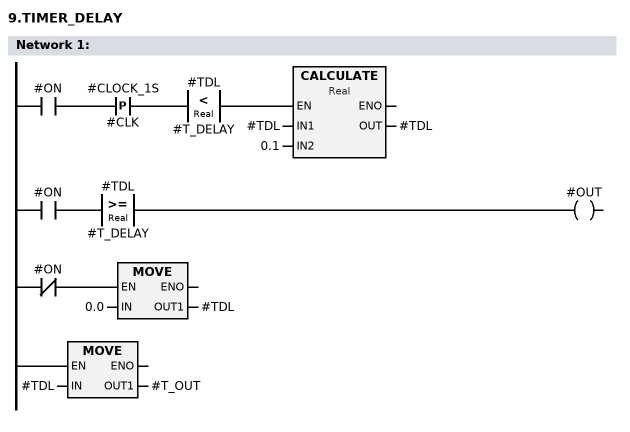
   RUNG wire#powerrail
      Contact( #ON )
      P_Contact(operand := #CLOCK_1S, bit := #CLK)
      { S7_Templates := "SrcType := Real" } LT_Contact(in1 := #TDL, in2 := #T_DELAY)
      { S7_Templates := "SrcType := Real"; S7_Expression := "IN1+IN2" } Calculate(in1 := #TDL, in2 := 0.1, out => #TDL)
   END_RUNG
   RUNG wire#powerrail
      Contact( #ON )
      { S7_Templates := "SrcType := Real" } GE_Contact(in1 := #TDL, in2 := #T_DELAY)
      Coil( #OUT )
   END_RUNG
   RUNG wire#powerrail
      I_Contact( #ON )
      Move(in := 0.0, out1 => #TDL)
   END_RUNG
   RUNG wire#powerrail
      Move(in := #TDL, out1 => #T_OUT)
   END_RUNG
   // the same network as SCL:
   #_w1 := #ON AND #CLOCK_1S AND NOT #CLK;   // rising edge of #CLOCK_1S
   #CLK := #CLOCK_1S;
   IF #_w1 AND (#TDL < #T_DELAY) THEN #TDL := #TDL+0.1; END_IF;
   #OUT := #ON AND (#TDL >= #T_DELAY);
   IF NOT #ON THEN #TDL := 0.0; END_IF;
   #T_OUT := #TDL;
END_REGION
END_FUNCTION_BLOCK

FUNCTION "FCCA_CCD_AGG12345" : Void   // FC19, LAD
{ S7_Optimized_Access := 'TRUE' }
VERSION : 0.1
// stored: AutoNumber true, CodeModifiedDate 2026-01-15T16:25:54.1563722Z, CompileDate 2026-01-15T16:25:54.3013674Z, CreationDate 2026-01-15T16:24:02.4619467Z, HandleErrorsWithinBlock false, InterfaceModifiedDate 2024-08-08T03:15:59.3806622Z, IsConsistent true, IsIECCheckEnabled false, IsKnowHowProtected false, IsWriteProtected false, LibraryConformanceStatus Error: The block contains calls of single instances. Warning: The object contains access to global data blocks. Warning: The block contains direct access to inputs, outputs, bit memories, indirect access to the registry or indirect access to external memory areas that are unknown at the time of compilation., ModifiedDate 2026-01-15T16:25:54.1563722Z, ParameterModified 2024-08-08T03:15:59.3806622Z, PLCSimAdvancedSupport false, SetENOAutomatically False, StructureModified 2024-08-08T03:15:59.3806622Z, UDAEnableTagReadback false
   VAR_TEMP   // added for the SCL form of the ladder/FBD networks
      _w1 : Bool;
   END_VAR
BEGIN

